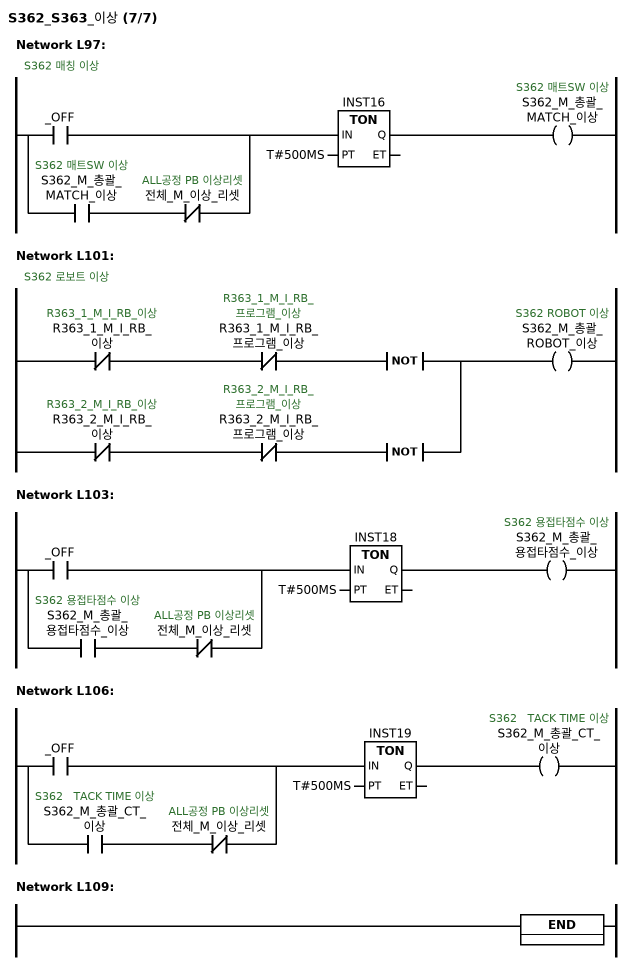
(* [picture p144: S362_S363_이상 rungs L97-L109] *)
(* S362 매칭 이상 *)
(* Rung L97 *)
INST16(IN := _OFF OR (S362_M_총괄_MATCH_이상 AND NOT 전체_M_이상_리셋), PT := T#500MS);
S362_M_총괄_MATCH_이상 := INST16.Q;
(* S362 로보트 이상 *)
(* Rung L101 *)
S362_M_총괄_ROBOT_이상 := NOT (NOT R363_1_M_I_RB_이상 AND NOT R363_1_M_I_RB_프로그램_이상) OR NOT (NOT R363_2_M_I_RB_이상 AND NOT R363_2_M_I_RB_프로그램_이상);
(* Rung L103 *)
INST18(IN := _OFF OR (S362_M_총괄_용접타점수_이상 AND NOT 전체_M_이상_리셋), PT := T#500MS);
S362_M_총괄_용접타점수_이상 := INST18.Q;
(* Rung L106 *)
INST19(IN := _OFF OR (S362_M_총괄_CT_이상 AND NOT 전체_M_이상_리셋), PT := T#500MS);
S362_M_총괄_CT_이상 := INST19.Q;
(* Rung L109 *)
END();
END_PROGRAM

PROGRAM S364_유틸리티 (* task: 스캔 프로그램 *)
VAR_EXTERNAL
    EGIS_CWS : BOOL;
    HOP_PBL_운전준비_ON : BOOL; (* AT %MW87500.0 *) (* HOP_PBL_운전준비_ON *)
    HOP_PLB_362_4_자동_운전 : BOOL; (* AT %MW87500.4 *) (* HOP PLB 362~4 자동기동 *)
    HOP_SSP_362_4_수동_선택 : BOOL; (* AT %MW87500.3 *) (* HOP 362~4 수동선택 *)
    HOP_SSP_362_4_자동_선택 : BOOL; (* AT %MW87500.2 *) (* HOP 362~4 자동선택 *)
    MCP_PBL_362_4_자동_운전 : BOOL; (* AT %MW87630.4 *) (* MCP PBL 362~4 자동기동 *)
    MCP_PBL_운전준비_ON : BOOL; (* AT %MW87630.0 *) (* MCP_PBL_운전준비_ON *)
    MCP_SPB_작업완료_RESET : BOOL; (* AT %MW87631.6 *) (* MCP_SPB_작업완료_RESET *)
    MCP_SPB_작업완료_SET : BOOL; (* AT %MW87631.7 *) (* MCP_SPB_작업완료_SET *)
    MCP_SSP_362_4_수동_선택 : BOOL; (* AT %MW87630.2 *) (* MCP 362~4 수동선택 *)
    MCP_SSP_362_4_자동_선택 : BOOL; (* AT %MW87630.3 *) (* MCP 362~4 자동동선택 *)
    R361_1_M_I_RB_1차_작업완료 : BOOL; (* AT %MW20011.2 *) (* R361_1_M_I_RB_1차_작업완료 *)
    R361_1_M_I_RB_2차_작업완료 : BOOL; (* AT %MW20011.3 *) (* R361_1_M_I_RB_2차_작업완료 *)
    R361_2_M_I_RB_2차_작업완료 : BOOL; (* AT %MW20021.3 *) (* R361_2_M_I_RB_2차_작업완료 *)
    R361_2_M_I_RB_간섭무_1 : BOOL; (* AT %MW20022.0 *) (* R361_2_M_I_RB_간섭무_1 *)
    R361_2_M_I_RB_원위치 : BOOL; (* AT %MW20020.3 *) (* R361_2_M_I_RB_원위치 *)
    R363_2_M_I_RB_간섭무_1 : BOOL; (* AT %MW20042.0 *) (* R363_2_M_I_RB_간섭무_1 *)
    R363_2_M_I_RB_원위치 : BOOL; (* AT %MW20040.3 *) (* R363_2_M_I_RB_원위치 *)
    R364_1_M_I_RB_1차_작업완료 : BOOL; (* AT %MW20051.2 *) (* R364_1_M_I_RB_1차_작업완료 *)
    R364_1_M_I_RB_간섭무_1 : BOOL; (* AT %MW20052.0 *) (* R364_1_M_I_RB_간섭무_1 *)
    R364_1_M_I_RB_원위치 : BOOL; (* AT %MW20050.3 *) (* R364_1_M_I_RB_원위치 *)
    S362_LC_정상1 : BOOL; (* AT %MW87105.3 *)
    S362_LC_정상2 : BOOL; (* AT %MW87105.4 *)
    S362_MAT_정상1 : BOOL; (* AT %MW87105.6 *)
    S362_MAT_정상2 : BOOL; (* AT %MW87105.7 *)
    S364_LC_정상1 : BOOL; (* AT %MW87165.3 *)
    S364_LC_정상2 : BOOL; (* AT %MW87165.4 *)
    S364_MAT_정상1 : BOOL; (* AT %MW87165.6 *)
    S364_MAT_정상2 : BOOL; (* AT %MW87165.7 *)
    S364_PB_AX_작업_완료 : BOOL; (* AT %MW87152.9 *) (* S364_PB_AX_작업_완료 *)
    S364_PRS_AX_LH_RACK_CHK1 : BOOL; (* AT %MW87162.0 *) (* S364_PRS_AX_LH_RACK_CHK1 *)
    S364_PRS_AX_LH_RACK_CHK2 : BOOL; (* AT %MW87162.1 *) (* S364_PRS_AX_LH_RACK_CHK2 *)
    S364_PRS_AX_LH_RACK_CHK3 : BOOL; (* AT %MW87162.2 *) (* S364_PRS_AX_LH_RACK_CHK3 *)
    S364_PRS_AX_LH_ROOF_FRT_CHK : BOOL; (* AT %MW87162.3 *) (* S364_PRS_AX_LH_ROOF_FRT_CHK *)
    S364_PRS_AX_LH_ROOF_RR_CHK : BOOL; (* AT %MW87162.4 *) (* S364_PRS_AX_LH_ROOF_RR_CHK *)
    S364_PRS_AX_RH_RACK_CHK1 : BOOL; (* AT %MW87152.0 *) (* S364_PRS_AX_RH_RACK_CHK1 *)
    S364_PRS_AX_RH_RACK_CHK2 : BOOL; (* AT %MW87152.1 *) (* S364_PRS_AX_RH_RACK_CHK2 *)
    S364_PRS_AX_RH_RACK_CHK3 : BOOL; (* AT %MW87152.2 *) (* S364_PRS_AX_RH_RACK_CHK3 *)
    S364_PRS_AX_RH_ROOF_FRT_CHK : BOOL; (* AT %MW87152.3 *) (* S364_PRS_AX_RH_ROOF_FRT_CHK *)
    S364_PRS_AX_RH_ROOF_RR_CHK : BOOL; (* AT %MW87152.4 *) (* S364_PRS_AX_RH_ROOF_RR_CHK *)
END_VAR
VAR_EXTERNAL RETAIN
    HMI_M_선택_MOD_S362 : BOOL; (* AT %MW6.0 *) (* HMI M 선택 MOD S362 *)
    HMI_M_선택_MOD_S364 : BOOL; (* AT %MW6.2 *) (* HMI M 선택 MOD S364 *)
    S362_M_BYPASS_보조 : BOOL; (* AT %MW1003.15 *) (* S362 M BYPASS 보조 *)
    S362_M_LC_정상 : BOOL; (* AT %MW1007.5 *) (* S362_M_LC_정상 *)
    S362_M_MAT_정상 : BOOL; (* AT %MW1007.6 *) (* S362_M_MAT_정상 *)
    S362_M_SAFETY_불간섭 : BOOL; (* AT %MW1004.4 *) (* S362_M_SAFETY_불간섭 *)
    S362_M_공정_차종_무 : BOOL; (* AT %MW1002.1 *) (* S362_M_공정_차종_무 *)
    S362_M_공정_차종_유 : BOOL; (* AT %MW1002.0 *) (* S362_M_공정_차종_유 *)
    S362_M_작업완료_SET_PLS : BOOL; (* AT %MW1000.8 *) (* S362 M 작업완료 SET PLS *)
    S362_M_작업완료_리셋_PLS : BOOL; (* AT %MW1000.9 *) (* S362 M 작업완료 리셋 PLS *)
    S362_M_총괄_이상 : BOOL; (* AT %MW1009.0 *) (* S362_M_총괄_이상 *)
    S364_M_AX_CLAMP_전진단 : BOOL; (* AT %MW2101.3 *) (* S364_M_AX_CLAMP_전진단 *)
    S364_M_AX_CLAMP_후진단 : BOOL; (* AT %MW2101.4 *) (* S364_M_AX_CLAMP_후진단 *)
    S364_M_AX_LATCH_전진단 : BOOL; (* AT %MW2100.3 *) (* S364_M_AX_LATCH_전진단 *)
    S364_M_AX_LATCH_후진단 : BOOL; (* AT %MW2100.4 *) (* S364_M_AX_LATCH_후진단 *)
    S364_M_AX_LH_SLD_CLP_전진단 : BOOL; (* AT %MW2103.3 *) (* S364_M_AX_LH_SLD_CLP_전진단 *)
    S364_M_AX_LH_SLD_CLP_후진단 : BOOL; (* AT %MW2103.4 *) (* S364_M_AX_LH_SLD_CLP_후진단 *)
    S364_M_AX_LH_SLD_LAT_전진단 : BOOL; (* AT %MW2102.3 *) (* S364_M_AX_LH_SLD_LAT_전진단 *)
    S364_M_AX_LH_SLD_LAT_후진단 : BOOL; (* AT %MW2102.4 *) (* S364_M_AX_LH_SLD_LAT_후진단 *)
    S364_M_AX_LH_SLD_전진단 : BOOL; (* AT %MW2107.3 *) (* S364_M_AX_LH_SLD_전진단 *)
    S364_M_AX_LH_SLD_후진단 : BOOL; (* AT %MW2107.4 *) (* S364_M_AX_LH_SLD_후진단 *)
    S364_M_AX_RH_SLD_CLP_전진단 : BOOL; (* AT %MW2111.3 *) (* S364_M_AX_RH_SLD_CLP_전진단 *)
    S364_M_AX_RH_SLD_CLP_후진단 : BOOL; (* AT %MW2111.4 *) (* S364_M_AX_RH_SLD_CLP_후진단 *)
    S364_M_AX_RH_SLD_LAT_전진단 : BOOL; (* AT %MW2110.3 *) (* S364_M_AX_RH_SLD_LAT_전진단 *)
    S364_M_AX_RH_SLD_LAT_후진단 : BOOL; (* AT %MW2110.4 *) (* S364_M_AX_RH_SLD_LAT_후진단 *)
    S364_M_AX_RH_SLD_전진단 : BOOL; (* AT %MW2115.3 *) (* S364_M_AX_RH_SLD_전진단 *)
    S364_M_AX_RH_SLD_후진단 : BOOL; (* AT %MW2115.4 *) (* S364_M_AX_RH_SLD_후진단 *)
    S364_M_BYPASS_보조 : BOOL; (* AT %MW2003.15 *) (* S364 M BYPASS 보조 *)
    S364_M_CTR_RACK_제품감지_무 : BOOL; (* AT %MW2002.9 *)
    S364_M_CTR_RACK_제품감지_유 : BOOL; (* AT %MW2002.8 *)
    S364_M_FRT_PNL_제품감지_무 : BOOL; (* AT %MW2002.13 *)
    S364_M_FRT_PNL_제품감지_유 : BOOL; (* AT %MW2002.12 *)
    S364_M_FRT_RACK_제품감지_무 : BOOL; (* AT %MW2002.7 *)
    S364_M_FRT_RACK_제품감지_유 : BOOL; (* AT %MW2002.6 *)
    S364_M_LC_정상 : BOOL; (* AT %MW2007.5 *) (* S364_M_LC_정상 *)
    S364_M_MAT_정상 : BOOL; (* AT %MW2007.6 *) (* S364_M_MAT_정상 *)
    S364_M_R361_1_언로딩완료 : BOOL; (* AT %MW2001.4 *)
    S364_M_R361_2_로딩가능 : BOOL; (* AT %MW2004.9 *)
    S364_M_R361_2_로딩완료 : BOOL; (* AT %MW2001.2 *)
    S364_M_R364_1_용접가능 : BOOL; (* AT %MW2004.10 *)
    S364_M_R364_1_용접완료 : BOOL; (* AT %MW2001.3 *)
    S364_M_RR_PNL_제품감지_무 : BOOL; (* AT %MW2002.15 *)
    S364_M_RR_PNL_제품감지_유 : BOOL; (* AT %MW2002.14 *)
    S364_M_RR_RACK_제품감지_무 : BOOL; (* AT %MW2002.11 *)
    S364_M_RR_RACK_제품감지_유 : BOOL; (* AT %MW2002.10 *)
    S364_M_SAFETY_불간섭 : BOOL; (* AT %MW2004.4 *) (* S364_M_SAFETY_불간섭 *)
    S364_M_SEQ : WORD; (* AT %MW10120 *) (* S364 M SEQ *)
    S364_M_공정_불간섭 : BOOL; (* AT %MW2004.1 *) (* S364_M_공정_불간섭 *)
    S364_M_공정_원위치 : BOOL; (* AT %MW2004.0 *) (* S364_M_공정_원위치 *)
    S364_M_공정_제품감지_무 : BOOL; (* AT %MW2002.5 *) (* S364_M_공정_제품감지_무 *)
    S364_M_공정_제품감지_유 : BOOL; (* AT %MW2002.4 *) (* S364_M_공정_제품감지_유 *)
    S364_M_공정_차종_무 : BOOL; (* AT %MW2002.1 *) (* S364_M_공정_차종_무 *)
    S364_M_공정_차종_유 : BOOL; (* AT %MW2002.0 *) (* S364_M_공정_차종_유 *)
    S364_M_수동모드 : BOOL; (* AT %MW2000.3 *) (* S364 선택 수동모드 *)
    S364_M_운전준비_ON : BOOL; (* AT %MW2000.0 *) (* S364 운전준비 ON *)
    S364_M_자동_START : BOOL; (* AT %MW2000.5 *) (* S364 자동운전중 *)
    S364_M_자동_운전중 : BOOL; (* AT %MW2000.4 *) (* S364 자동운전중 *)
    S364_M_자동모드 : BOOL; (* AT %MW2000.1 *) (* S364 선택 자동모드 *)
    S364_M_작업_완료 : BOOL; (* AT %MW2001.0 *) (* S364_M_작업_완료 *)
    S364_M_작업완료_SET_PLS : BOOL; (* AT %MW2000.8 *) (* S364 M 작업완료 SET PLS *)
    S364_M_작업완료_리셋_PLS : BOOL; (* AT %MW2000.9 *) (* S364 M 작업완료 리셋 PLS *)
    S364_M_작업자_작업가능 : BOOL; (* AT %MW2004.8 *)
    S364_M_작업자_작업완료 : BOOL; (* AT %MW2001.1 *)
    S364_M_차종1_AX : BOOL; (* AT %MW10121.0 *) (* S364 M 차종1 AX *)
    S364_M_차종1_B : BOOL; (* AT %MW10121.1 *) (* S364 M 차종1 B *)
    S364_M_차종1_C : BOOL; (* AT %MW10121.2 *) (* S364 M 차종1 C *)
    S364_M_차종1_D : BOOL; (* AT %MW10121.3 *) (* S364 M 차종1 D *)
    S364_M_차종1_E : BOOL; (* AT %MW10121.4 *) (* S364 M 차종1 E *)
    S364_M_차종1_F : BOOL; (* AT %MW10121.5 *) (* S364 M 차종1 F *)
    S364_M_차종1_G : BOOL; (* AT %MW10121.6 *) (* S364 M 차종1 G *)
    S364_M_차종1_H : BOOL; (* AT %MW10121.7 *) (* S364 M 차종1 H *)
    S364_M_차종2_3DR : BOOL; (* AT %MW10121.8 *) (* S364 M 차종2 3DR *)
    S364_M_차종2_4DR : BOOL; (* AT %MW10121.9 *) (* S364 M 차종2 4DR *)
    S364_M_차종2_5DR : BOOL; (* AT %MW10121.10 *) (* S364 M 차종2 5DR *)
    S364_M_차종2_SP1 : BOOL; (* AT %MW10121.12 *) (* S364 M 차종2 SP1 *)
    S364_M_차종2_SP2 : BOOL; (* AT %MW10121.13 *) (* S364 M 차종2 SP2 *)
    S364_M_차종2_WGN : BOOL; (* AT %MW10121.11 *) (* S364 M 차종2 WGN *)
    S364_M_차종3_LHD : BOOL; (* AT %MW10121.14 *) (* S364 M 차종3 LHD *)
    S364_M_차종3_RHD : BOOL; (* AT %MW10121.15 *) (* S364 M 차종3 RHD *)
    S364_M_차종4_EEC : BOOL; (* AT %MW10122.3 *) (* S364 M 차종4 EEC *)
    S364_M_차종4_SP1 : BOOL; (* AT %MW10122.8 *) (* S364 M 차종4 SP1 *)
    S364_M_차종4_SP2 : BOOL; (* AT %MW10122.9 *) (* S364 M 차종4 SP2 *)
    S364_M_차종4_SP3 : BOOL; (* AT %MW10122.11 *) (* S364 M 차종4 SP3 *)
    S364_M_차종4_SP4 : BOOL; (* AT %MW10122.12 *) (* S364 M 차종4 SP4 *)
    S364_M_차종4_SP5 : BOOL; (* AT %MW10122.13 *) (* S364 M 차종4 SP5 *)
    S364_M_차종4_SP6 : BOOL; (* AT %MW10122.14 *) (* S364 M 차종4 SP6 *)
    S364_M_차종4_SP7 : BOOL; (* AT %MW10122.15 *) (* S364 M 차종4 SP7 *)
    S364_M_차종4_내수 : BOOL; (* AT %MW10122.0 *) (* S364 M 차종4 내수 *)
    S364_M_차종4_러시아 : BOOL; (* AT %MW10122.10 *) (* S364 M 차종4 러시아 *)
    S364_M_차종4_북미 : BOOL; (* AT %MW10122.2 *) (* S364 M 차종4 북미 *)
    S364_M_차종4_브라질 : BOOL; (* AT %MW10122.7 *) (* S364 M 차종4 브라질 *)
    S364_M_차종4_수출 : BOOL; (* AT %MW10122.1 *) (* S364 M 차종4 수출 *)
    S364_M_차종4_중국 : BOOL; (* AT %MW10122.6 *) (* S364 M 차종4 중국 *)
    S364_M_차종4_중동 : BOOL; (* AT %MW10122.5 *) (* S364 M 차종4 중동 *)
    S364_M_차종4_호주 : BOOL; (* AT %MW10122.4 *) (* S364 M 차종4 호주 *)
    S364_M_차종5_AT : BOOL; (* AT %MW10123.1 *) (* S364 M 차종5 AT *)
    S364_M_차종5_MT : BOOL; (* AT %MW10123.0 *) (* S364 M 차종5 MT *)
    S364_M_차종5_SP1 : BOOL; (* AT %MW10123.2 *) (* S364 M 차종5 SP1 *)
    S364_M_차종6_DSROOF : BOOL; (* AT %MW10123.6 *) (* S364 M 차종6 DSROOF *)
    S364_M_차종6_SP1 : BOOL; (* AT %MW10123.7 *) (* S364 M 차종6 SP1 *)
    S364_M_차종6_썬루프 : BOOL; (* AT %MW10123.4 *) (* S364 M 차종6 썬루프 *)
    S364_M_차종6_일반루프 : BOOL; (* AT %MW10123.3 *) (* S364 M 차종6 일반루프 *)
    S364_M_차종6_파노라마루프 : BOOL; (* AT %MW10123.5 *) (* S364 M 차종6 파노라마루프 *)
    S364_M_차종7_DSL : BOOL; (* AT %MW10123.9 *) (* S364 M 차종7 DSL *)
    S364_M_차종7_GSL : BOOL; (* AT %MW10123.8 *) (* S364 M 차종7 GSL *)
    S364_M_차종7_SP1 : BOOL; (* AT %MW10123.10 *) (* S364 M 차종7 SP1 *)
    S364_M_차종7_SP2 : BOOL; (* AT %MW10123.11 *) (* S364 M 차종7 SP2 *)
    S364_M_차종7_SP3 : BOOL; (* AT %MW10123.12 *) (* S364 M 차종7 SP3 *)
    S364_M_차종7_SP4 : BOOL; (* AT %MW10123.13 *) (* S364 M 차종7 SP4 *)
    S364_M_차종7_SP5 : BOOL; (* AT %MW10123.14 *) (* S364 M 차종7 SP5 *)
    S364_M_차종7_SP6 : BOOL; (* AT %MW10123.15 *) (* S364 M 차종7 SP6 *)
    S364_M_차종8_2WD : BOOL; (* AT %MW10124.0 *) (* S364 M 차종8 2WD *)
    S364_M_차종8_4WD : BOOL; (* AT %MW10124.1 *) (* S364 M 차종8 4WD *)
    S364_M_차종8_SP1 : BOOL; (* AT %MW10124.2 *) (* S364 M 차종8 SP1 *)
    S364_M_차종9_MPI : BOOL; (* AT %MW10124.3 *) (* S364 M 차종9 MPI *)
    S364_M_차종9_SP1 : BOOL; (* AT %MW10124.5 *) (* S364 M 차종9 SP1 *)
    S364_M_차종9_SP10 : BOOL; (* AT %MW10124.14 *) (* S364 M 차종9 SP10 *)
    S364_M_차종9_SP11 : BOOL; (* AT %MW10124.15 *) (* S364 M 차종9 SP11 *)
    S364_M_차종9_SP2 : BOOL; (* AT %MW10124.6 *) (* S364 M 차종9 SP2 *)
    S364_M_차종9_SP3 : BOOL; (* AT %MW10124.7 *) (* S364 M 차종9 SP3 *)
    S364_M_차종9_SP4 : BOOL; (* AT %MW10124.8 *) (* S364 M 차종9 SP4 *)
    S364_M_차종9_SP5 : BOOL; (* AT %MW10124.9 *) (* S364 M 차종9 SP5 *)
    S364_M_차종9_SP6 : BOOL; (* AT %MW10124.10 *) (* S364 M 차종9 SP6 *)
    S364_M_차종9_SP7 : BOOL; (* AT %MW10124.11 *) (* S364 M 차종9 SP7 *)
    S364_M_차종9_SP8 : BOOL; (* AT %MW10124.12 *) (* S364 M 차종9 SP8 *)
    S364_M_차종9_SP9 : BOOL; (* AT %MW10124.13 *) (* S364 M 차종9 SP9 *)
    S364_M_차종9_T_GDI : BOOL; (* AT %MW10124.4 *) (* S364 M 차종9 T GDI *)
    S364_M_차종_OPT1_R_RACK_무 : BOOL; (* AT %MW10125.3 *) (* S364 M 차종 OPT1 R RACK 무 *)
    S364_M_차종_OPT1_R_RACK_유 : BOOL; (* AT %MW10125.2 *) (* S364 M 차종 OPT1 R RACK 유 *)
    S364_M_차종_OPT1_S_REP_EATER_무 : BOOL; (* AT %MW10125.7 *) (* S364 M 차종 OPT1 S REP EATER 무 *)
    S364_M_차종_OPT1_S_REP_EATER_유 : BOOL; (* AT %MW10125.6 *) (* S364 M 차종 OPT1 S REP EATER 유 *)
    S364_M_차종_OPT1_VAN_무 : BOOL; (* AT %MW10125.9 *) (* S364 M 차종 OPT1 VAN 무 *)
    S364_M_차종_OPT1_VAN_유 : BOOL; (* AT %MW10125.8 *) (* S364 M 차종 OPT1 VAN 유 *)
    S364_M_차종_OPT1_슬라이딩_무 : BOOL; (* AT %MW10125.1 *) (* S364 M 차종 OPT1 슬라이딩 무 *)
    S364_M_차종_OPT1_슬라이딩_유 : BOOL; (* AT %MW10125.0 *) (* S364 M 차종 OPT1 슬라이딩 유 *)
    S364_M_차종_OPT1_폴딩_무 : BOOL; (* AT %MW10125.5 *) (* S364 M 차종 OPT1 폴딩 무 *)
    S364_M_차종_OPT1_폴딩_유 : BOOL; (* AT %MW10125.4 *) (* S364 M 차종 OPT1 폴딩 유 *)
    S364_M_차종_공대차 : BOOL; (* AT %MW10130.12 *) (* S364 M 차종 공대차 *)
    S364_M_차종_공차 : BOOL; (* AT %MW10130.10 *) (* S364 M 차종 공차 *)
    S364_M_차종_불량차 : BOOL; (* AT %MW10130.11 *) (* S364 M 차종 불량차 *)
    S364_M_총괄_이상 : BOOL; (* AT %MW2009.0 *) (* S364_M_총괄_이상 *)
    전체_M_GATE_자동기동 : BOOL; (* AT %MW308.1 *) (* 전체_M_자동_운전 *)
    전체_라인_M_총괄_SAFETY_이상 : BOOL; (* AT %MW300.2 *) (* ALL공정 SAFETY  이상총괄 *)
    전체_라인_M_총괄_공기압_이상 : BOOL; (* AT %MW300.3 *) (* ALL공정 공기압 이상총괄 *)
    전체_라인_M_총괄_비상정지_이상 : BOOL; (* AT %MW300.1 *) (* ALL공정 비상정지 이상총괄 *)
    전체_라인_M_총괄_이상 : BOOL; (* AT %MW300.0 *) (* ALL공정 총괄이상 *)
END_VAR
VAR
    S364_READY : TON;
    T364_AUTO : TON;
END_VAR
VAR
    _t1 : BOOL;
    _e2 : R_TRIG;
END_VAR

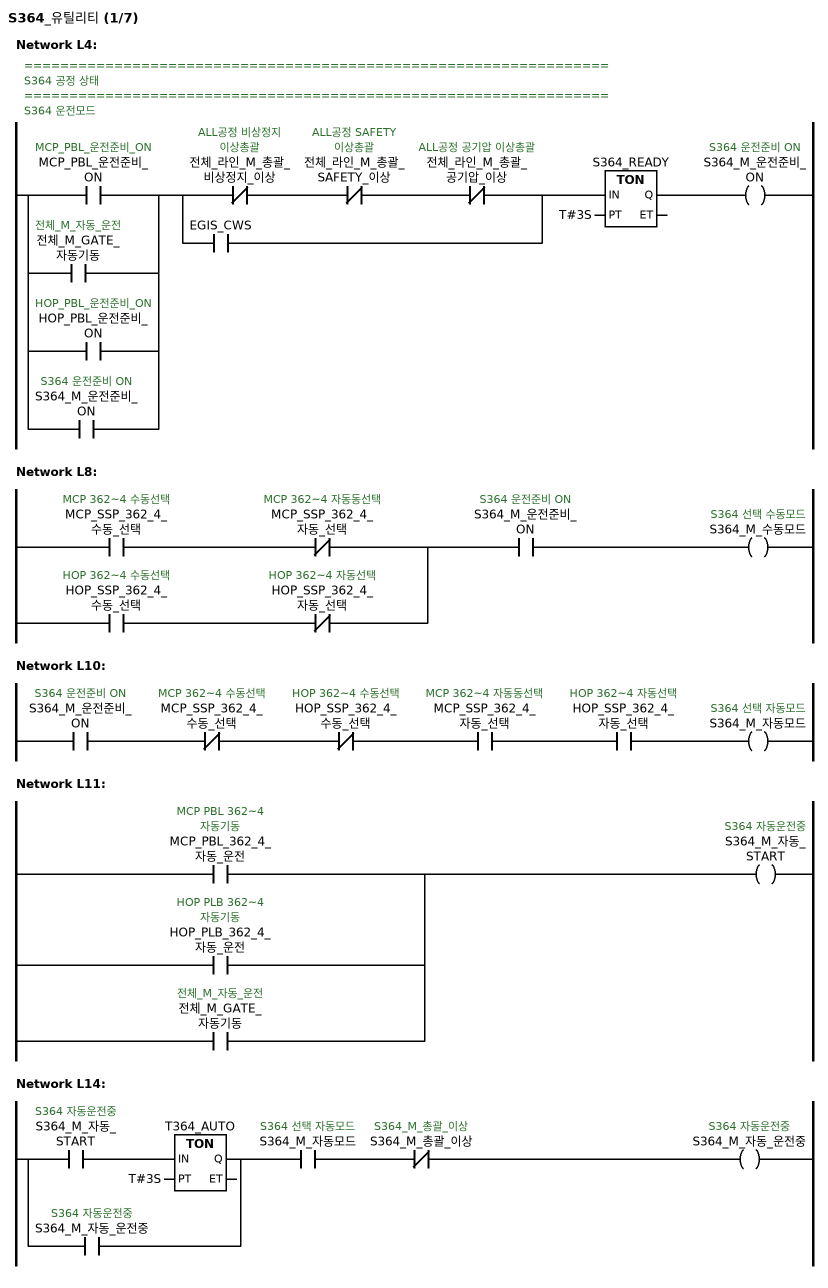
(* ================================================================= *)
(* S364 공정 상태 *)
(* ================================================================= *)
(* S364 운전모드 *)
(* Rung L4 *)
S364_READY(IN := (MCP_PBL_운전준비_ON OR 전체_M_GATE_자동기동 OR HOP_PBL_운전준비_ON OR S364_M_운전준비_ON) AND ((NOT 전체_라인_M_총괄_비상정지_이상 AND NOT 전체_라인_M_총괄_SAFETY_이상 AND NOT 전체_라인_M_총괄_공기압_이상) OR EGIS_CWS), PT := T#3S);
S364_M_운전준비_ON := S364_READY.Q;
(* Rung L8 *)
S364_M_수동모드 := ((MCP_SSP_362_4_수동_선택 AND NOT MCP_SSP_362_4_자동_선택) OR (HOP_SSP_362_4_수동_선택 AND NOT HOP_SSP_362_4_자동_선택)) AND S364_M_운전준비_ON;
(* Rung L10 *)
S364_M_자동모드 := S364_M_운전준비_ON AND NOT MCP_SSP_362_4_수동_선택 AND NOT HOP_SSP_362_4_수동_선택 AND MCP_SSP_362_4_자동_선택 AND HOP_SSP_362_4_자동_선택;
(* Rung L11 *)
S364_M_자동_START := MCP_PBL_362_4_자동_운전 OR HOP_PLB_362_4_자동_운전 OR 전체_M_GATE_자동기동;
(* Rung L14 *)
T364_AUTO(IN := S364_M_자동_START, PT := T#3S);
S364_M_자동_운전중 := (T364_AUTO.Q OR S364_M_자동_운전중) AND S364_M_자동모드 AND NOT S364_M_총괄_이상;

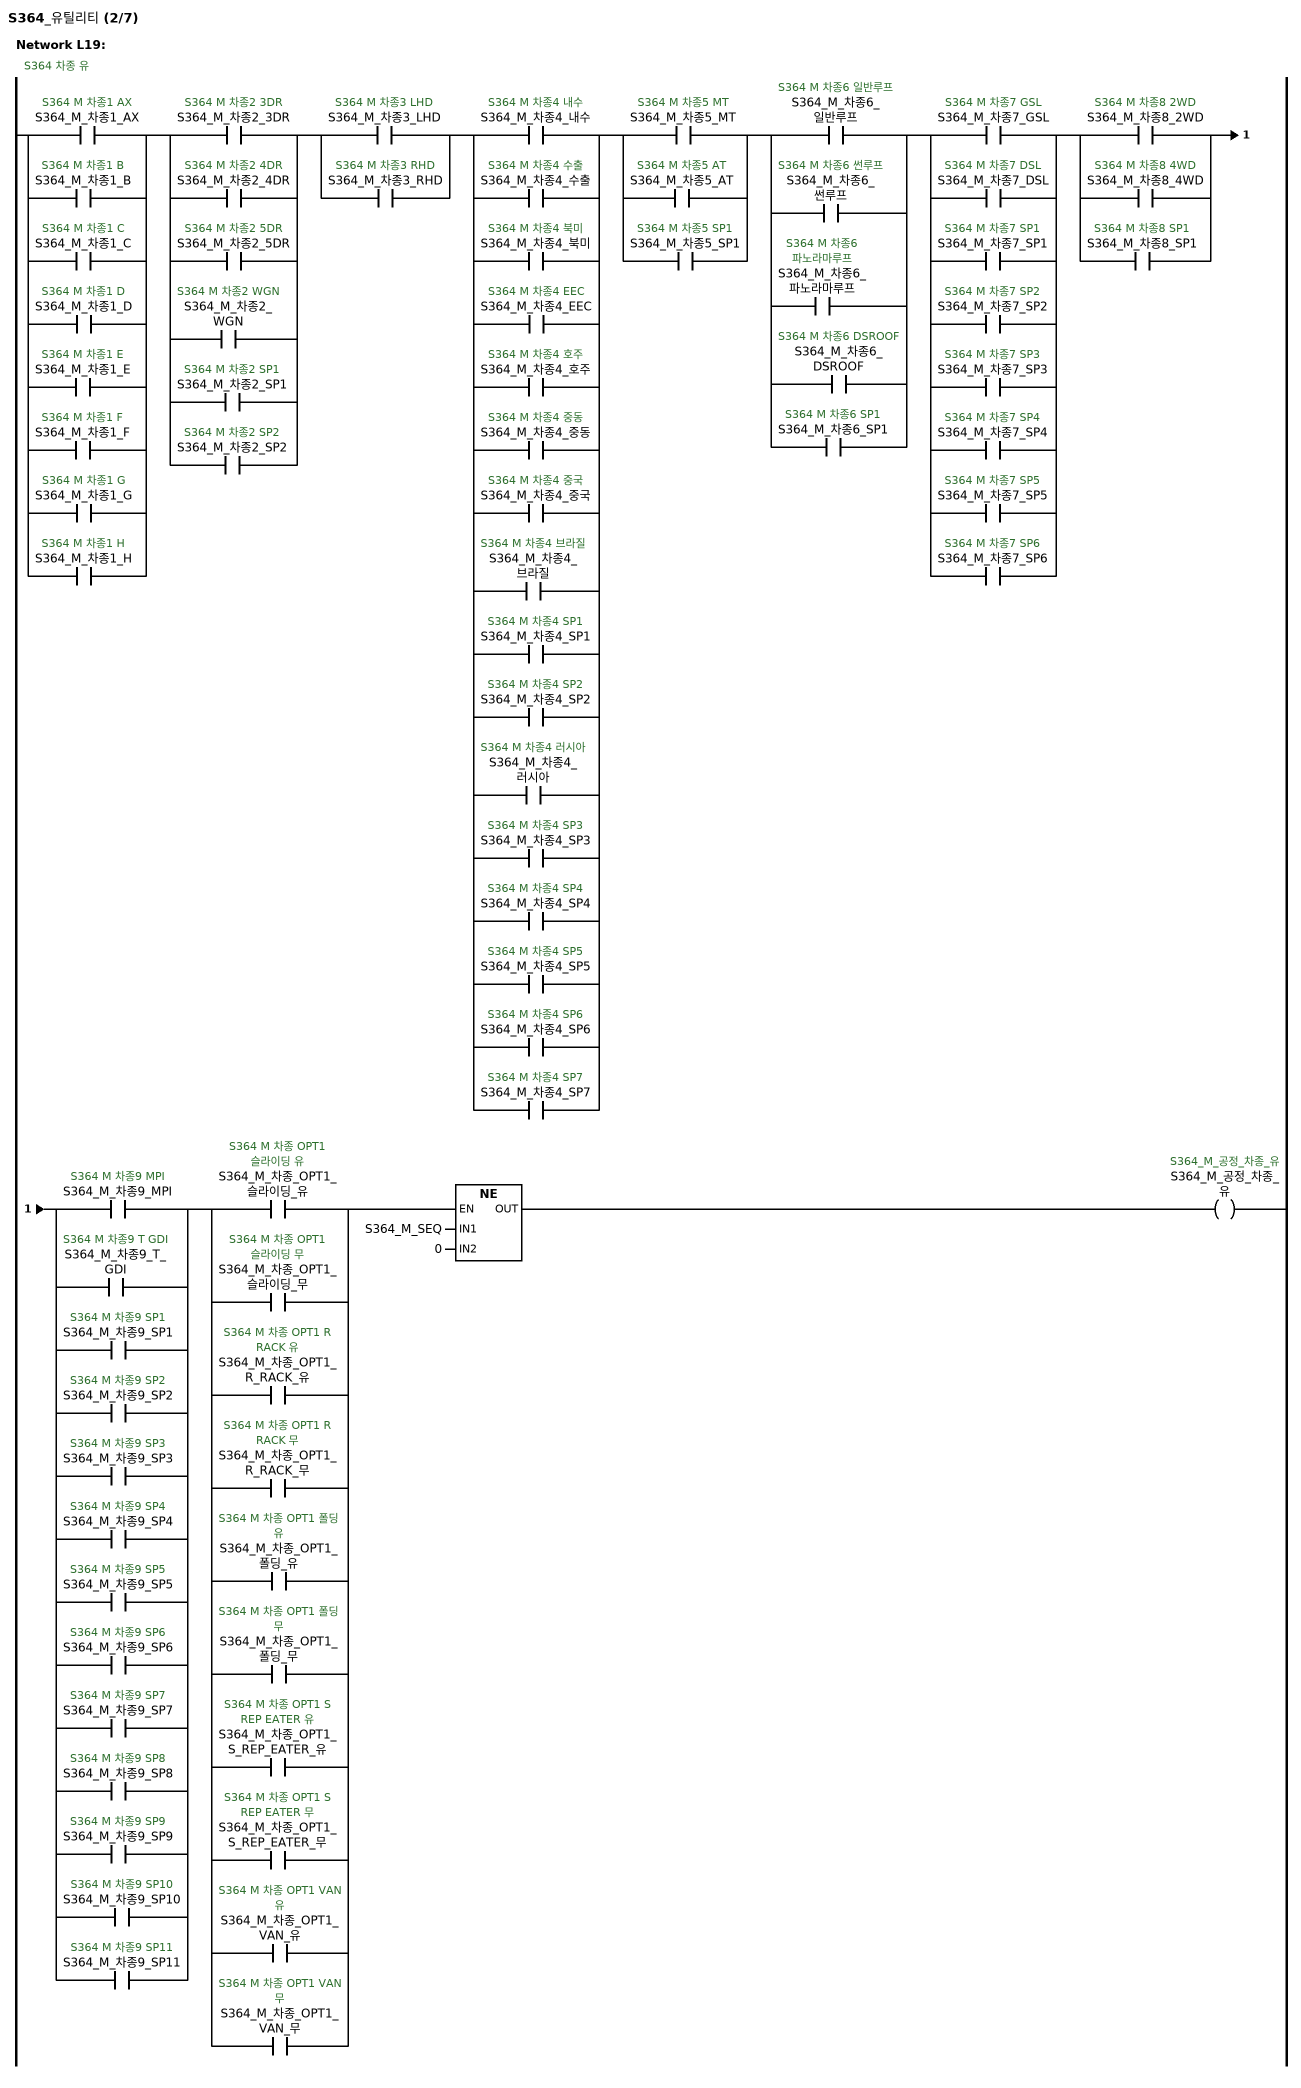
(* S364 차종 유 *)
(* Rung L19 *)
IF (S364_M_차종1_AX OR S364_M_차종1_B OR S364_M_차종1_C OR S364_M_차종1_D OR S364_M_차종1_E OR S364_M_차종1_F OR S364_M_차종1_G OR S364_M_차종1_H) AND (S364_M_차종2_3DR OR S364_M_차종2_4DR OR S364_M_차종2_5DR OR S364_M_차종2_WGN OR S364_M_차종2_SP1 OR S364_M_차종2_SP2) AND (S364_M_차종3_LHD OR S364_M_차종3_RHD) AND (S364_M_차종4_내수 OR S364_M_차종4_수출 OR S364_M_차종4_북미 OR S364_M_차종4_EEC OR S364_M_차종4_호주 OR S364_M_차종4_중동 OR S364_M_차종4_중국 OR S364_M_차종4_브라질 OR S364_M_차종4_SP1 OR S364_M_차종4_SP2 OR S364_M_차종4_러시아 OR S364_M_차종4_SP3 OR S364_M_차종4_SP4 OR S364_M_차종4_SP5 OR S364_M_차종4_SP6 OR S364_M_차종4_SP7) AND (S364_M_차종5_MT OR S364_M_차종5_AT OR S364_M_차종5_SP1) AND (S364_M_차종6_일반루프 OR S364_M_차종6_썬루프 OR S364_M_차종6_파노라마루프 OR S364_M_차종6_DSROOF OR S364_M_차종6_SP1) AND (S364_M_차종7_GSL OR S364_M_차종7_DSL OR S364_M_차종7_SP1 OR S364_M_차종7_SP2 OR S364_M_차종7_SP3 OR S364_M_차종7_SP4 OR S364_M_차종7_SP5 OR S364_M_차종7_SP6) AND (S364_M_차종8_2WD OR S364_M_차종8_4WD OR S364_M_차종8_SP1) AND (S364_M_차종9_MPI OR S364_M_차종9_T_GDI OR S364_M_차종9_SP1 OR S364_M_차종9_SP2 OR S364_M_차종9_SP3 OR S364_M_차종9_SP4 OR S364_M_차종9_SP5 OR S364_M_차종9_SP6 OR S364_M_차종9_SP7 OR S364_M_차종9_SP8 OR S364_M_차종9_SP9 OR S364_M_차종9_SP10 OR S364_M_차종9_SP11) AND (S364_M_차종_OPT1_슬라이딩_유 OR S364_M_차종_OPT1_슬라이딩_무 OR S364_M_차종_OPT1_R_RACK_유 OR S364_M_차종_OPT1_R_RACK_무 OR S364_M_차종_OPT1_폴딩_유 OR S364_M_차종_OPT1_폴딩_무 OR S364_M_차종_OPT1_S_REP_EATER_유 OR S364_M_차종_OPT1_S_REP_EATER_무 OR S364_M_차종_OPT1_VAN_유 OR S364_M_차종_OPT1_VAN_무) THEN
    _t1 := S364_M_SEQ <> 0;
END_IF;
S364_M_공정_차종_유 := _t1;

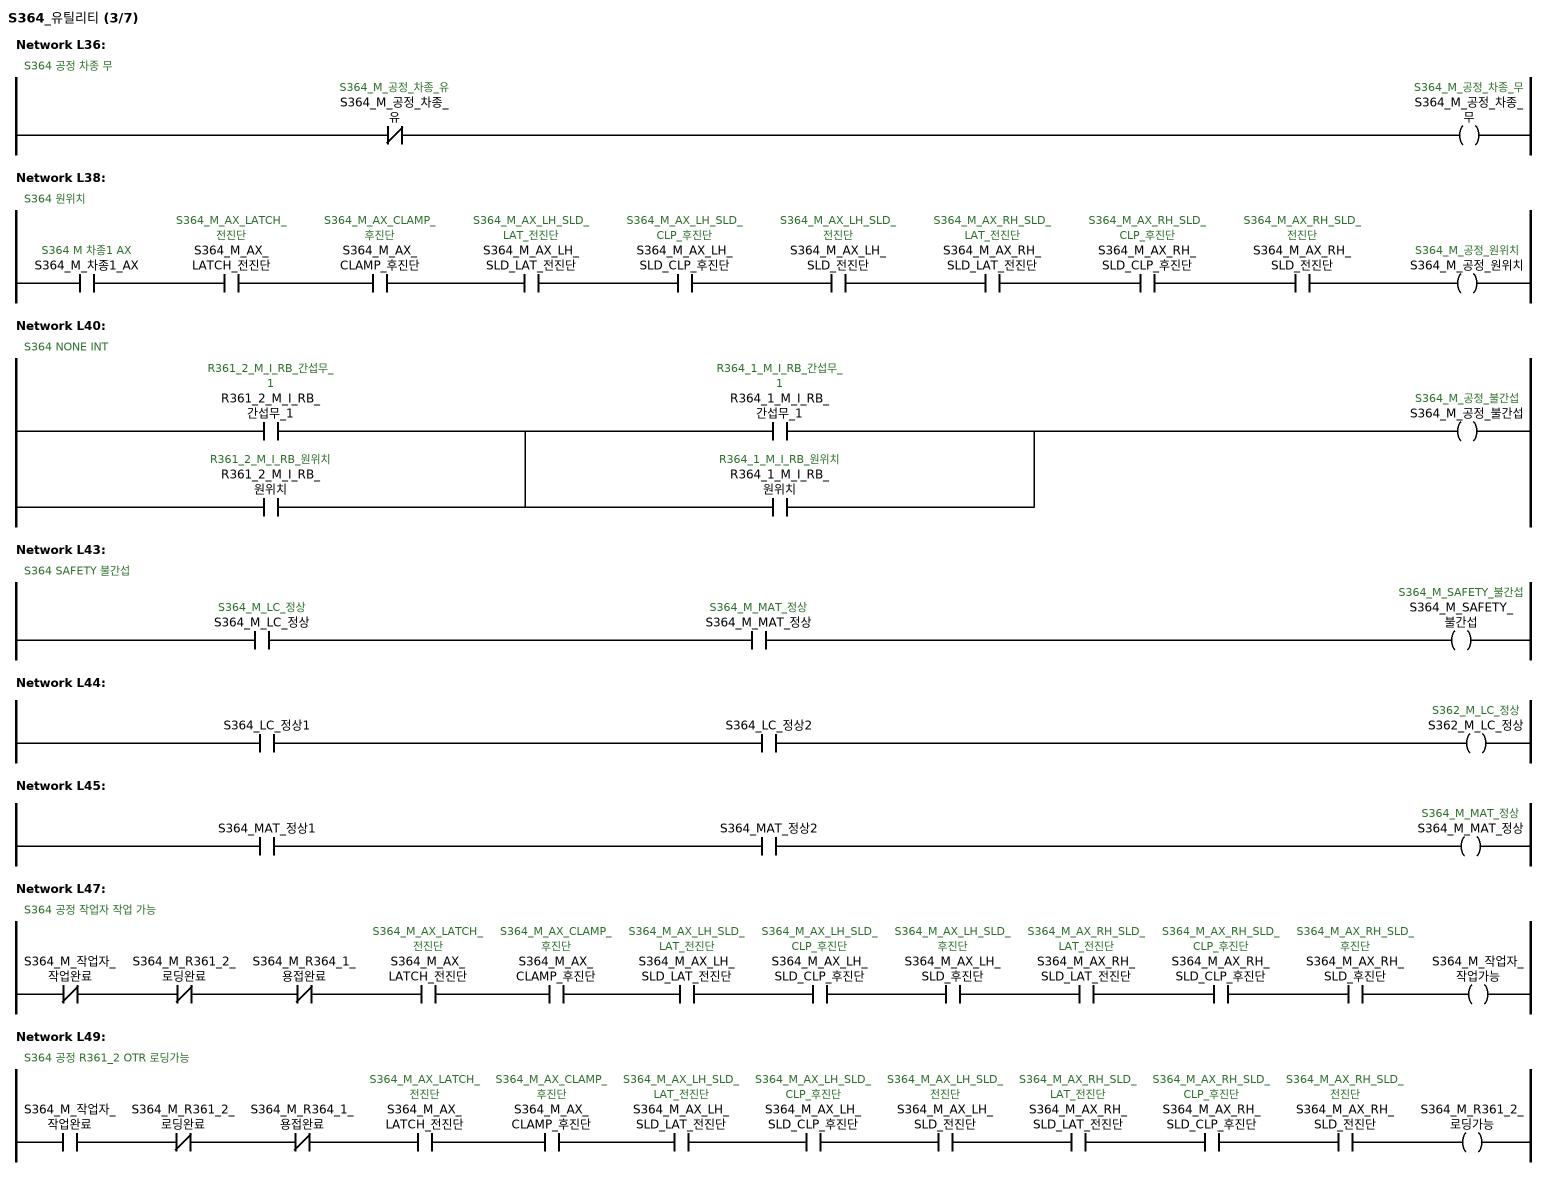
(* S364 공정 차종 무 *)
(* Rung L36 *)
S364_M_공정_차종_무 := NOT S364_M_공정_차종_유;
(* S364 원위치 *)
(* Rung L38 *)
S364_M_공정_원위치 := S364_M_차종1_AX AND S364_M_AX_LATCH_전진단 AND S364_M_AX_CLAMP_후진단 AND S364_M_AX_LH_SLD_LAT_전진단 AND S364_M_AX_LH_SLD_CLP_후진단 AND S364_M_AX_LH_SLD_전진단 AND S364_M_AX_RH_SLD_LAT_전진단 AND S364_M_AX_RH_SLD_CLP_후진단 AND S364_M_AX_RH_SLD_전진단;
(* S364 NONE INT *)
(* Rung L40 *)
S364_M_공정_불간섭 := (R361_2_M_I_RB_간섭무_1 OR R361_2_M_I_RB_원위치) AND (R364_1_M_I_RB_간섭무_1 OR R364_1_M_I_RB_원위치);
(* S364 SAFETY 불간섭 *)
(* Rung L43 *)
S364_M_SAFETY_불간섭 := S364_M_LC_정상 AND S364_M_MAT_정상;
(* Rung L44 *)
S362_M_LC_정상 := S364_LC_정상1 AND S364_LC_정상2;
(* Rung L45 *)
S364_M_MAT_정상 := S364_MAT_정상1 AND S364_MAT_정상2;
(* S364 공정 작업자 작업 가능 *)
(* Rung L47 *)
S364_M_작업자_작업가능 := NOT S364_M_작업자_작업완료 AND NOT S364_M_R361_2_로딩완료 AND NOT S364_M_R364_1_용접완료 AND S364_M_AX_LATCH_전진단 AND S364_M_AX_CLAMP_후진단 AND S364_M_AX_LH_SLD_LAT_전진단 AND S364_M_AX_LH_SLD_CLP_후진단 AND S364_M_AX_LH_SLD_후진단 AND S364_M_AX_RH_SLD_LAT_전진단 AND S364_M_AX_RH_SLD_CLP_후진단 AND S364_M_AX_RH_SLD_후진단;
(* S364 공정 R361_2 OTR 로딩가능 *)
(* Rung L49 *)
S364_M_R361_2_로딩가능 := S364_M_작업자_작업완료 AND NOT S364_M_R361_2_로딩완료 AND NOT S364_M_R364_1_용접완료 AND S364_M_AX_LATCH_전진단 AND S364_M_AX_CLAMP_후진단 AND S364_M_AX_LH_SLD_LAT_전진단 AND S364_M_AX_LH_SLD_CLP_후진단 AND S364_M_AX_LH_SLD_전진단 AND S364_M_AX_RH_SLD_LAT_전진단 AND S364_M_AX_RH_SLD_CLP_후진단 AND S364_M_AX_RH_SLD_전진단;

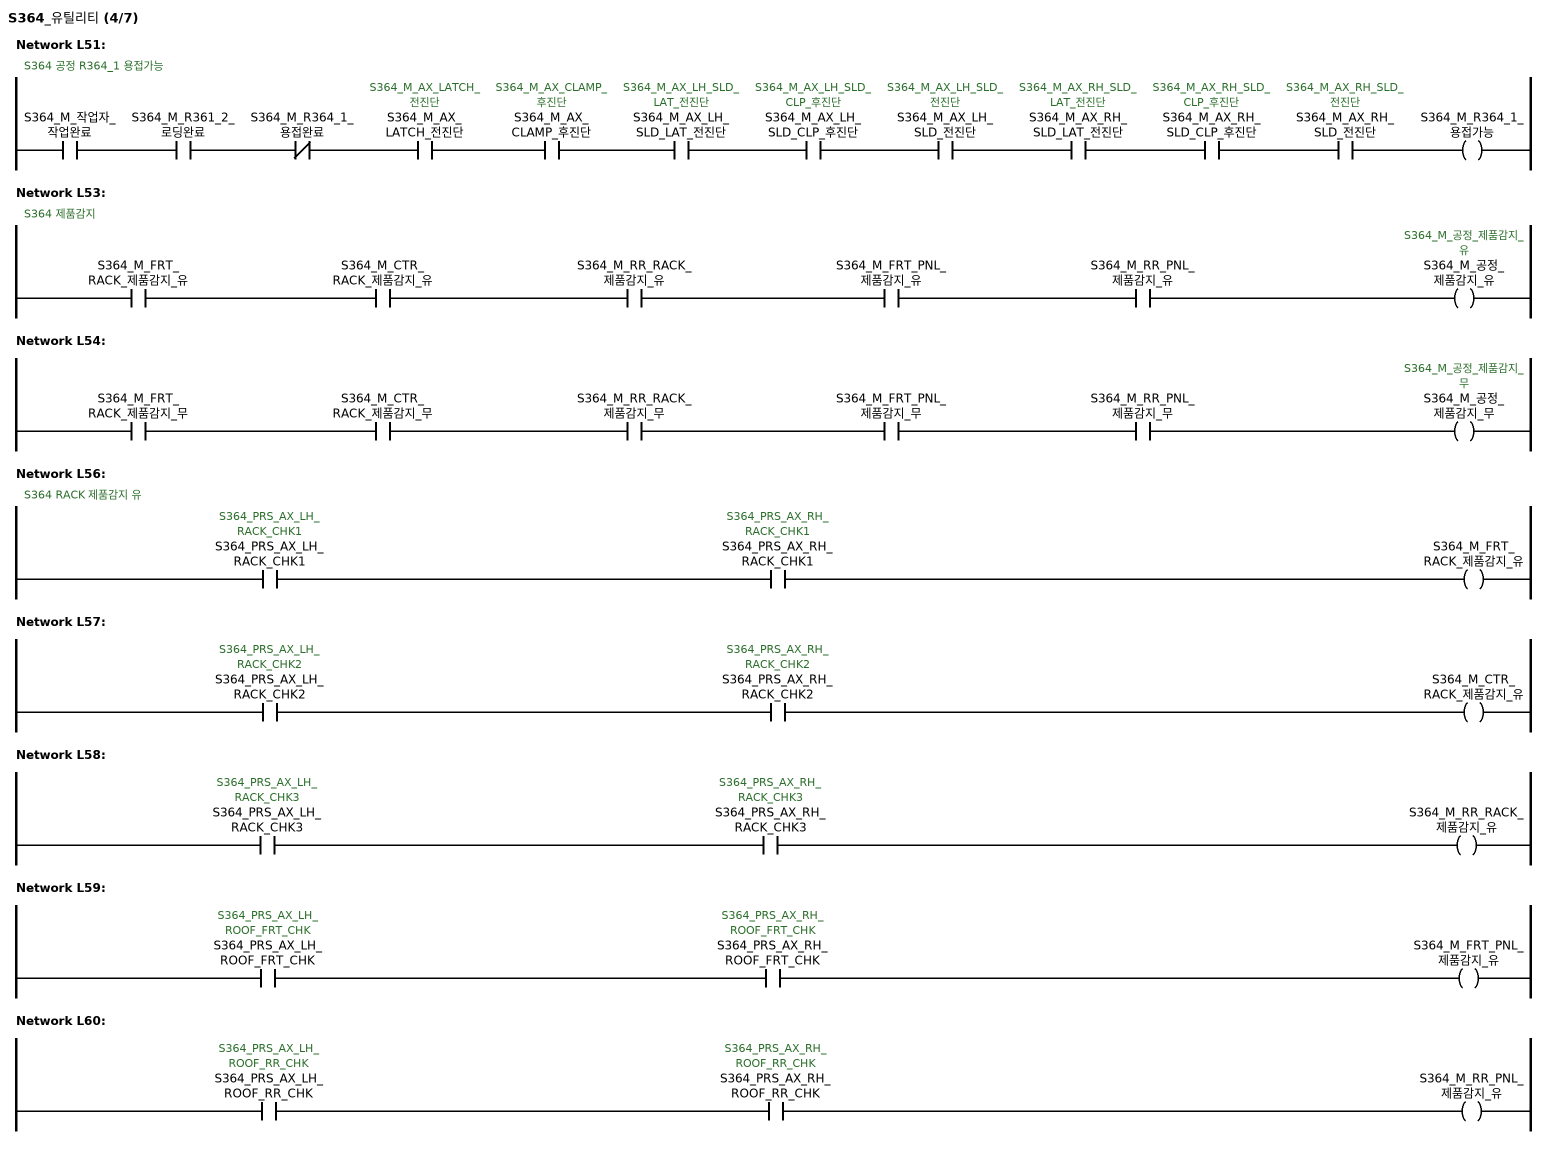
(* S364 공정 R364_1 용접가능 *)
(* Rung L51 *)
S364_M_R364_1_용접가능 := S364_M_작업자_작업완료 AND S364_M_R361_2_로딩완료 AND NOT S364_M_R364_1_용접완료 AND S364_M_AX_LATCH_전진단 AND S364_M_AX_CLAMP_후진단 AND S364_M_AX_LH_SLD_LAT_전진단 AND S364_M_AX_LH_SLD_CLP_후진단 AND S364_M_AX_LH_SLD_전진단 AND S364_M_AX_RH_SLD_LAT_전진단 AND S364_M_AX_RH_SLD_CLP_후진단 AND S364_M_AX_RH_SLD_전진단;
(* S364 제품감지 *)
(* Rung L53 *)
S364_M_공정_제품감지_유 := S364_M_FRT_RACK_제품감지_유 AND S364_M_CTR_RACK_제품감지_유 AND S364_M_RR_RACK_제품감지_유 AND S364_M_FRT_PNL_제품감지_유 AND S364_M_RR_PNL_제품감지_유;
(* Rung L54 *)
S364_M_공정_제품감지_무 := S364_M_FRT_RACK_제품감지_무 AND S364_M_CTR_RACK_제품감지_무 AND S364_M_RR_RACK_제품감지_무 AND S364_M_FRT_PNL_제품감지_무 AND S364_M_RR_PNL_제품감지_무;
(* S364 RACK 제품감지 유 *)
(* Rung L56 *)
S364_M_FRT_RACK_제품감지_유 := S364_PRS_AX_LH_RACK_CHK1 AND S364_PRS_AX_RH_RACK_CHK1;
(* Rung L57 *)
S364_M_CTR_RACK_제품감지_유 := S364_PRS_AX_LH_RACK_CHK2 AND S364_PRS_AX_RH_RACK_CHK2;
(* Rung L58 *)
S364_M_RR_RACK_제품감지_유 := S364_PRS_AX_LH_RACK_CHK3 AND S364_PRS_AX_RH_RACK_CHK3;
(* Rung L59 *)
S364_M_FRT_PNL_제품감지_유 := S364_PRS_AX_LH_ROOF_FRT_CHK AND S364_PRS_AX_RH_ROOF_FRT_CHK;
(* Rung L60 *)
S364_M_RR_PNL_제품감지_유 := S364_PRS_AX_LH_ROOF_RR_CHK AND S364_PRS_AX_RH_ROOF_RR_CHK;

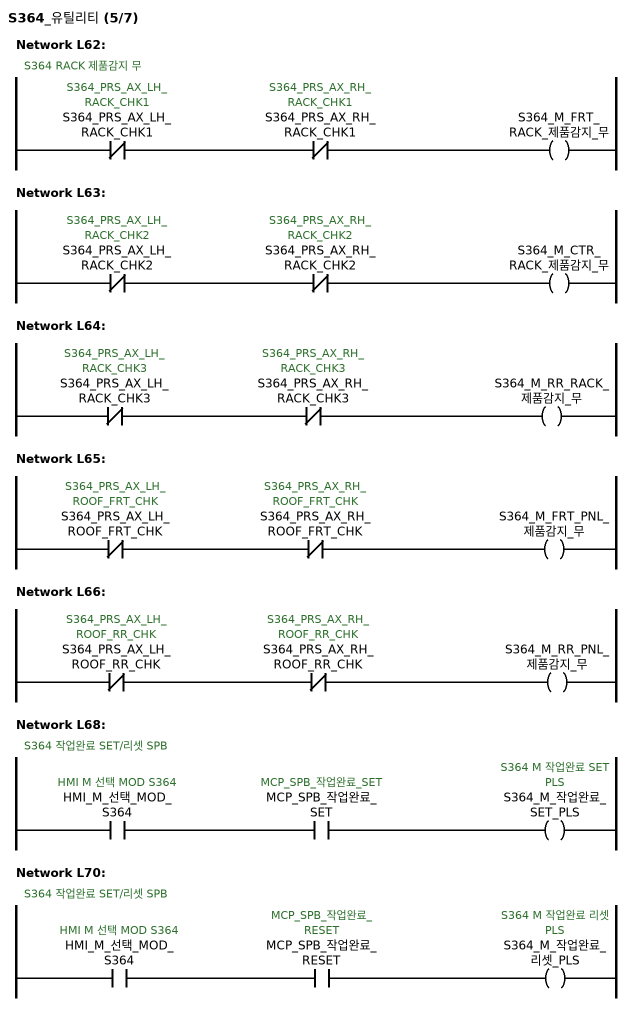
(* S364 RACK 제품감지 무 *)
(* Rung L62 *)
S364_M_FRT_RACK_제품감지_무 := NOT S364_PRS_AX_LH_RACK_CHK1 AND NOT S364_PRS_AX_RH_RACK_CHK1;
(* Rung L63 *)
S364_M_CTR_RACK_제품감지_무 := NOT S364_PRS_AX_LH_RACK_CHK2 AND NOT S364_PRS_AX_RH_RACK_CHK2;
(* Rung L64 *)
S364_M_RR_RACK_제품감지_무 := NOT S364_PRS_AX_LH_RACK_CHK3 AND NOT S364_PRS_AX_RH_RACK_CHK3;
(* Rung L65 *)
S364_M_FRT_PNL_제품감지_무 := NOT S364_PRS_AX_LH_ROOF_FRT_CHK AND NOT S364_PRS_AX_RH_ROOF_FRT_CHK;
(* Rung L66 *)
S364_M_RR_PNL_제품감지_무 := NOT S364_PRS_AX_LH_ROOF_RR_CHK AND NOT S364_PRS_AX_RH_ROOF_RR_CHK;
(* S364 작업완료 SET/리셋 SPB *)
(* Rung L68 *)
S364_M_작업완료_SET_PLS := HMI_M_선택_MOD_S364 AND MCP_SPB_작업완료_SET;
(* S364 작업완료 SET/리셋 SPB *)
(* Rung L70 *)
S364_M_작업완료_리셋_PLS := HMI_M_선택_MOD_S364 AND MCP_SPB_작업완료_RESET;

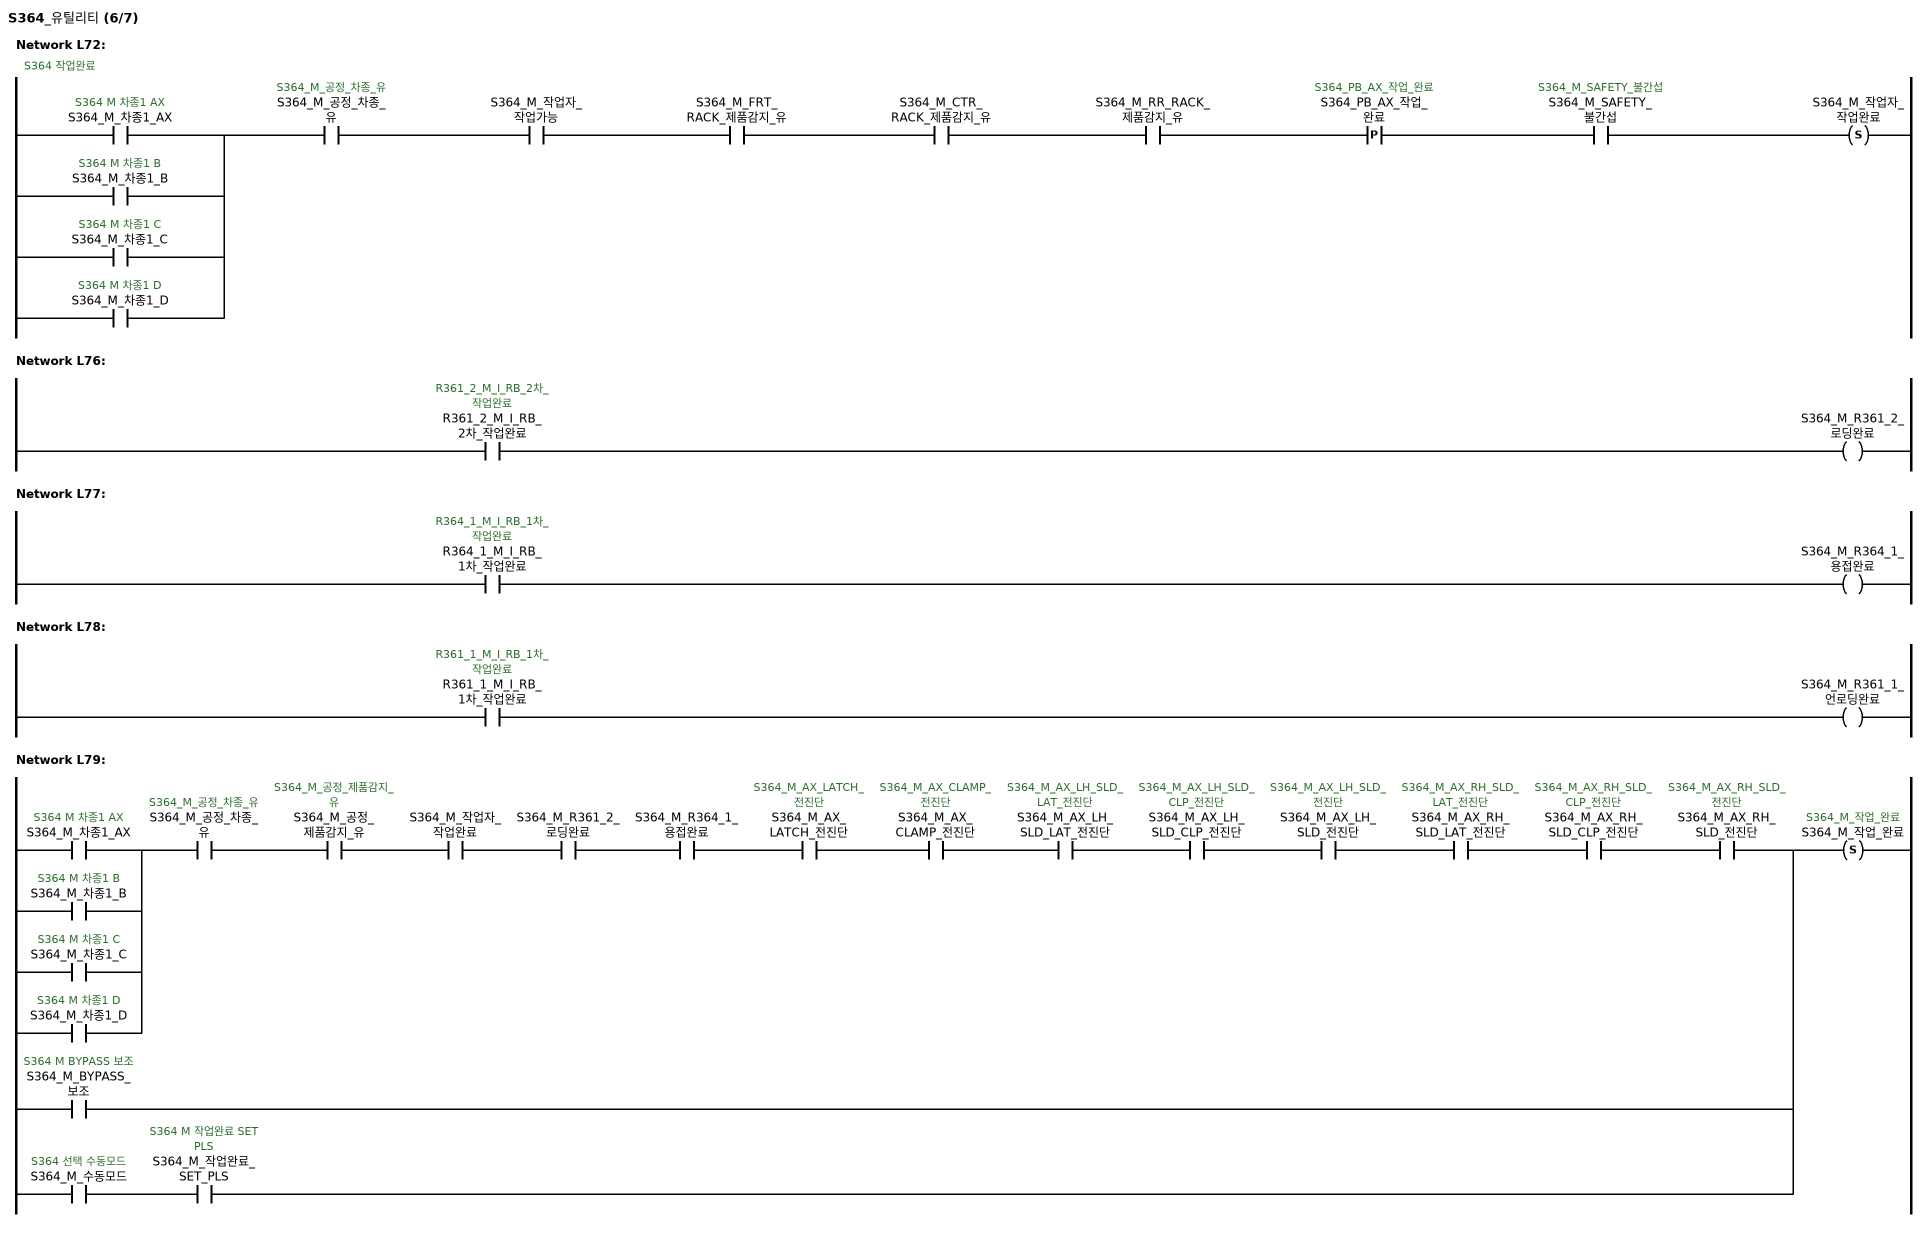
(* S364 작업완료 *)
(* Rung L72 *)
_e2(CLK := S364_PB_AX_작업_완료);
IF (S364_M_차종1_AX OR S364_M_차종1_B OR S364_M_차종1_C OR S364_M_차종1_D) AND S364_M_공정_차종_유 AND S364_M_작업자_작업가능 AND S364_M_FRT_RACK_제품감지_유 AND S364_M_CTR_RACK_제품감지_유 AND S364_M_RR_RACK_제품감지_유 AND _e2.Q AND S364_M_SAFETY_불간섭 THEN
    S364_M_작업자_작업완료 := TRUE;
END_IF;
(* Rung L76 *)
S364_M_R361_2_로딩완료 := R361_2_M_I_RB_2차_작업완료;
(* Rung L77 *)
S364_M_R364_1_용접완료 := R364_1_M_I_RB_1차_작업완료;
(* Rung L78 *)
S364_M_R361_1_언로딩완료 := R361_1_M_I_RB_1차_작업완료;
(* Rung L79 *)
IF ((S364_M_차종1_AX OR S364_M_차종1_B OR S364_M_차종1_C OR S364_M_차종1_D) AND S364_M_공정_차종_유 AND S364_M_공정_제품감지_유 AND S364_M_작업자_작업완료 AND S364_M_R361_2_로딩완료 AND S364_M_R364_1_용접완료 AND S364_M_AX_LATCH_전진단 AND S364_M_AX_CLAMP_전진단 AND S364_M_AX_LH_SLD_LAT_전진단 AND S364_M_AX_LH_SLD_CLP_전진단 AND S364_M_AX_LH_SLD_전진단 AND S364_M_AX_RH_SLD_LAT_전진단 AND S364_M_AX_RH_SLD_CLP_전진단 AND S364_M_AX_RH_SLD_전진단) OR S364_M_BYPASS_보조 OR (S364_M_수동모드 AND S364_M_작업완료_SET_PLS) THEN
    S364_M_작업_완료 := TRUE;
END_IF;

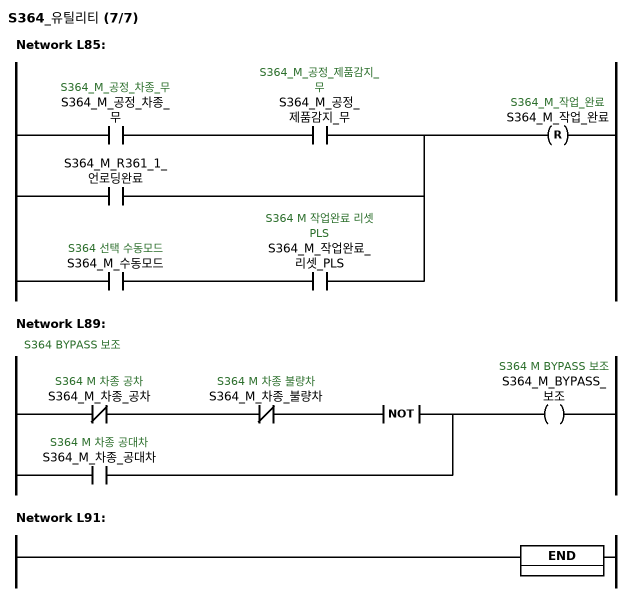
(* Rung L85 *)
IF (S364_M_공정_차종_무 AND S364_M_공정_제품감지_무) OR S364_M_R361_1_언로딩완료 OR (S364_M_수동모드 AND S364_M_작업완료_리셋_PLS) THEN
    S364_M_작업_완료 := FALSE;
END_IF;
(* S364 BYPASS 보조 *)
(* Rung L89 *)
S364_M_BYPASS_보조 := NOT (NOT S364_M_차종_공차 AND NOT S364_M_차종_불량차) OR S364_M_차종_공대차;
(* Rung L91 *)
END();
END_PROGRAM

PROGRAM S364_동작 (* task: 스캔 프로그램 *)
VAR_EXTERNAL RETAIN
    ALWAYS_ON : BOOL; (* AT %MW3.1 *) (* 항시 ON *)
    S364_HOME : BOOL; (* AT %MW2048.0 *) (* S364_HOME *)
    S364_M_AX_CLAMP_전진_LS_이상 : BOOL; (* AT %MW2101.5 *) (* S364_M_AX_CLAMP_전진_LS_이상 *)
    S364_M_AX_CLAMP_전진_보조 : BOOL; (* AT %MW2101.1 *) (* S364_M_AX_CLAMP_전진_보조 *)
    S364_M_AX_CLAMP_전진단 : BOOL; (* AT %MW2101.3 *) (* S364_M_AX_CLAMP_전진단 *)
    S364_M_AX_CLAMP_조건 : BOOL; (* AT %MW2101.0 *) (* S364_M_AX_CLAMP_조건 *)
    S364_M_AX_CLAMP_후진_LS_이상 : BOOL; (* AT %MW2101.6 *) (* S364_M_AX_CLAMP_후진_LS_이상 *)
    S364_M_AX_CLAMP_후진_보조 : BOOL; (* AT %MW2101.2 *) (* S364_M_AX_CLAMP_후진_보조 *)
    S364_M_AX_CLAMP_후진단 : BOOL; (* AT %MW2101.4 *) (* S364_M_AX_CLAMP_후진단 *)
    S364_M_AX_LATCH_전진_LS_이상 : BOOL; (* AT %MW2100.5 *) (* S364_M_AX_LATCH_전진_LS_이상 *)
    S364_M_AX_LATCH_전진_보조 : BOOL; (* AT %MW2100.1 *) (* S364_M_AX_LATCH_전진_보조 *)
    S364_M_AX_LATCH_전진단 : BOOL; (* AT %MW2100.3 *) (* S364_M_AX_LATCH_전진단 *)
    S364_M_AX_LATCH_조건 : BOOL; (* AT %MW2100.0 *) (* S364_M_AX_LATCH_조건 *)
    S364_M_AX_LATCH_후진_LS_이상 : BOOL; (* AT %MW2100.6 *) (* S364_M_AX_LATCH_후진_LS_이상 *)
    S364_M_AX_LATCH_후진_보조 : BOOL; (* AT %MW2100.2 *) (* S364_M_AX_LATCH_후진_보조 *)
    S364_M_AX_LATCH_후진단 : BOOL; (* AT %MW2100.4 *) (* S364_M_AX_LATCH_후진단 *)
    S364_M_AX_LH_SLD_CLP_전진_LS_이상 : BOOL; (* AT %MW2103.5 *) (* S364_M_AX_LH_SLD_CLP_전진_LS_이상 *)
    S364_M_AX_LH_SLD_CLP_전진_보조 : BOOL; (* AT %MW2103.1 *) (* S364_M_AX_LH_SLD_CLP_전진_보조 *)
    S364_M_AX_LH_SLD_CLP_전진단 : BOOL; (* AT %MW2103.3 *) (* S364_M_AX_LH_SLD_CLP_전진단 *)
    S364_M_AX_LH_SLD_CLP_조건 : BOOL; (* AT %MW2103.0 *) (* S364_M_AX_LH_SLD_CLP_조건 *)
    S364_M_AX_LH_SLD_CLP_후진_LS_이상 : BOOL; (* AT %MW2103.6 *) (* S364_M_AX_LH_SLD_CLP_후진_LS_이상 *)
    S364_M_AX_LH_SLD_CLP_후진_보조 : BOOL; (* AT %MW2103.2 *) (* S364_M_AX_LH_SLD_CLP_후진_보조 *)
    S364_M_AX_LH_SLD_CLP_후진단 : BOOL; (* AT %MW2103.4 *) (* S364_M_AX_LH_SLD_CLP_후진단 *)
    S364_M_AX_LH_SLD_LAT_전진_LS_이상 : BOOL; (* AT %MW2102.5 *) (* S364_M_AX_LH_SLD_LAT_전진_LS_이상 *)
    S364_M_AX_LH_SLD_LAT_전진_보조 : BOOL; (* AT %MW2102.1 *) (* S364_M_AX_LH_SLD_LAT_전진_보조 *)
    S364_M_AX_LH_SLD_LAT_전진단 : BOOL; (* AT %MW2102.3 *) (* S364_M_AX_LH_SLD_LAT_전진단 *)
    S364_M_AX_LH_SLD_LAT_조건 : BOOL; (* AT %MW2102.0 *) (* S364_M_AX_LH_SLD_LAT_조건 *)
    S364_M_AX_LH_SLD_LAT_후진_LS_이상 : BOOL; (* AT %MW2102.6 *) (* S364_M_AX_LH_SLD_LAT_후진_LS_이상 *)
    S364_M_AX_LH_SLD_LAT_후진_보조 : BOOL; (* AT %MW2102.2 *) (* S364_M_AX_LH_SLD_LAT_후진_보조 *)
    S364_M_AX_LH_SLD_LAT_후진단 : BOOL; (* AT %MW2102.4 *) (* S364_M_AX_LH_SLD_LAT_후진단 *)
    S364_M_AX_LH_SLD_전진_LS_이상 : BOOL; (* AT %MW2107.5 *) (* S364_M_AX_LH_SLD_전진_LS_이상 *)
    S364_M_AX_LH_SLD_전진_보조 : BOOL; (* AT %MW2107.1 *) (* S364_M_AX_LH_SLD_전진_보조 *)
    S364_M_AX_LH_SLD_전진단 : BOOL; (* AT %MW2107.3 *) (* S364_M_AX_LH_SLD_전진단 *)
    S364_M_AX_LH_SLD_조건 : BOOL; (* AT %MW2107.0 *) (* S364_M_AX_LH_SLD_조건 *)
    S364_M_AX_LH_SLD_후진_LS_이상 : BOOL; (* AT %MW2107.6 *) (* S364_M_AX_LH_SLD_후진_LS_이상 *)
    S364_M_AX_LH_SLD_후진_보조 : BOOL; (* AT %MW2107.2 *) (* S364_M_AX_LH_SLD_후진_보조 *)
    S364_M_AX_LH_SLD_후진단 : BOOL; (* AT %MW2107.4 *) (* S364_M_AX_LH_SLD_후진단 *)
    S364_M_AX_RH_SLD_CLP_전진_LS_이상 : BOOL; (* AT %MW2111.5 *) (* S364_M_AX_RH_SLD_CLP_전진_LS_이상 *)
    S364_M_AX_RH_SLD_CLP_전진_보조 : BOOL; (* AT %MW2111.1 *) (* S364_M_AX_RH_SLD_CLP_전진_보조 *)
    S364_M_AX_RH_SLD_CLP_전진단 : BOOL; (* AT %MW2111.3 *) (* S364_M_AX_RH_SLD_CLP_전진단 *)
    S364_M_AX_RH_SLD_CLP_조건 : BOOL; (* AT %MW2111.0 *) (* S364_M_AX_RH_SLD_CLP_조건 *)
    S364_M_AX_RH_SLD_CLP_후진_LS_이상 : BOOL; (* AT %MW2111.6 *) (* S364_M_AX_RH_SLD_CLP_후진_LS_이상 *)
    S364_M_AX_RH_SLD_CLP_후진_보조 : BOOL; (* AT %MW2111.2 *) (* S364_M_AX_RH_SLD_CLP_후진_보조 *)
    S364_M_AX_RH_SLD_CLP_후진단 : BOOL; (* AT %MW2111.4 *) (* S364_M_AX_RH_SLD_CLP_후진단 *)
    S364_M_AX_RH_SLD_LAT_전진_LS_이상 : BOOL; (* AT %MW2110.5 *) (* S364_M_AX_RH_SLD_LAT_전진_LS_이상 *)
    S364_M_AX_RH_SLD_LAT_전진_보조 : BOOL; (* AT %MW2110.1 *) (* S364_M_AX_RH_SLD_LAT_전진_보조 *)
    S364_M_AX_RH_SLD_LAT_전진단 : BOOL; (* AT %MW2110.3 *) (* S364_M_AX_RH_SLD_LAT_전진단 *)
    S364_M_AX_RH_SLD_LAT_조건 : BOOL; (* AT %MW2110.0 *) (* S364_M_AX_RH_SLD_LAT_조건 *)
    S364_M_AX_RH_SLD_LAT_후진_LS_이상 : BOOL; (* AT %MW2110.6 *) (* S364_M_AX_RH_SLD_LAT_후진_LS_이상 *)
    S364_M_AX_RH_SLD_LAT_후진_보조 : BOOL; (* AT %MW2110.2 *) (* S364_M_AX_RH_SLD_LAT_후진_보조 *)
    S364_M_AX_RH_SLD_LAT_후진단 : BOOL; (* AT %MW2110.4 *) (* S364_M_AX_RH_SLD_LAT_후진단 *)
    S364_M_AX_RH_SLD_전진_LS_이상 : BOOL; (* AT %MW2115.5 *) (* S364_M_AX_RH_SLD_전진_LS_이상 *)
    S364_M_AX_RH_SLD_전진_보조 : BOOL; (* AT %MW2115.1 *) (* S364_M_AX_RH_SLD_전진_보조 *)
    S364_M_AX_RH_SLD_전진단 : BOOL; (* AT %MW2115.3 *) (* S364_M_AX_RH_SLD_전진단 *)
    S364_M_AX_RH_SLD_조건 : BOOL; (* AT %MW2115.0 *) (* S364_M_AX_RH_SLD_조건 *)
    S364_M_AX_RH_SLD_후진_LS_이상 : BOOL; (* AT %MW2115.6 *) (* S364_M_AX_RH_SLD_후진_LS_이상 *)
    S364_M_AX_RH_SLD_후진_보조 : BOOL; (* AT %MW2115.2 *) (* S364_M_AX_RH_SLD_후진_보조 *)
    S364_M_AX_RH_SLD_후진단 : BOOL; (* AT %MW2115.4 *) (* S364_M_AX_RH_SLD_후진단 *)
    S364_M_CTR_RACK_제품감지_유 : BOOL; (* AT %MW2002.8 *)
    S364_M_FRT_RACK_제품감지_유 : BOOL; (* AT %MW2002.6 *)
    S364_M_R361_2_로딩완료 : BOOL; (* AT %MW2001.2 *)
    S364_M_RR_RACK_제품감지_유 : BOOL; (* AT %MW2002.10 *)
    S364_M_공정_불간섭 : BOOL; (* AT %MW2004.1 *) (* S364_M_공정_불간섭 *)
    S364_M_공정_제품감지_무 : BOOL; (* AT %MW2002.5 *) (* S364_M_공정_제품감지_무 *)
    S364_M_공정_제품감지_유 : BOOL; (* AT %MW2002.4 *) (* S364_M_공정_제품감지_유 *)
    S364_M_공정_차종_무 : BOOL; (* AT %MW2002.1 *) (* S364_M_공정_차종_무 *)
    S364_M_공정_차종_유 : BOOL; (* AT %MW2002.0 *) (* S364_M_공정_차종_유 *)
    S364_M_동작_선택_1 : BOOL; (* AT %MW2040.0 *) (* S364_M_동작_선택_1 *)
    S364_M_동작_선택_11 : BOOL; (* AT %MW2040.10 *) (* S364_M_동작_선택_11 *)
    S364_M_동작_선택_12 : BOOL; (* AT %MW2040.11 *) (* S364_M_동작_선택_12 *)
    S364_M_동작_선택_16 : BOOL; (* AT %MW2040.15 *) (* S364_M_동작_선택_16 *)
    S364_M_동작_선택_2 : BOOL; (* AT %MW2040.1 *) (* S364_M_동작_선택_2 *)
    S364_M_동작_선택_3 : BOOL; (* AT %MW2040.2 *) (* S364_M_동작_선택_3 *)
    S364_M_동작_선택_4 : BOOL; (* AT %MW2040.3 *) (* S364_M_동작_선택_4 *)
    S364_M_동작_선택_8 : BOOL; (* AT %MW2040.7 *) (* S364_M_동작_선택_8 *)
    S364_M_수동모드 : BOOL; (* AT %MW2000.3 *) (* S364 선택 수동모드 *)
    S364_M_운전준비_ON : BOOL; (* AT %MW2000.0 *) (* S364 운전준비 ON *)
    S364_M_자동_운전중 : BOOL; (* AT %MW2000.4 *) (* S364 자동운전중 *)
    S364_M_작업_완료 : BOOL; (* AT %MW2001.0 *) (* S364_M_작업_완료 *)
    S364_M_작업자_작업완료 : BOOL; (* AT %MW2001.1 *)
    S364_M_차종1_AX : BOOL; (* AT %MW10121.0 *) (* S364 M 차종1 AX *)
    S364_전진_ON : BOOL; (* AT %MW2048.1 *) (* S364_전진_ON *)
    S364_후진_ON : BOOL; (* AT %MW2048.2 *) (* S364_후진_ON *)
    전체_M_이상_리셋 : BOOL; (* AT %MW308.2 *) (* ALL공정 PB 이상리셋 *)
END_VAR
VAR_EXTERNAL
    EGIS_CWS : BOOL;
    S364_M_AX_CLAMP_전진_LAMP : WORD; (* AT %MW11602 *) (* S364_M_AX_CLAMP_전진_LAMP *)
    S364_M_AX_CLAMP_후진_LAMP : WORD; (* AT %MW11603 *) (* S364_M_AX_CLAMP_후진_LAMP *)
    S364_M_AX_LATCH_전진_LAMP : WORD; (* AT %MW11600 *) (* S364_M_AX_LATCH_전진_LAMP *)
    S364_M_AX_LATCH_후진_LAMP : WORD; (* AT %MW11601 *) (* S364_M_AX_LATCH_후진_LAMP *)
    S364_M_AX_LH_SLD_CLP_전진_LAMP : WORD; (* AT %MW11606 *) (* S364_M_AX_LH_SLD_CLP_전진_LAMP *)
    S364_M_AX_LH_SLD_CLP_후진_LAMP : WORD; (* AT %MW11607 *) (* S364_M_AX_LH_SLD_CLP_후진_LAMP *)
    S364_M_AX_LH_SLD_LAT_전진_LAMP : WORD; (* AT %MW11604 *) (* S364_M_AX_LH_SLD_LAT_전진_LAMP *)
    S364_M_AX_LH_SLD_LAT_후진_LAMP : WORD; (* AT %MW11605 *) (* S364_M_AX_LH_SLD_LAT_후진_LAMP *)
    S364_M_AX_LH_SLD_전진_LAMP : WORD; (* AT %MW11614 *) (* S364_M_AX_LH_SLD_전진_LAMP *)
    S364_M_AX_LH_SLD_후진_LAMP : WORD; (* AT %MW11615 *) (* S364_M_AX_LH_SLD_후진_LAMP *)
    S364_M_AX_RH_SLD_CLP_전진_LAMP : WORD; (* AT %MW11622 *) (* S364_M_AX_RH_SLD_CLP_전진_LAMP *)
    S364_M_AX_RH_SLD_CLP_후진_LAMP : WORD; (* AT %MW11623 *) (* S364_M_AX_RH_SLD_CLP_후진_LAMP *)
    S364_M_AX_RH_SLD_LAT_전진_LAMP : WORD; (* AT %MW11620 *) (* S364_M_AX_RH_SLD_LAT_전진_LAMP *)
    S364_M_AX_RH_SLD_LAT_후진_LAMP : WORD; (* AT %MW11621 *) (* S364_M_AX_RH_SLD_LAT_후진_LAMP *)
    S364_M_AX_RH_SLD_전진_LAMP : WORD; (* AT %MW11630 *) (* S364_M_AX_RH_SLD_전진_LAMP *)
    S364_M_AX_RH_SLD_후진_LAMP : WORD; (* AT %MW11631 *) (* S364_M_AX_RH_SLD_후진_LAMP *)
    S364_RS_AX_LH_CLAMP_후진1 : BOOL; (* AT %MW87160.3 *) (* S364_RS_AX_LH_CLAMP_후진1 *)
    S364_RS_AX_LH_CLAMP_후진2 : BOOL; (* AT %MW87160.4 *) (* S364_RS_AX_LH_CLAMP_후진2 *)
    S364_RS_AX_LH_LATCH_후진1 : BOOL; (* AT %MW87160.0 *) (* S364_RS_AX_LH_LATCH_후진1 *)
    S364_RS_AX_LH_LATCH_후진2 : BOOL; (* AT %MW87160.1 *) (* S364_RS_AX_LH_LATCH_후진2 *)
    S364_RS_AX_LH_SLD_CLP_전진 : BOOL; (* AT %MW87161.0 *) (* S364_RS_AX_LH_SLD_CLP_전진 *)
    S364_RS_AX_LH_SLD_CLP_후진1 : BOOL; (* AT %MW87161.1 *) (* S364_RS_AX_LH_SLD_CLP_후진1 *)
    S364_RS_AX_LH_SLD_CLP_후진2 : BOOL; (* AT %MW87161.2 *) (* S364_RS_AX_LH_SLD_CLP_후진2 *)
    S364_RS_AX_LH_SLD_CLP_후진3 : BOOL; (* AT %MW87161.3 *) (* S364_RS_AX_LH_SLD_CLP_후진3 *)
    S364_RS_AX_LH_SLD_CLP_후진4 : BOOL; (* AT %MW87161.4 *) (* S364_RS_AX_LH_SLD_CLP_후진4 *)
    S364_RS_AX_LH_SLD_LAT_전진 : BOOL; (* AT %MW87160.8 *) (* S364_RS_AX_LH_SLD_LAT_전진 *)
    S364_RS_AX_LH_SLD_LAT_후진1 : BOOL; (* AT %MW87160.9 *) (* S364_RS_AX_LH_SLD_LAT_후진1 *)
    S364_RS_AX_LH_SLD_LAT_후진2 : BOOL; (* AT %MW87160.10 *) (* S364_RS_AX_LH_SLD_LAT_후진2 *)
    S364_RS_AX_LH_SLD_LAT_후진3 : BOOL; (* AT %MW87160.11 *) (* S364_RS_AX_LH_SLD_LAT_후진3 *)
    S364_RS_AX_LH_SLD_LAT_후진4 : BOOL; (* AT %MW87160.12 *) (* S364_RS_AX_LH_SLD_LAT_후진4 *)
    S364_RS_AX_LH_SLIDE_전진 : BOOL; (* AT %MW87151.8 *) (* S364_RS_AX_LH_SLIDE_전진 *)
    S364_RS_AX_LH_SLIDE_후진 : BOOL; (* AT %MW87151.9 *) (* S364_RS_AX_LH_SLIDE_후진 *)
    S364_RS_AX_RH_CLAMP_전진 : BOOL; (* AT %MW87150.4 *) (* S364_RS_AX_RH_CLAMP_전진 *)
    S364_RS_AX_RH_CLAMP_후진1 : BOOL; (* AT %MW87150.5 *) (* S364_RS_AX_RH_CLAMP_후진1 *)
    S364_RS_AX_RH_CLAMP_후진2 : BOOL; (* AT %MW87150.6 *) (* S364_RS_AX_RH_CLAMP_후진2 *)
    S364_RS_AX_RH_LATCH_전진 : BOOL; (* AT %MW87150.0 *) (* S364_RS_AX_RH_LATCH_전진 *)
    S364_RS_AX_RH_LATCH_후진1 : BOOL; (* AT %MW87150.1 *) (* S364_RS_AX_RH_LATCH_후진1 *)
    S364_RS_AX_RH_LATCH_후진2 : BOOL; (* AT %MW87150.2 *) (* S364_RS_AX_RH_LATCH_후진2 *)
    S364_RS_AX_RH_SLD_CLP_전진 : BOOL; (* AT %MW87151.0 *) (* S364_RS_AX_RH_SLD_CLP_전진 *)
    S364_RS_AX_RH_SLD_CLP_후진1 : BOOL; (* AT %MW87151.1 *) (* S364_RS_AX_RH_SLD_CLP_후진1 *)
    S364_RS_AX_RH_SLD_CLP_후진2 : BOOL; (* AT %MW87151.2 *) (* S364_RS_AX_RH_SLD_CLP_후진2 *)
    S364_RS_AX_RH_SLD_CLP_후진3 : BOOL; (* AT %MW87151.3 *) (* S364_RS_AX_RH_SLD_CLP_후진3 *)
    S364_RS_AX_RH_SLD_CLP_후진4 : BOOL; (* AT %MW87151.4 *) (* S364_RS_AX_RH_SLD_CLP_후진4 *)
    S364_RS_AX_RH_SLD_LAT_전진 : BOOL; (* AT %MW87150.8 *) (* S364_RS_AX_RH_SLD_LAT_전진 *)
    S364_RS_AX_RH_SLD_LAT_후진1 : BOOL; (* AT %MW87150.9 *) (* S364_RS_AX_RH_SLD_LAT_후진1 *)
    S364_RS_AX_RH_SLD_LAT_후진2 : BOOL; (* AT %MW87150.10 *) (* S364_RS_AX_RH_SLD_LAT_후진2 *)
    S364_RS_AX_RH_SLD_LAT_후진3 : BOOL; (* AT %MW87150.11 *) (* S364_RS_AX_RH_SLD_LAT_후진3 *)
    S364_RS_AX_RH_SLD_LAT_후진4 : BOOL; (* AT %MW87150.12 *) (* S364_RS_AX_RH_SLD_LAT_후진4 *)
    S364_RS_AX_RH_SLIDE_전진 : BOOL; (* AT %MW87151.10 *) (* S364_RS_AX_RH_SLIDE_전진 *)
    S364_RS_AX_RH_SLIDE_후진 : BOOL; (* AT %MW87151.11 *) (* S364_RS_AX_RH_SLIDE_후진 *)
    S364_SOL_AX_CLAMP_전진 : BOOL; (* AT %MW97153.2 *) (* S364_SOL_AX_CLAMP_전진 *)
    S364_SOL_AX_CLAMP_후진 : BOOL; (* AT %MW97153.3 *) (* S364_SOL_AX_CLAMP_후진 *)
    S364_SOL_AX_LATCH_전진 : BOOL; (* AT %MW97153.0 *) (* S364_SOL_AX_LATCH_전진 *)
    S364_SOL_AX_LATCH_후진 : BOOL; (* AT %MW97153.1 *) (* S364_SOL_AX_LATCH_후진 *)
    S364_SOL_AX_LH_BRAKE_ON : BOOL; (* AT %MW97154.2 *) (* S364_SOL_AX_LH_BRAKE_ON *)
    S364_SOL_AX_LH_SLD_CLP_전진 : BOOL; (* AT %MW97153.6 *) (* S364_SOL_AX_LH_SLD_CLP_전진 *)
    S364_SOL_AX_LH_SLD_CLP_후진 : BOOL; (* AT %MW97153.7 *) (* S364_SOL_AX_LH_SLD_CLP_후진 *)
    S364_SOL_AX_LH_SLD_LAT_전진 : BOOL; (* AT %MW97153.4 *) (* S364_SOL_AX_LH_SLD_LAT_전진 *)
    S364_SOL_AX_LH_SLD_LAT_후진 : BOOL; (* AT %MW97153.5 *) (* S364_SOL_AX_LH_SLD_LAT_후진 *)
    S364_SOL_AX_LH_SLIDE_전진 : BOOL; (* AT %MW97154.0 *) (* S364_SOL_AX_LH_SLIDE_전진 *)
    S364_SOL_AX_LH_SLIDE_후진 : BOOL; (* AT %MW97154.1 *) (* S364_SOL_AX_LH_SLIDE_후진 *)
    S364_SOL_AX_RH_BRAKE_ON : BOOL; (* AT %MW97154.6 *) (* S364_SOL_AX_RH_BRAKE_ON *)
    S364_SOL_AX_RH_SLD_CLP_전진 : BOOL; (* AT %MW97153.10 *) (* S364_SOL_AX_RH_SLD_CLP_전진 *)
    S364_SOL_AX_RH_SLD_CLP_후진 : BOOL; (* AT %MW97153.11 *) (* S364_SOL_AX_RH_SLD_CLP_후진 *)
    S364_SOL_AX_RH_SLD_LAT_전진 : BOOL; (* AT %MW97153.8 *) (* S364_SOL_AX_RH_SLD_LAT_전진 *)
    S364_SOL_AX_RH_SLD_LAT_후진 : BOOL; (* AT %MW97153.9 *) (* S364_SOL_AX_RH_SLD_LAT_후진 *)
    S364_SOL_AX_RH_SLIDE_전진 : BOOL; (* AT %MW97154.4 *) (* S364_SOL_AX_RH_SLIDE_전진 *)
    S364_SOL_AX_RH_SLIDE_후진 : BOOL; (* AT %MW97154.5 *) (* S364_SOL_AX_RH_SLIDE_후진 *)
END_VAR
VAR
    S364_AX_CLAMP : ACT_6_CYL;
    S364_AX_LATCH : ACT_6_CYL;
    S364_AX_LH_SLIDE : ACT_6_CYL;
    S364_AX_LH_SLIDE_LATCH : ACT_6_CYL;
    S364_AX_RH_SLIDE : ACT_6_CYL;
    S364_AX_RH_SLIDE_CLAMP : ACT_6_CYL;
    S364_AX_RH_SLIDE_LATCH : ACT_6_CYL;
    S365_AX_LH_SLIDE_CLAMP : ACT_6_CYL;
END_VAR

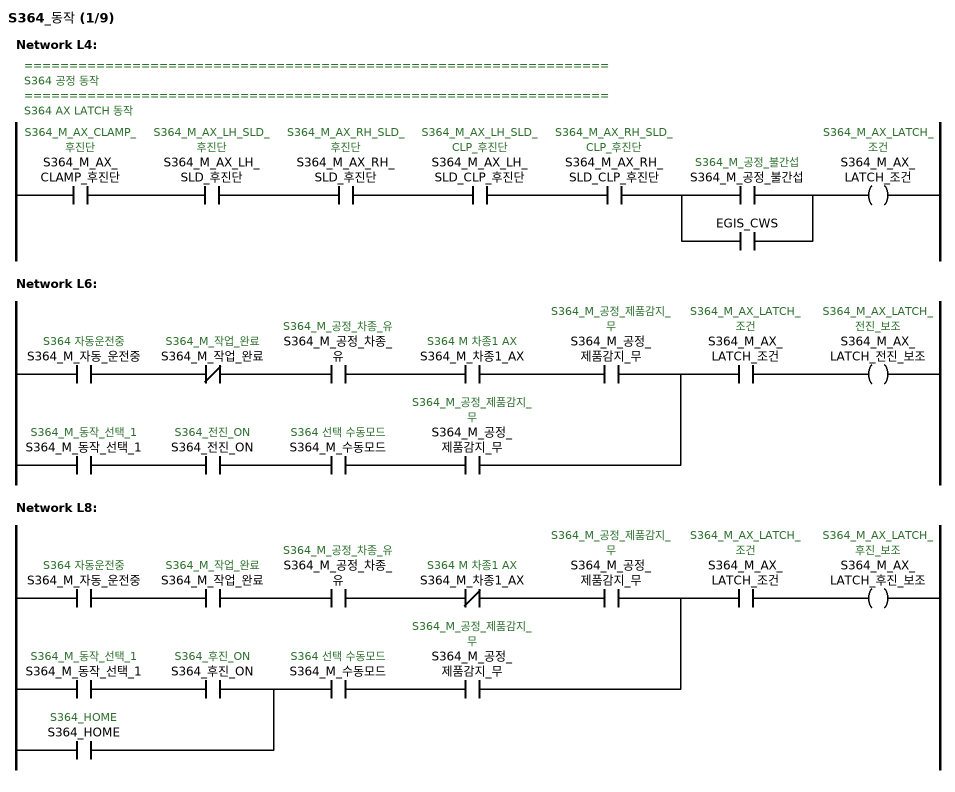
(* ================================================================= *)
(* S364 공정 동작 *)
(* ================================================================= *)
(* S364 AX LATCH 동작 *)
(* Rung L4 *)
S364_M_AX_LATCH_조건 := S364_M_AX_CLAMP_후진단 AND S364_M_AX_LH_SLD_후진단 AND S364_M_AX_RH_SLD_후진단 AND S364_M_AX_LH_SLD_CLP_후진단 AND S364_M_AX_RH_SLD_CLP_후진단 AND (S364_M_공정_불간섭 OR EGIS_CWS);
(* Rung L6 *)
S364_M_AX_LATCH_전진_보조 := ((S364_M_자동_운전중 AND NOT S364_M_작업_완료 AND S364_M_공정_차종_유 AND S364_M_차종1_AX AND S364_M_공정_제품감지_무) OR (S364_M_동작_선택_1 AND S364_전진_ON AND S364_M_수동모드 AND S364_M_공정_제품감지_무)) AND S364_M_AX_LATCH_조건;
(* Rung L8 *)
S364_M_AX_LATCH_후진_보조 := ((S364_M_자동_운전중 AND S364_M_작업_완료 AND S364_M_공정_차종_유 AND NOT S364_M_차종1_AX AND S364_M_공정_제품감지_무) OR (((S364_M_동작_선택_1 AND S364_후진_ON) OR S364_HOME) AND S364_M_수동모드 AND S364_M_공정_제품감지_무)) AND S364_M_AX_LATCH_조건;

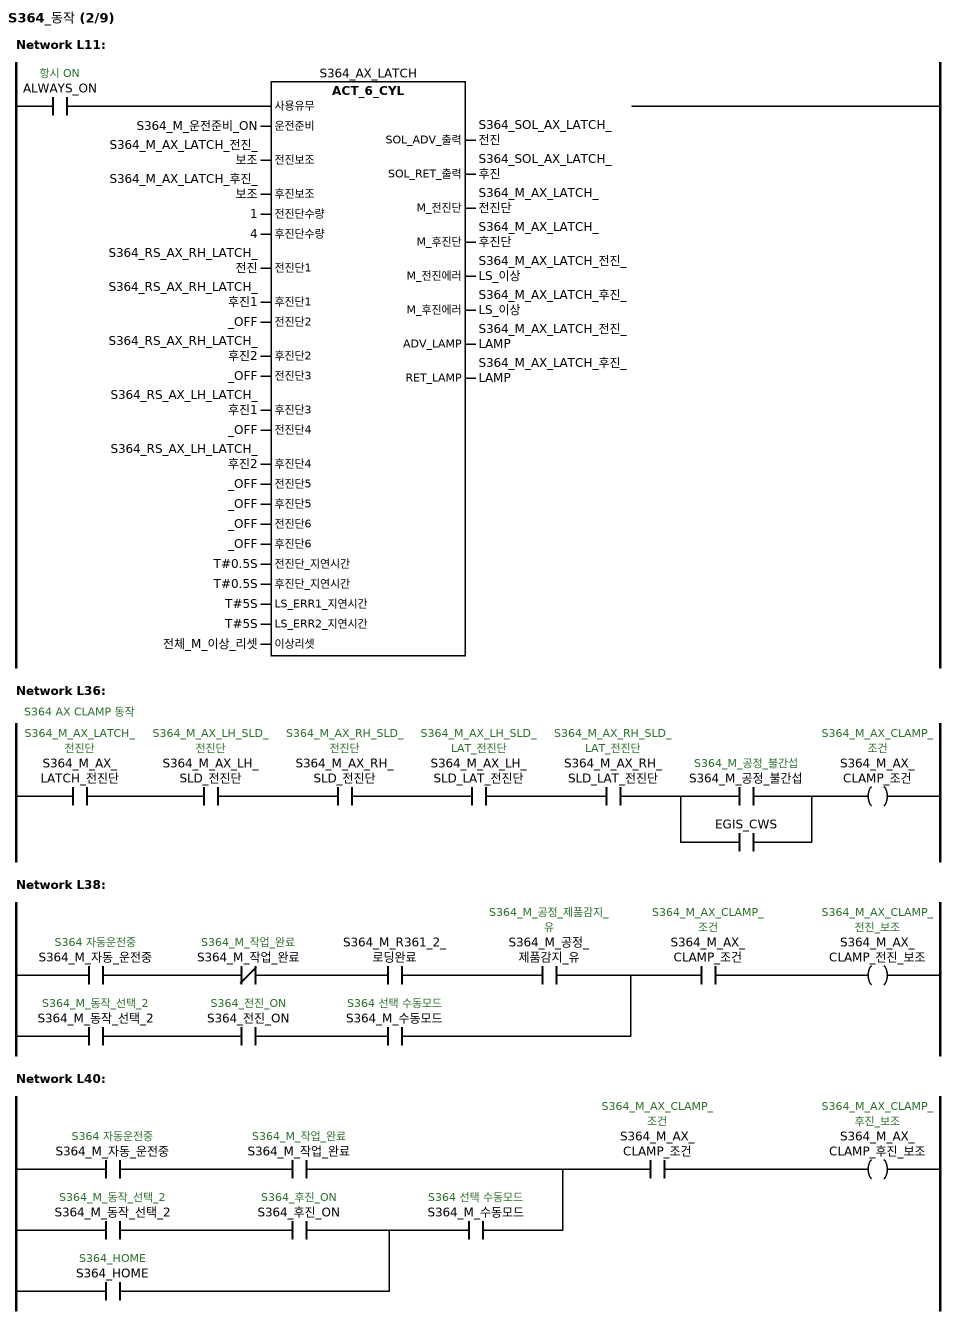
(* Rung L11 *)
S364_AX_LATCH(사용유무 := ALWAYS_ON, 운전준비 := S364_M_운전준비_ON, 전진보조 := S364_M_AX_LATCH_전진_보조, 후진보조 := S364_M_AX_LATCH_후진_보조, 전진단수량 := 1, 후진단수량 := 4, 전진단1 := S364_RS_AX_RH_LATCH_전진, 후진단1 := S364_RS_AX_RH_LATCH_후진1, 전진단2 := _OFF, 후진단2 := S364_RS_AX_RH_LATCH_후진2, 전진단3 := _OFF, 후진단3 := S364_RS_AX_LH_LATCH_후진1, 전진단4 := _OFF, 후진단4 := S364_RS_AX_LH_LATCH_후진2, 전진단5 := _OFF, 후진단5 := _OFF, 전진단6 := _OFF, 후진단6 := _OFF, 전진단_지연시간 := T#0.5S, 후진단_지연시간 := T#0.5S, LS_ERR1_지연시간 := T#5S, LS_ERR2_지연시간 := T#5S, 이상리셋 := 전체_M_이상_리셋, SOL_ADV_출력 => S364_SOL_AX_LATCH_전진, SOL_RET_출력 => S364_SOL_AX_LATCH_후진, M_전진단 => S364_M_AX_LATCH_전진단, M_후진단 => S364_M_AX_LATCH_후진단, M_전진에러 => S364_M_AX_LATCH_전진_LS_이상, M_후진에러 => S364_M_AX_LATCH_후진_LS_이상, ADV_LAMP => S364_M_AX_LATCH_전진_LAMP, RET_LAMP => S364_M_AX_LATCH_후진_LAMP);
(* S364 AX CLAMP 동작 *)
(* Rung L36 *)
S364_M_AX_CLAMP_조건 := S364_M_AX_LATCH_전진단 AND S364_M_AX_LH_SLD_전진단 AND S364_M_AX_RH_SLD_전진단 AND S364_M_AX_LH_SLD_LAT_전진단 AND S364_M_AX_RH_SLD_LAT_전진단 AND (S364_M_공정_불간섭 OR EGIS_CWS);
(* Rung L38 *)
S364_M_AX_CLAMP_전진_보조 := ((S364_M_자동_운전중 AND NOT S364_M_작업_완료 AND S364_M_R361_2_로딩완료 AND S364_M_공정_제품감지_유) OR (S364_M_동작_선택_2 AND S364_전진_ON AND S364_M_수동모드)) AND S364_M_AX_CLAMP_조건;
(* Rung L40 *)
S364_M_AX_CLAMP_후진_보조 := ((S364_M_자동_운전중 AND S364_M_작업_완료) OR (((S364_M_동작_선택_2 AND S364_후진_ON) OR S364_HOME) AND S364_M_수동모드)) AND S364_M_AX_CLAMP_조건;

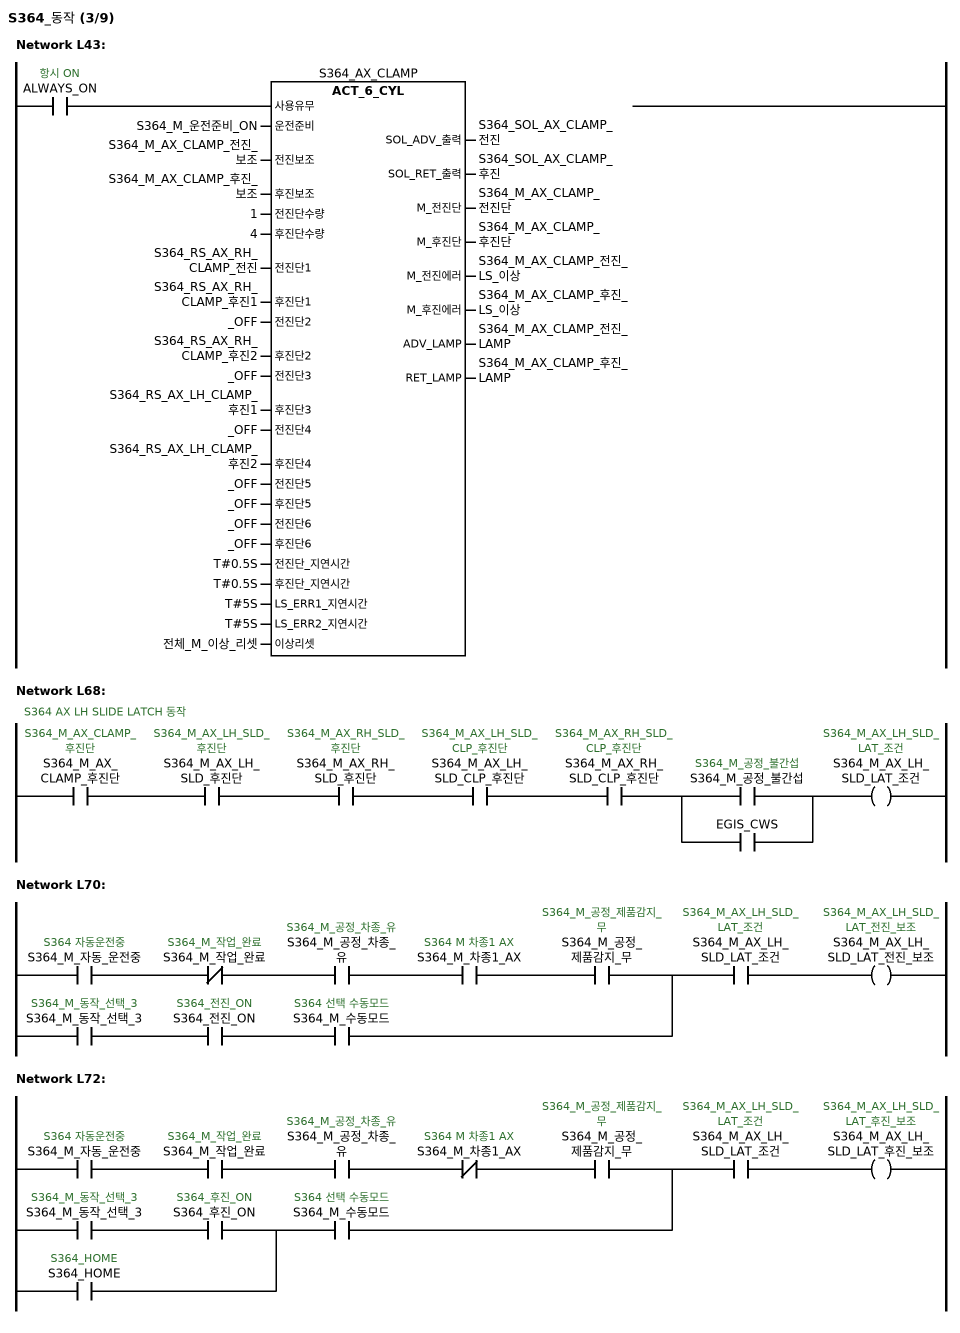
(* Rung L43 *)
S364_AX_CLAMP(사용유무 := ALWAYS_ON, 운전준비 := S364_M_운전준비_ON, 전진보조 := S364_M_AX_CLAMP_전진_보조, 후진보조 := S364_M_AX_CLAMP_후진_보조, 전진단수량 := 1, 후진단수량 := 4, 전진단1 := S364_RS_AX_RH_CLAMP_전진, 후진단1 := S364_RS_AX_RH_CLAMP_후진1, 전진단2 := _OFF, 후진단2 := S364_RS_AX_RH_CLAMP_후진2, 전진단3 := _OFF, 후진단3 := S364_RS_AX_LH_CLAMP_후진1, 전진단4 := _OFF, 후진단4 := S364_RS_AX_LH_CLAMP_후진2, 전진단5 := _OFF, 후진단5 := _OFF, 전진단6 := _OFF, 후진단6 := _OFF, 전진단_지연시간 := T#0.5S, 후진단_지연시간 := T#0.5S, LS_ERR1_지연시간 := T#5S, LS_ERR2_지연시간 := T#5S, 이상리셋 := 전체_M_이상_리셋, SOL_ADV_출력 => S364_SOL_AX_CLAMP_전진, SOL_RET_출력 => S364_SOL_AX_CLAMP_후진, M_전진단 => S364_M_AX_CLAMP_전진단, M_후진단 => S364_M_AX_CLAMP_후진단, M_전진에러 => S364_M_AX_CLAMP_전진_LS_이상, M_후진에러 => S364_M_AX_CLAMP_후진_LS_이상, ADV_LAMP => S364_M_AX_CLAMP_전진_LAMP, RET_LAMP => S364_M_AX_CLAMP_후진_LAMP);
(* S364 AX LH SLIDE LATCH 동작 *)
(* Rung L68 *)
S364_M_AX_LH_SLD_LAT_조건 := S364_M_AX_CLAMP_후진단 AND S364_M_AX_LH_SLD_후진단 AND S364_M_AX_RH_SLD_후진단 AND S364_M_AX_LH_SLD_CLP_후진단 AND S364_M_AX_RH_SLD_CLP_후진단 AND (S364_M_공정_불간섭 OR EGIS_CWS);
(* Rung L70 *)
S364_M_AX_LH_SLD_LAT_전진_보조 := ((S364_M_자동_운전중 AND NOT S364_M_작업_완료 AND S364_M_공정_차종_유 AND S364_M_차종1_AX AND S364_M_공정_제품감지_무) OR (S364_M_동작_선택_3 AND S364_전진_ON AND S364_M_수동모드)) AND S364_M_AX_LH_SLD_LAT_조건;
(* Rung L72 *)
S364_M_AX_LH_SLD_LAT_후진_보조 := ((S364_M_자동_운전중 AND S364_M_작업_완료 AND S364_M_공정_차종_유 AND NOT S364_M_차종1_AX AND S364_M_공정_제품감지_무) OR (((S364_M_동작_선택_3 AND S364_후진_ON) OR S364_HOME) AND S364_M_수동모드)) AND S364_M_AX_LH_SLD_LAT_조건;

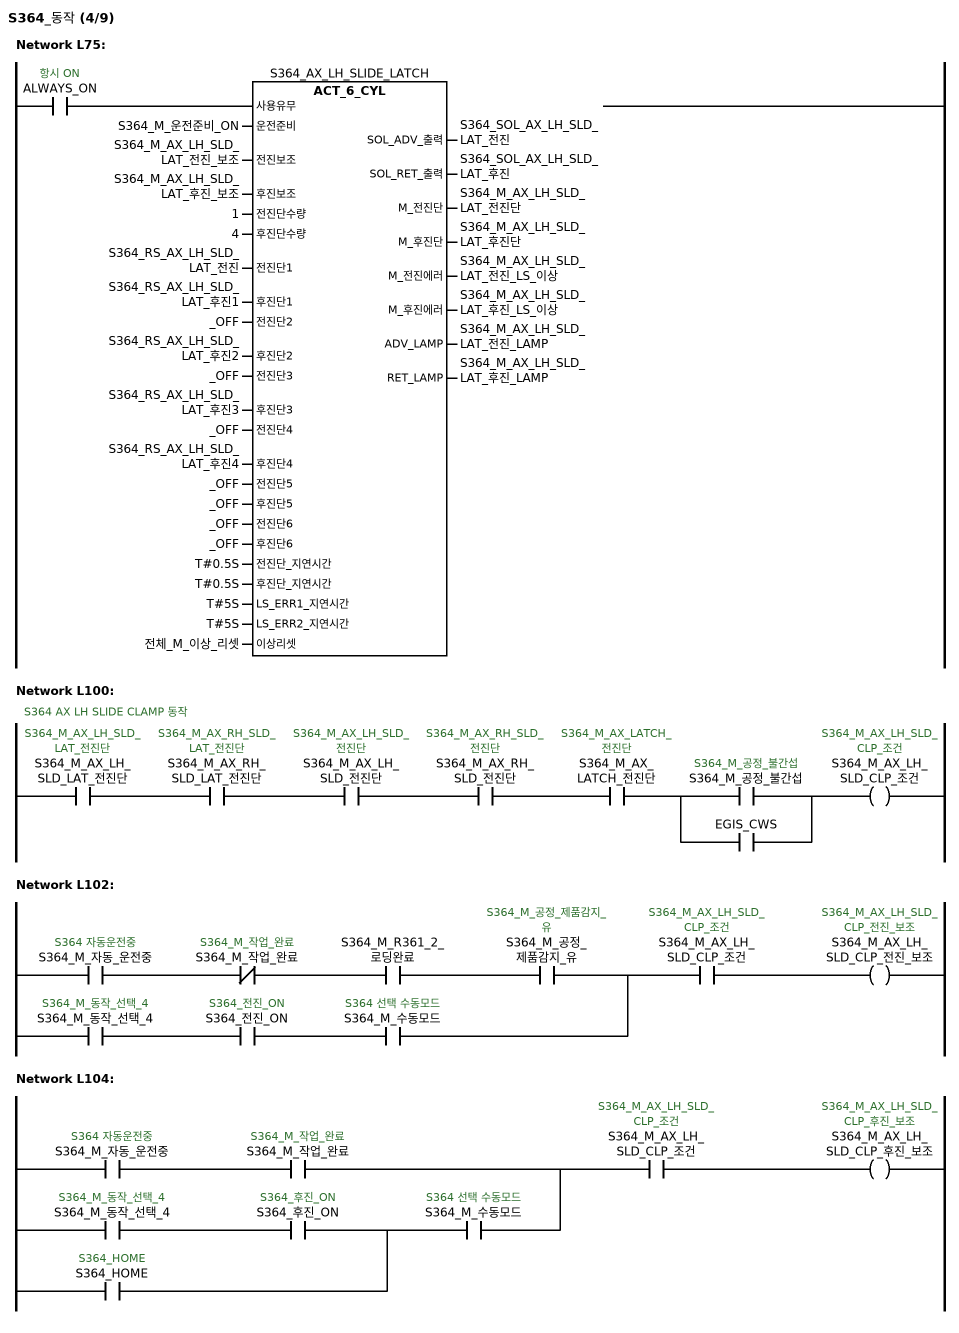
(* Rung L75 *)
S364_AX_LH_SLIDE_LATCH(사용유무 := ALWAYS_ON, 운전준비 := S364_M_운전준비_ON, 전진보조 := S364_M_AX_LH_SLD_LAT_전진_보조, 후진보조 := S364_M_AX_LH_SLD_LAT_후진_보조, 전진단수량 := 1, 후진단수량 := 4, 전진단1 := S364_RS_AX_LH_SLD_LAT_전진, 후진단1 := S364_RS_AX_LH_SLD_LAT_후진1, 전진단2 := _OFF, 후진단2 := S364_RS_AX_LH_SLD_LAT_후진2, 전진단3 := _OFF, 후진단3 := S364_RS_AX_LH_SLD_LAT_후진3, 전진단4 := _OFF, 후진단4 := S364_RS_AX_LH_SLD_LAT_후진4, 전진단5 := _OFF, 후진단5 := _OFF, 전진단6 := _OFF, 후진단6 := _OFF, 전진단_지연시간 := T#0.5S, 후진단_지연시간 := T#0.5S, LS_ERR1_지연시간 := T#5S, LS_ERR2_지연시간 := T#5S, 이상리셋 := 전체_M_이상_리셋, SOL_ADV_출력 => S364_SOL_AX_LH_SLD_LAT_전진, SOL_RET_출력 => S364_SOL_AX_LH_SLD_LAT_후진, M_전진단 => S364_M_AX_LH_SLD_LAT_전진단, M_후진단 => S364_M_AX_LH_SLD_LAT_후진단, M_전진에러 => S364_M_AX_LH_SLD_LAT_전진_LS_이상, M_후진에러 => S364_M_AX_LH_SLD_LAT_후진_LS_이상, ADV_LAMP => S364_M_AX_LH_SLD_LAT_전진_LAMP, RET_LAMP => S364_M_AX_LH_SLD_LAT_후진_LAMP);
(* S364 AX LH SLIDE CLAMP 동작 *)
(* Rung L100 *)
S364_M_AX_LH_SLD_CLP_조건 := S364_M_AX_LH_SLD_LAT_전진단 AND S364_M_AX_RH_SLD_LAT_전진단 AND S364_M_AX_LH_SLD_전진단 AND S364_M_AX_RH_SLD_전진단 AND S364_M_AX_LATCH_전진단 AND (S364_M_공정_불간섭 OR EGIS_CWS);
(* Rung L102 *)
S364_M_AX_LH_SLD_CLP_전진_보조 := ((S364_M_자동_운전중 AND NOT S364_M_작업_완료 AND S364_M_R361_2_로딩완료 AND S364_M_공정_제품감지_유) OR (S364_M_동작_선택_4 AND S364_전진_ON AND S364_M_수동모드)) AND S364_M_AX_LH_SLD_CLP_조건;
(* Rung L104 *)
S364_M_AX_LH_SLD_CLP_후진_보조 := ((S364_M_자동_운전중 AND S364_M_작업_완료) OR (((S364_M_동작_선택_4 AND S364_후진_ON) OR S364_HOME) AND S364_M_수동모드)) AND S364_M_AX_LH_SLD_CLP_조건;

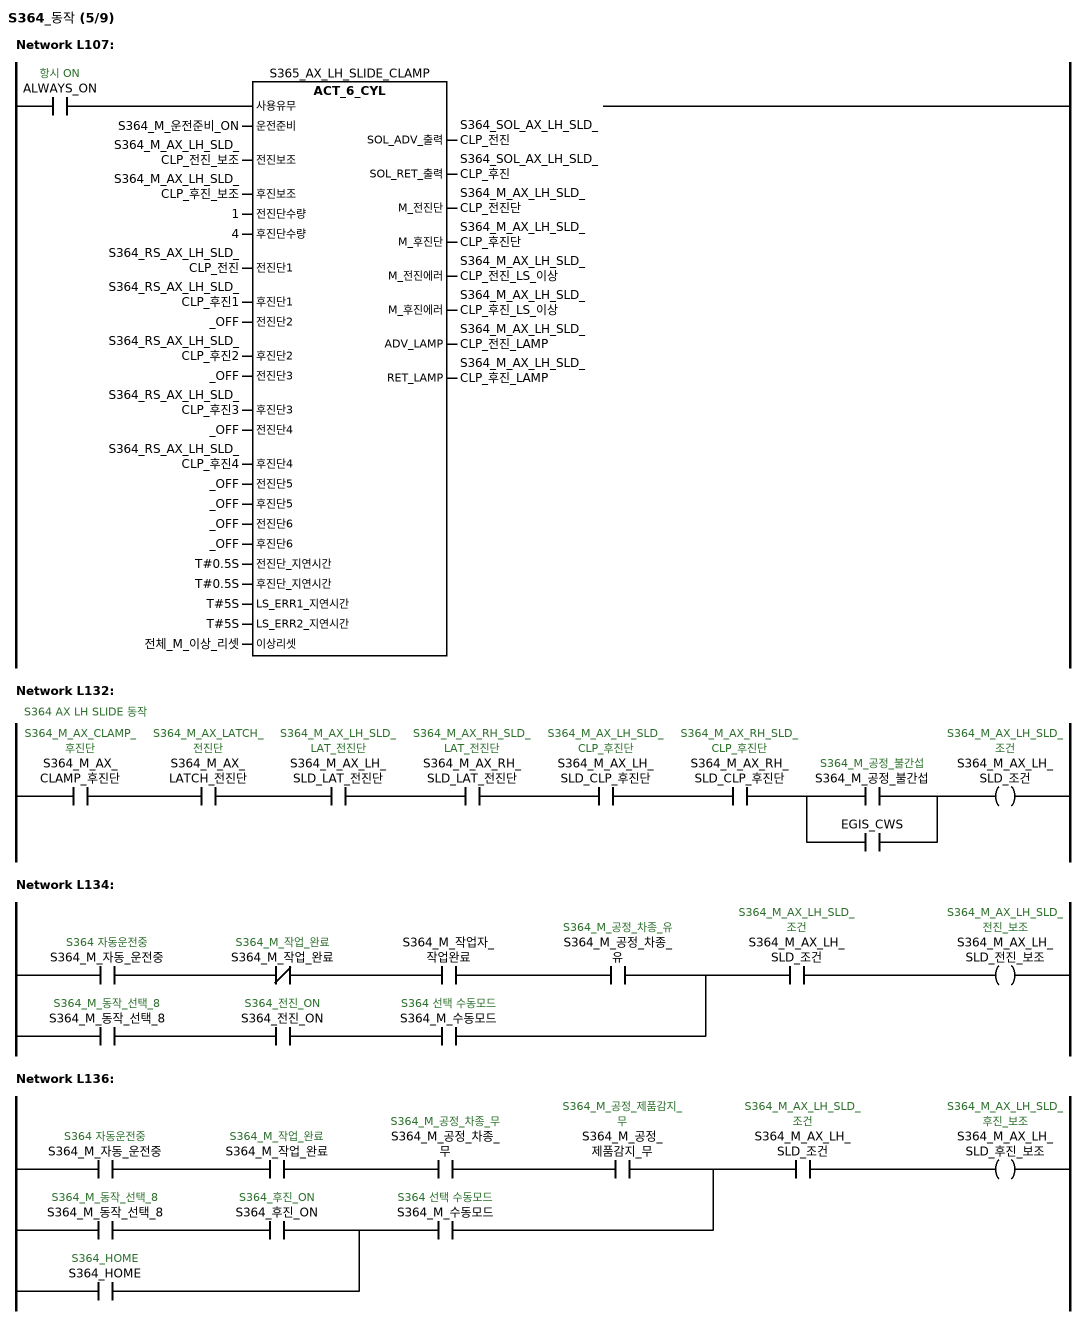
(* Rung L107 *)
S365_AX_LH_SLIDE_CLAMP(사용유무 := ALWAYS_ON, 운전준비 := S364_M_운전준비_ON, 전진보조 := S364_M_AX_LH_SLD_CLP_전진_보조, 후진보조 := S364_M_AX_LH_SLD_CLP_후진_보조, 전진단수량 := 1, 후진단수량 := 4, 전진단1 := S364_RS_AX_LH_SLD_CLP_전진, 후진단1 := S364_RS_AX_LH_SLD_CLP_후진1, 전진단2 := _OFF, 후진단2 := S364_RS_AX_LH_SLD_CLP_후진2, 전진단3 := _OFF, 후진단3 := S364_RS_AX_LH_SLD_CLP_후진3, 전진단4 := _OFF, 후진단4 := S364_RS_AX_LH_SLD_CLP_후진4, 전진단5 := _OFF, 후진단5 := _OFF, 전진단6 := _OFF, 후진단6 := _OFF, 전진단_지연시간 := T#0.5S, 후진단_지연시간 := T#0.5S, LS_ERR1_지연시간 := T#5S, LS_ERR2_지연시간 := T#5S, 이상리셋 := 전체_M_이상_리셋, SOL_ADV_출력 => S364_SOL_AX_LH_SLD_CLP_전진, SOL_RET_출력 => S364_SOL_AX_LH_SLD_CLP_후진, M_전진단 => S364_M_AX_LH_SLD_CLP_전진단, M_후진단 => S364_M_AX_LH_SLD_CLP_후진단, M_전진에러 => S364_M_AX_LH_SLD_CLP_전진_LS_이상, M_후진에러 => S364_M_AX_LH_SLD_CLP_후진_LS_이상, ADV_LAMP => S364_M_AX_LH_SLD_CLP_전진_LAMP, RET_LAMP => S364_M_AX_LH_SLD_CLP_후진_LAMP);
(* S364 AX LH SLIDE 동작 *)
(* Rung L132 *)
S364_M_AX_LH_SLD_조건 := S364_M_AX_CLAMP_후진단 AND S364_M_AX_LATCH_전진단 AND S364_M_AX_LH_SLD_LAT_전진단 AND S364_M_AX_RH_SLD_LAT_전진단 AND S364_M_AX_LH_SLD_CLP_후진단 AND S364_M_AX_RH_SLD_CLP_후진단 AND (S364_M_공정_불간섭 OR EGIS_CWS);
(* Rung L134 *)
S364_M_AX_LH_SLD_전진_보조 := ((S364_M_자동_운전중 AND NOT S364_M_작업_완료 AND S364_M_작업자_작업완료 AND S364_M_공정_차종_유) OR (S364_M_동작_선택_8 AND S364_전진_ON AND S364_M_수동모드)) AND S364_M_AX_LH_SLD_조건;
(* Rung L136 *)
S364_M_AX_LH_SLD_후진_보조 := ((S364_M_자동_운전중 AND S364_M_작업_완료 AND S364_M_공정_차종_무 AND S364_M_공정_제품감지_무) OR (((S364_M_동작_선택_8 AND S364_후진_ON) OR S364_HOME) AND S364_M_수동모드)) AND S364_M_AX_LH_SLD_조건;

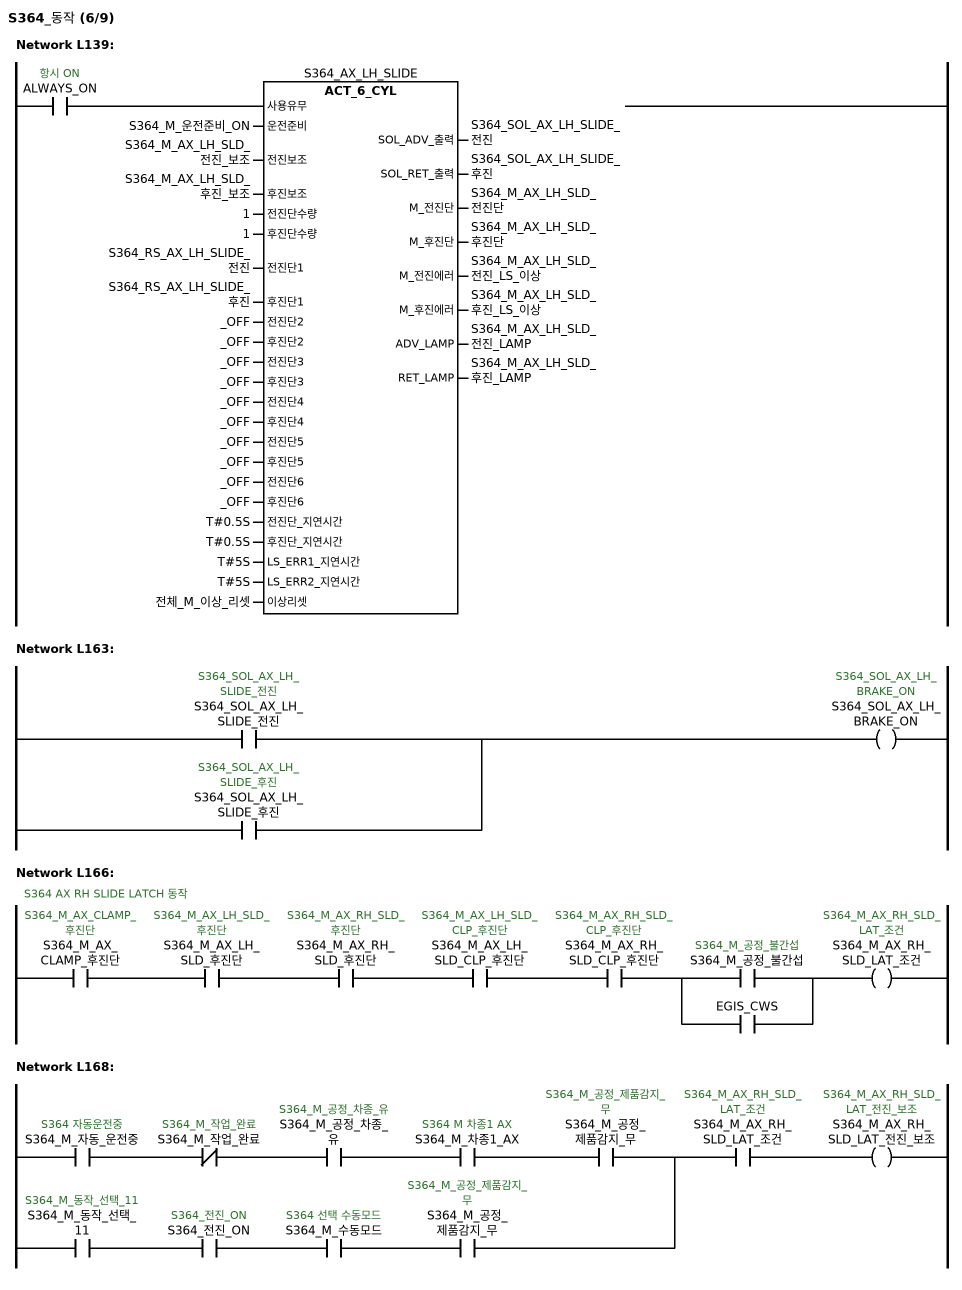
(* Rung L139 *)
S364_AX_LH_SLIDE(사용유무 := ALWAYS_ON, 운전준비 := S364_M_운전준비_ON, 전진보조 := S364_M_AX_LH_SLD_전진_보조, 후진보조 := S364_M_AX_LH_SLD_후진_보조, 전진단수량 := 1, 후진단수량 := 1, 전진단1 := S364_RS_AX_LH_SLIDE_전진, 후진단1 := S364_RS_AX_LH_SLIDE_후진, 전진단2 := _OFF, 후진단2 := _OFF, 전진단3 := _OFF, 후진단3 := _OFF, 전진단4 := _OFF, 후진단4 := _OFF, 전진단5 := _OFF, 후진단5 := _OFF, 전진단6 := _OFF, 후진단6 := _OFF, 전진단_지연시간 := T#0.5S, 후진단_지연시간 := T#0.5S, LS_ERR1_지연시간 := T#5S, LS_ERR2_지연시간 := T#5S, 이상리셋 := 전체_M_이상_리셋, SOL_ADV_출력 => S364_SOL_AX_LH_SLIDE_전진, SOL_RET_출력 => S364_SOL_AX_LH_SLIDE_후진, M_전진단 => S364_M_AX_LH_SLD_전진단, M_후진단 => S364_M_AX_LH_SLD_후진단, M_전진에러 => S364_M_AX_LH_SLD_전진_LS_이상, M_후진에러 => S364_M_AX_LH_SLD_후진_LS_이상, ADV_LAMP => S364_M_AX_LH_SLD_전진_LAMP, RET_LAMP => S364_M_AX_LH_SLD_후진_LAMP);
(* Rung L163 *)
S364_SOL_AX_LH_BRAKE_ON := S364_SOL_AX_LH_SLIDE_전진 OR S364_SOL_AX_LH_SLIDE_후진;
(* S364 AX RH SLIDE LATCH 동작 *)
(* Rung L166 *)
S364_M_AX_RH_SLD_LAT_조건 := S364_M_AX_CLAMP_후진단 AND S364_M_AX_LH_SLD_후진단 AND S364_M_AX_RH_SLD_후진단 AND S364_M_AX_LH_SLD_CLP_후진단 AND S364_M_AX_RH_SLD_CLP_후진단 AND (S364_M_공정_불간섭 OR EGIS_CWS);
(* Rung L168 *)
S364_M_AX_RH_SLD_LAT_전진_보조 := ((S364_M_자동_운전중 AND NOT S364_M_작업_완료 AND S364_M_공정_차종_유 AND S364_M_차종1_AX AND S364_M_공정_제품감지_무) OR (S364_M_동작_선택_11 AND S364_전진_ON AND S364_M_수동모드 AND S364_M_공정_제품감지_무)) AND S364_M_AX_RH_SLD_LAT_조건;

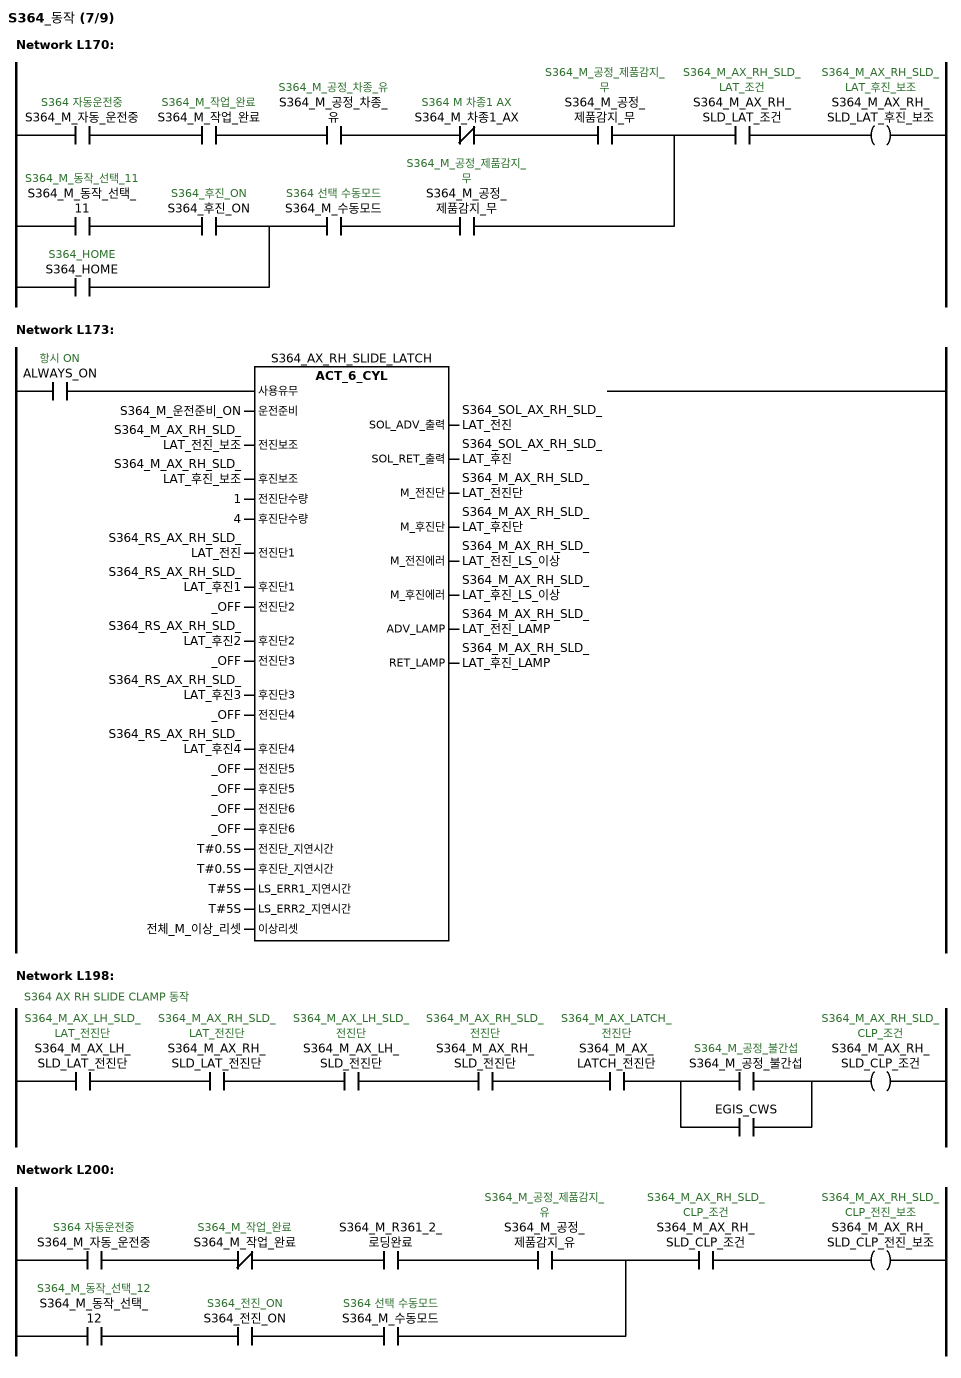
(* Rung L170 *)
S364_M_AX_RH_SLD_LAT_후진_보조 := ((S364_M_자동_운전중 AND S364_M_작업_완료 AND S364_M_공정_차종_유 AND NOT S364_M_차종1_AX AND S364_M_공정_제품감지_무) OR (((S364_M_동작_선택_11 AND S364_후진_ON) OR S364_HOME) AND S364_M_수동모드 AND S364_M_공정_제품감지_무)) AND S364_M_AX_RH_SLD_LAT_조건;
(* Rung L173 *)
S364_AX_RH_SLIDE_LATCH(사용유무 := ALWAYS_ON, 운전준비 := S364_M_운전준비_ON, 전진보조 := S364_M_AX_RH_SLD_LAT_전진_보조, 후진보조 := S364_M_AX_RH_SLD_LAT_후진_보조, 전진단수량 := 1, 후진단수량 := 4, 전진단1 := S364_RS_AX_RH_SLD_LAT_전진, 후진단1 := S364_RS_AX_RH_SLD_LAT_후진1, 전진단2 := _OFF, 후진단2 := S364_RS_AX_RH_SLD_LAT_후진2, 전진단3 := _OFF, 후진단3 := S364_RS_AX_RH_SLD_LAT_후진3, 전진단4 := _OFF, 후진단4 := S364_RS_AX_RH_SLD_LAT_후진4, 전진단5 := _OFF, 후진단5 := _OFF, 전진단6 := _OFF, 후진단6 := _OFF, 전진단_지연시간 := T#0.5S, 후진단_지연시간 := T#0.5S, LS_ERR1_지연시간 := T#5S, LS_ERR2_지연시간 := T#5S, 이상리셋 := 전체_M_이상_리셋, SOL_ADV_출력 => S364_SOL_AX_RH_SLD_LAT_전진, SOL_RET_출력 => S364_SOL_AX_RH_SLD_LAT_후진, M_전진단 => S364_M_AX_RH_SLD_LAT_전진단, M_후진단 => S364_M_AX_RH_SLD_LAT_후진단, M_전진에러 => S364_M_AX_RH_SLD_LAT_전진_LS_이상, M_후진에러 => S364_M_AX_RH_SLD_LAT_후진_LS_이상, ADV_LAMP => S364_M_AX_RH_SLD_LAT_전진_LAMP, RET_LAMP => S364_M_AX_RH_SLD_LAT_후진_LAMP);
(* S364 AX RH SLIDE CLAMP 동작 *)
(* Rung L198 *)
S364_M_AX_RH_SLD_CLP_조건 := S364_M_AX_LH_SLD_LAT_전진단 AND S364_M_AX_RH_SLD_LAT_전진단 AND S364_M_AX_LH_SLD_전진단 AND S364_M_AX_RH_SLD_전진단 AND S364_M_AX_LATCH_전진단 AND (S364_M_공정_불간섭 OR EGIS_CWS);
(* Rung L200 *)
S364_M_AX_RH_SLD_CLP_전진_보조 := ((S364_M_자동_운전중 AND NOT S364_M_작업_완료 AND S364_M_R361_2_로딩완료 AND S364_M_공정_제품감지_유) OR (S364_M_동작_선택_12 AND S364_전진_ON AND S364_M_수동모드)) AND S364_M_AX_RH_SLD_CLP_조건;

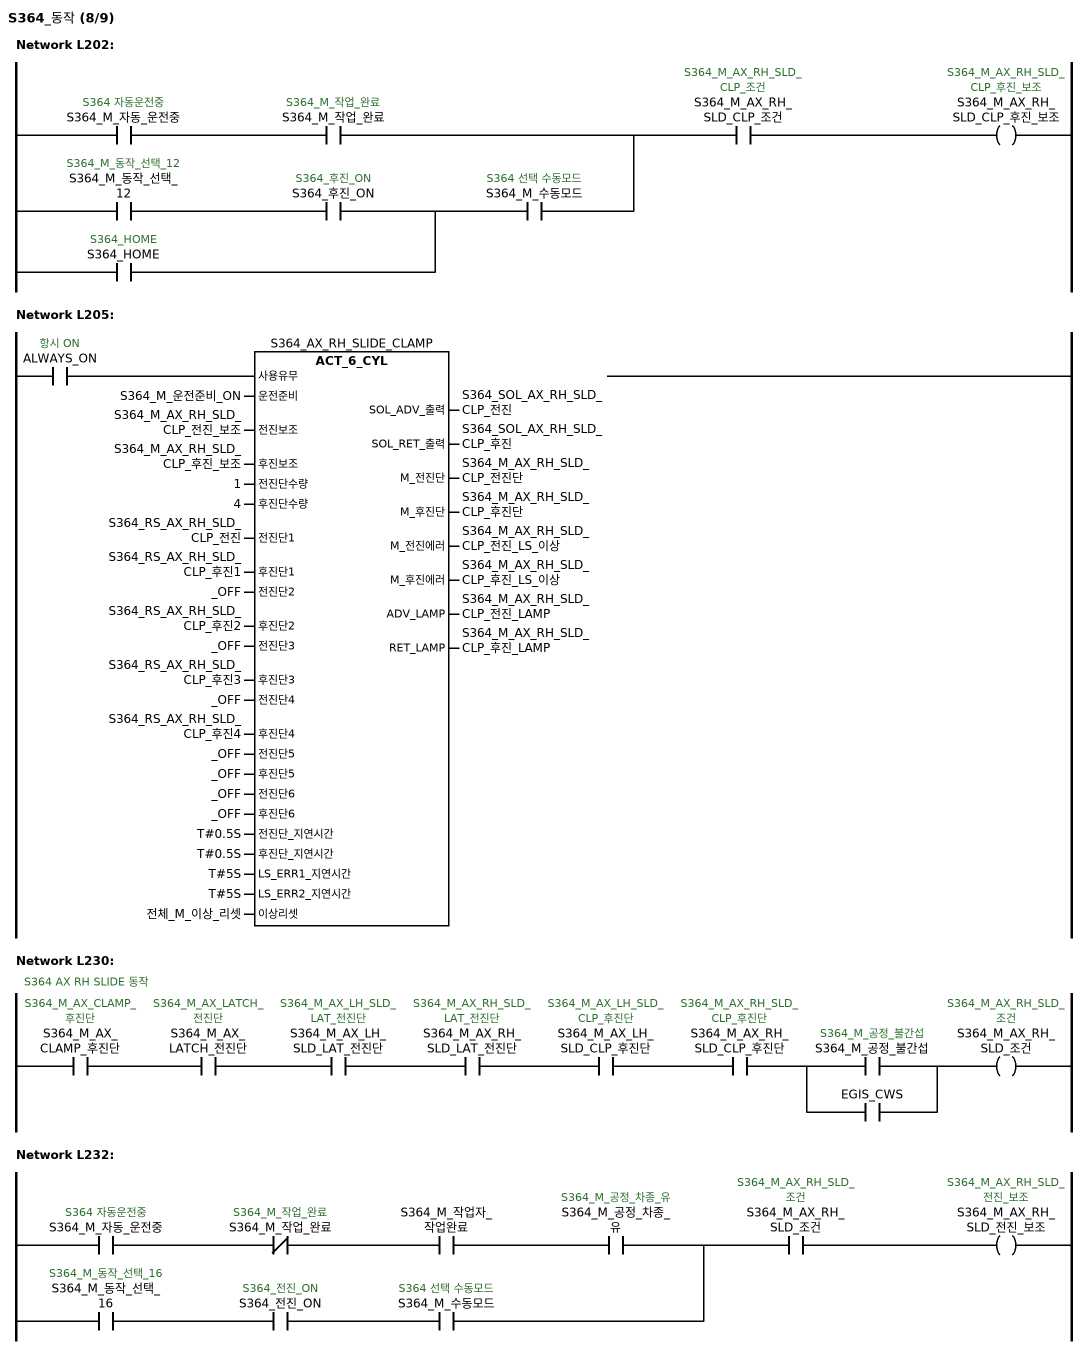
(* Rung L202 *)
S364_M_AX_RH_SLD_CLP_후진_보조 := ((S364_M_자동_운전중 AND S364_M_작업_완료) OR (((S364_M_동작_선택_12 AND S364_후진_ON) OR S364_HOME) AND S364_M_수동모드)) AND S364_M_AX_RH_SLD_CLP_조건;
(* Rung L205 *)
S364_AX_RH_SLIDE_CLAMP(사용유무 := ALWAYS_ON, 운전준비 := S364_M_운전준비_ON, 전진보조 := S364_M_AX_RH_SLD_CLP_전진_보조, 후진보조 := S364_M_AX_RH_SLD_CLP_후진_보조, 전진단수량 := 1, 후진단수량 := 4, 전진단1 := S364_RS_AX_RH_SLD_CLP_전진, 후진단1 := S364_RS_AX_RH_SLD_CLP_후진1, 전진단2 := _OFF, 후진단2 := S364_RS_AX_RH_SLD_CLP_후진2, 전진단3 := _OFF, 후진단3 := S364_RS_AX_RH_SLD_CLP_후진3, 전진단4 := _OFF, 후진단4 := S364_RS_AX_RH_SLD_CLP_후진4, 전진단5 := _OFF, 후진단5 := _OFF, 전진단6 := _OFF, 후진단6 := _OFF, 전진단_지연시간 := T#0.5S, 후진단_지연시간 := T#0.5S, LS_ERR1_지연시간 := T#5S, LS_ERR2_지연시간 := T#5S, 이상리셋 := 전체_M_이상_리셋, SOL_ADV_출력 => S364_SOL_AX_RH_SLD_CLP_전진, SOL_RET_출력 => S364_SOL_AX_RH_SLD_CLP_후진, M_전진단 => S364_M_AX_RH_SLD_CLP_전진단, M_후진단 => S364_M_AX_RH_SLD_CLP_후진단, M_전진에러 => S364_M_AX_RH_SLD_CLP_전진_LS_이상, M_후진에러 => S364_M_AX_RH_SLD_CLP_후진_LS_이상, ADV_LAMP => S364_M_AX_RH_SLD_CLP_전진_LAMP, RET_LAMP => S364_M_AX_RH_SLD_CLP_후진_LAMP);
(* S364 AX RH SLIDE 동작 *)
(* Rung L230 *)
S364_M_AX_RH_SLD_조건 := S364_M_AX_CLAMP_후진단 AND S364_M_AX_LATCH_전진단 AND S364_M_AX_LH_SLD_LAT_전진단 AND S364_M_AX_RH_SLD_LAT_전진단 AND S364_M_AX_LH_SLD_CLP_후진단 AND S364_M_AX_RH_SLD_CLP_후진단 AND (S364_M_공정_불간섭 OR EGIS_CWS);
(* Rung L232 *)
S364_M_AX_RH_SLD_전진_보조 := ((S364_M_자동_운전중 AND NOT S364_M_작업_완료 AND S364_M_작업자_작업완료 AND S364_M_공정_차종_유) OR (S364_M_동작_선택_16 AND S364_전진_ON AND S364_M_수동모드)) AND S364_M_AX_RH_SLD_조건;

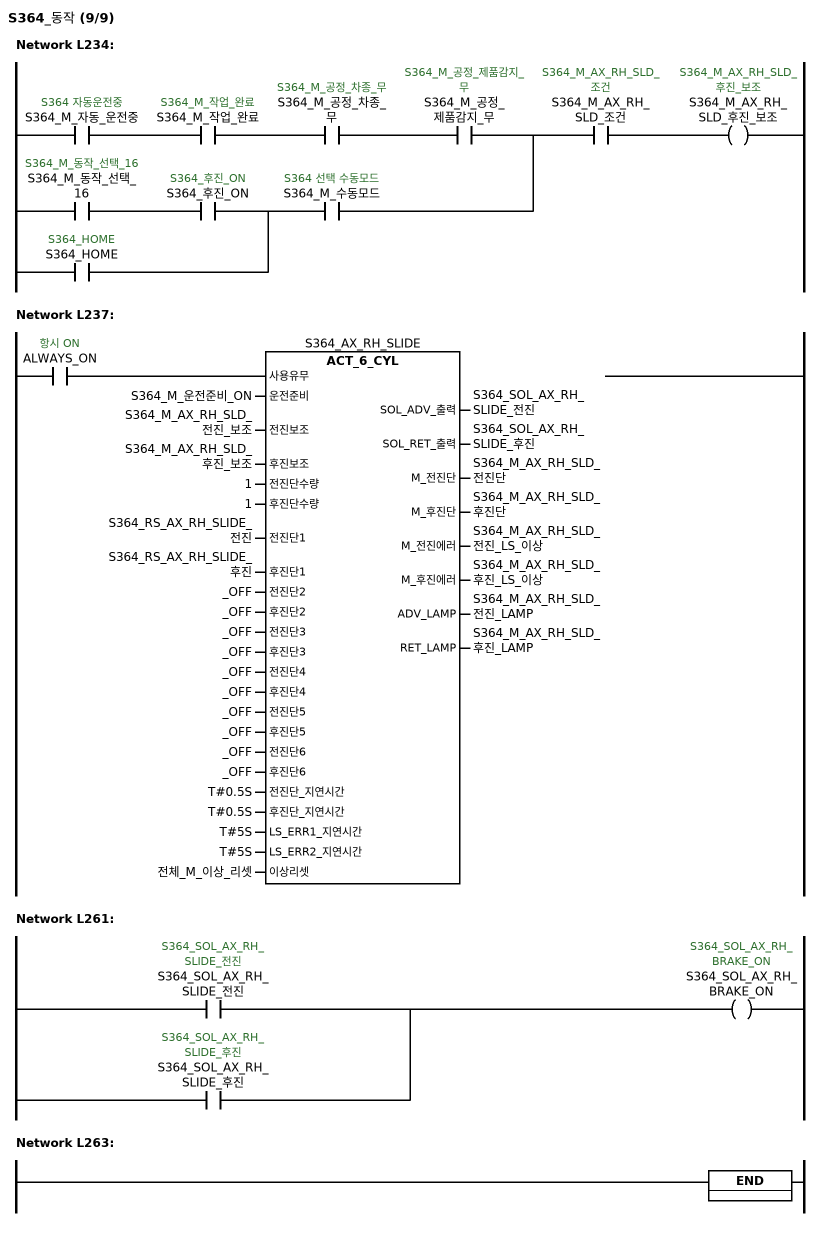
(* Rung L234 *)
S364_M_AX_RH_SLD_후진_보조 := ((S364_M_자동_운전중 AND S364_M_작업_완료 AND S364_M_공정_차종_무 AND S364_M_공정_제품감지_무) OR (((S364_M_동작_선택_16 AND S364_후진_ON) OR S364_HOME) AND S364_M_수동모드)) AND S364_M_AX_RH_SLD_조건;
(* Rung L237 *)
S364_AX_RH_SLIDE(사용유무 := ALWAYS_ON, 운전준비 := S364_M_운전준비_ON, 전진보조 := S364_M_AX_RH_SLD_전진_보조, 후진보조 := S364_M_AX_RH_SLD_후진_보조, 전진단수량 := 1, 후진단수량 := 1, 전진단1 := S364_RS_AX_RH_SLIDE_전진, 후진단1 := S364_RS_AX_RH_SLIDE_후진, 전진단2 := _OFF, 후진단2 := _OFF, 전진단3 := _OFF, 후진단3 := _OFF, 전진단4 := _OFF, 후진단4 := _OFF, 전진단5 := _OFF, 후진단5 := _OFF, 전진단6 := _OFF, 후진단6 := _OFF, 전진단_지연시간 := T#0.5S, 후진단_지연시간 := T#0.5S, LS_ERR1_지연시간 := T#5S, LS_ERR2_지연시간 := T#5S, 이상리셋 := 전체_M_이상_리셋, SOL_ADV_출력 => S364_SOL_AX_RH_SLIDE_전진, SOL_RET_출력 => S364_SOL_AX_RH_SLIDE_후진, M_전진단 => S364_M_AX_RH_SLD_전진단, M_후진단 => S364_M_AX_RH_SLD_후진단, M_전진에러 => S364_M_AX_RH_SLD_전진_LS_이상, M_후진에러 => S364_M_AX_RH_SLD_후진_LS_이상, ADV_LAMP => S364_M_AX_RH_SLD_전진_LAMP, RET_LAMP => S364_M_AX_RH_SLD_후진_LAMP);
(* Rung L261 *)
S364_SOL_AX_RH_BRAKE_ON := S364_SOL_AX_RH_SLIDE_전진 OR S364_SOL_AX_RH_SLIDE_후진;
(* Rung L263 *)
END();
END_PROGRAM

PROGRAM S364_로보트 (* task: 스캔 프로그램 *)
VAR_EXTERNAL RETAIN
    ALWAYS_ON : BOOL; (* AT %MW3.1 *) (* 항시 ON *)
    MCP_M_부저_정지 : BOOL; (* AT %MW350.5 *) (* MCP 부저정지 *)
    MCP_M_비상정지 : BOOL; (* AT %MW350.7 *) (* MCP 비상정지 이상 *)
    S362_M_공정_제품감지_유 : BOOL; (* AT %MW1001.4 *) (* S362_M_공정_제품감지_유 *)
    S364_M_R361_1_언로딩완료 : BOOL; (* AT %MW2001.4 *)
    S364_M_R361_2_로딩완료 : BOOL; (* AT %MW2001.2 *)
    S364_M_R364_1_용접가능 : BOOL; (* AT %MW2004.10 *)
    S364_M_공정_제품감지_무 : BOOL; (* AT %MW2002.5 *) (* S364_M_공정_제품감지_무 *)
    S364_M_공정_차종_AX : BOOL; (* AT %MW2002.3 *) (* S364_M_공정_차종_AX *)
    S364_M_공정_차종_무 : BOOL; (* AT %MW2002.1 *) (* S364_M_공정_차종_무 *)
    S364_M_공정_차종_유 : BOOL; (* AT %MW2002.0 *) (* S364_M_공정_차종_유 *)
    S364_M_수동모드 : BOOL; (* AT %MW2000.3 *) (* S364 선택 수동모드 *)
    S364_M_자동_START : BOOL; (* AT %MW2000.5 *) (* S364 자동운전중 *)
    S364_M_자동_운전중 : BOOL; (* AT %MW2000.4 *) (* S364 자동운전중 *)
    S364_M_작업_완료 : BOOL; (* AT %MW2001.0 *) (* S364_M_작업_완료 *)
    S364_M_작업완료_SET_PLS : BOOL; (* AT %MW2000.8 *) (* S364 M 작업완료 SET PLS *)
    S364_M_작업완료_리셋_PLS : BOOL; (* AT %MW2000.9 *) (* S364 M 작업완료 리셋 PLS *)
    S364_M_작업자_작업완료 : BOOL; (* AT %MW2001.1 *)
    S364_M_총괄_이상 : BOOL; (* AT %MW2009.0 *) (* S364_M_총괄_이상 *)
    전체_M_GATE_비상정지_정상 : BOOL; (* AT %MW308.4 *) (* 전체 M GATE 비상정지 정상 *)
    전체_M_GATE_자동기동 : BOOL; (* AT %MW308.1 *) (* 전체_M_자동_운전 *)
    전체_M_운전준비_보조 : BOOL; (* AT %MW308.5 *)
    전체_M_이상_리셋 : BOOL; (* AT %MW308.2 *) (* ALL공정 PB 이상리셋 *)
    전체_공정_M_총괄_비상정지_정상 : BOOL; (* AT %MW304.1 *)
END_VAR
VAR
    INST1 : FB494_Robot_Hyundai_HMMI_v1;
    INST2 : FB494_Robot_Hyundai_HMMI_v1;
    INST3 : FB494_Robot_Hyundai_HMMI_v1;
    R361_1_M_RB_PROG_NO : INT;
    R361_2_M_RB_PROG_NO : INT;
    R364_1_M_RB_PROG_NO : INT;
    로보트제외 : BOOL;
END_VAR
VAR_EXTERNAL
    MCP_PBL_운전준비_ON : BOOL; (* AT %MW87630.0 *) (* MCP_PBL_운전준비_ON *)
    R361_1_I_RB_INPUT : ARRAY[0..3] OF WORD; (* AT %MW84010 *) (* R361_1_I_RB_INPUT *)
    R361_1_M_I_RB_1차_작업완료 : BOOL; (* AT %MW20011.2 *) (* R361_1_M_I_RB_1차_작업완료 *)
    R361_1_M_I_RB_2차_작업완료 : BOOL; (* AT %MW20011.3 *) (* R361_1_M_I_RB_2차_작업완료 *)
    R361_1_M_I_RB_3차_작업완료 : BOOL; (* AT %MW20011.4 *) (* R361_1_M_I_RB_3차_작업완료 *)
    R361_1_M_I_RB_4차_작업완료 : BOOL; (* AT %MW20011.5 *) (* R361_1_M_I_RB_4차_작업완료 *)
    R361_1_M_I_RB_5차_작업완료 : BOOL; (* AT %MW20011.6 *) (* R361_1_M_I_RB_5차_작업완료 *)
    R361_1_M_I_RB_6차_작업완료 : BOOL; (* AT %MW20011.7 *) (* R361_1_M_I_RB_6차_작업완료 *)
    R361_1_M_I_RB_7차_작업완료 : BOOL; (* AT %MW20011.8 *) (* R361_1_M_I_RB_7차_작업완료 *)
    R361_1_M_I_RB_PAUSE_보조 : BOOL; (* AT %MW20010.5 *) (* R361_1_M_I_RB_PAUSE_보조 *)
    R361_1_M_I_RB_PLC_RUN_CHK_이상 : BOOL; (* AT %MW20010.7 *) (* R361_1_M_I_RB_PLC_RUN_CHK_이상 *)
    R361_1_M_I_RB_간섭무_1 : BOOL; (* AT %MW20012.0 *) (* R361_1_M_I_RB_간섭무_1 *)
    R361_1_M_I_RB_간섭무_10 : BOOL; (* AT %MW20012.9 *) (* R361_1_M_I_RB_간섭무_10 *)
    R361_1_M_I_RB_간섭무_11 : BOOL; (* AT %MW20012.10 *) (* R361_1_M_I_RB_간섭무_11 *)
    R361_1_M_I_RB_간섭무_12 : BOOL; (* AT %MW20012.11 *) (* R361_1_M_I_RB_간섭무_12 *)
    R361_1_M_I_RB_간섭무_2 : BOOL; (* AT %MW20012.1 *) (* R361_1_M_I_RB_간섭무_2 *)
    R361_1_M_I_RB_간섭무_3 : BOOL; (* AT %MW20012.2 *) (* R361_1_M_I_RB_간섭무_3 *)
    R361_1_M_I_RB_간섭무_4 : BOOL; (* AT %MW20012.3 *) (* R361_1_M_I_RB_간섭무_4 *)
    R361_1_M_I_RB_간섭무_5 : BOOL; (* AT %MW20012.4 *) (* R361_1_M_I_RB_간섭무_5 *)
    R361_1_M_I_RB_간섭무_6 : BOOL; (* AT %MW20012.5 *) (* R361_1_M_I_RB_간섭무_6 *)
    R361_1_M_I_RB_간섭무_7 : BOOL; (* AT %MW20012.6 *) (* R361_1_M_I_RB_간섭무_7 *)
    R361_1_M_I_RB_간섭무_8 : BOOL; (* AT %MW20012.7 *) (* R361_1_M_I_RB_간섭무_8 *)
    R361_1_M_I_RB_간섭무_9 : BOOL; (* AT %MW20012.8 *) (* R361_1_M_I_RB_간섭무_9 *)
    R361_1_M_I_RB_비상정지 : BOOL; (* AT %MW20010.4 *) (* R361_1_M_I_RB_비상정지 *)
    R361_1_M_I_RB_운전준비 : BOOL; (* AT %MW20010.0 *) (* R361_1_M_I_RB_운전준비 *)
    R361_1_M_I_RB_원위치 : BOOL; (* AT %MW20010.3 *) (* R361_1_M_I_RB_원위치 *)
    R361_1_M_I_RB_이상 : BOOL; (* AT %MW20010.2 *) (* R361_1_M_I_RB_이상 *)
    R361_1_M_I_RB_자동 : BOOL; (* AT %MW20010.1 *) (* R361_1_M_I_RB_자동 *)
    R361_1_M_I_RB_최종작업완료 : BOOL; (* AT %MW20011.0 *) (* R361_1_M_I_RB_최종작업완료 *)
    R361_1_M_I_RB_프로그램_이상 : BOOL; (* AT %MW20010.6 *) (* R361_1_M_I_RB_프로그램_이상 *)
    R361_1_M_O_RB_1_CYCLE_SET : BOOL; (* AT %MW21010.3 *) (* R361_1_M_O_RB_1_CYCLE_SET *)
    R361_1_M_O_RB_1차_작업완료_리셋 : BOOL; (* AT %MW21012.0 *) (* R361_1_M_O_RB_1차_작업완료_리셋 *)
    R361_1_M_O_RB_2차_작업완료_리셋 : BOOL; (* AT %MW21012.1 *) (* R361_1_M_O_RB_2차_작업완료_리셋 *)
    R361_1_M_O_RB_2차_진입OK : BOOL; (* AT %MW21011.8 *) (* R361_1_M_O_RB_2차_진입OK *)
    R361_1_M_O_RB_3차_작업완료_리셋 : BOOL; (* AT %MW21012.2 *) (* R361_1_M_O_RB_3차_작업완료_리셋 *)
    R361_1_M_O_RB_3차_진입OK : BOOL; (* AT %MW21011.9 *) (* R361_1_M_O_RB_3차_진입OK *)
    R361_1_M_O_RB_4차_작업완료_리셋 : BOOL; (* AT %MW21012.3 *) (* R361_1_M_O_RB_4차_작업완료_리셋 *)
    R361_1_M_O_RB_4차_진입OK : BOOL; (* AT %MW21011.10 *) (* R361_1_M_O_RB_4차_진입OK *)
    R361_1_M_O_RB_5차_작업완료_리셋 : BOOL; (* AT %MW21012.4 *) (* R361_1_M_O_RB_5차_작업완료_리셋 *)
    R361_1_M_O_RB_5차_진입OK : BOOL; (* AT %MW21011.11 *) (* R361_1_M_O_RB_5차_진입OK *)
    R361_1_M_O_RB_6차_작업완료_리셋 : BOOL; (* AT %MW21012.5 *) (* R361_1_M_O_RB_6차_작업완료_리셋 *)
    R361_1_M_O_RB_6차_진입OK : BOOL; (* AT %MW21011.12 *) (* R361_1_M_O_RB_6차_진입OK *)
    R361_1_M_O_RB_7차_작업완료_리셋 : BOOL; (* AT %MW21012.6 *) (* R361_1_M_O_RB_7차_작업완료_리셋 *)
    R361_1_M_O_RB_7차_진입OK : BOOL; (* AT %MW21011.13 *) (* R361_1_M_O_RB_7차_진입OK *)
    R361_1_M_O_RB_ATD_OK : BOOL; (* AT %MW21010.6 *) (* R361_1_M_O_RB_ATD_OK *)
    R361_1_M_O_RB_PLT_10_진입OK : BOOL; (* AT %MW21013.10 *) (* R361_1_M_O_RB_PLT_10_진입OK *)
    R361_1_M_O_RB_PLT_11_진입OK : BOOL; (* AT %MW21013.11 *) (* R361_1_M_O_RB_PLT_11_진입OK *)
    R361_1_M_O_RB_PLT_12_진입OK : BOOL; (* AT %MW21013.12 *) (* R361_1_M_O_RB_PLT_12_진입OK *)
    R361_1_M_O_RB_PLT_1_진입OK : BOOL; (* AT %MW21013.1 *) (* R361_1_M_O_RB_PLT_1_진입OK *)
    R361_1_M_O_RB_PLT_2_진입OK : BOOL; (* AT %MW21013.2 *) (* R361_1_M_O_RB_PLT_2_진입OK *)
    R361_1_M_O_RB_PLT_3_진입OK : BOOL; (* AT %MW21013.3 *) (* R361_1_M_O_RB_PLT_3_진입OK *)
    R361_1_M_O_RB_PLT_4_진입OK : BOOL; (* AT %MW21013.4 *) (* R361_1_M_O_RB_PLT_4_진입OK *)
    R361_1_M_O_RB_PLT_5_진입OK : BOOL; (* AT %MW21013.5 *) (* R361_1_M_O_RB_PLT_5_진입OK *)
    R361_1_M_O_RB_PLT_6_진입OK : BOOL; (* AT %MW21013.6 *) (* R361_1_M_O_RB_PLT_6_진입OK *)
    R361_1_M_O_RB_PLT_7_진입OK : BOOL; (* AT %MW21013.7 *) (* R361_1_M_O_RB_PLT_7_진입OK *)
    R361_1_M_O_RB_PLT_8_진입OK : BOOL; (* AT %MW21013.8 *) (* R361_1_M_O_RB_PLT_8_진입OK *)
    R361_1_M_O_RB_PLT_9_진입OK : BOOL; (* AT %MW21013.9 *) (* R361_1_M_O_RB_PLT_9_진입OK *)
    R361_1_M_O_RB_PLT_카운터리셋_보조 : BOOL; (* AT %MW21010.10 *) (* R361_1_M_O_RB_PLT_카운터리셋_보조 *)
    R361_1_M_O_RB_RESTART_OK : BOOL; (* AT %MW21010.2 *) (* R361_1_M_O_RB_RESTART_OK *)
    R361_1_M_O_RB_START_OK : BOOL; (* AT %MW21010.0 *) (* R361_1_M_O_RB_START_OK *)
    R361_1_M_O_RB_TEST_MODE_5000회 : BOOL; (* AT %MW21010.12 *) (* R361_1_M_O_RB_TEST_MODE_5000회 *)
    R361_1_M_O_RB_TIP_교체_시작 : BOOL; (* AT %MW21010.7 *) (* R361_1_M_O_RB_TIP_교체_시작 *)
    R361_1_M_O_RB_TIP_교체_완료 : BOOL; (* AT %MW21010.8 *) (* R361_1_M_O_RB_TIP_교체_완료 *)
    R361_1_M_O_RB_VIP_MODE : BOOL; (* AT %MW21010.11 *) (* R361_1_M_O_RB_VIP_MODE *)
    R361_1_M_O_RB_냉각수_차단_요청 : BOOL; (* AT %MW21010.9 *) (* R361_1_M_O_RB_냉각수_차단_요청 *)
    R361_1_M_O_RB_진입OK_AX차종 : BOOL; (* AT %MW21011.0 *) (* R361_1_M_O_RB_진입OK_AX차종 *)
    R361_1_M_O_RB_진입OK_B차종 : BOOL; (* AT %MW21011.1 *) (* R361_1_M_O_RB_진입OK_B차종 *)
    R361_1_M_O_RB_진입OK_C차종 : BOOL; (* AT %MW21011.2 *) (* R361_1_M_O_RB_진입OK_C차종 *)
    R361_1_M_O_RB_진입OK_D차종 : BOOL; (* AT %MW21011.3 *) (* R361_1_M_O_RB_진입OK_D차종 *)
    R361_1_M_O_RB_진입OK_E차종 : BOOL; (* AT %MW21011.4 *) (* R361_1_M_O_RB_진입OK_E차종 *)
    R361_1_M_O_RB_진입OK_F차종 : BOOL; (* AT %MW21011.5 *) (* R361_1_M_O_RB_진입OK_F차종 *)
    R361_1_M_O_RB_진입OK_G차종 : BOOL; (* AT %MW21011.6 *) (* R361_1_M_O_RB_진입OK_G차종 *)
    R361_1_M_O_RB_진입OK_H차종 : BOOL; (* AT %MW21011.7 *) (* R361_1_M_O_RB_진입OK_H차종 *)
    R361_1_M_O_RB_최종_작업완료_리셋 : BOOL; (* AT %MW21010.5 *) (* R361_1_M_O_RB_최종_작업완료_리셋 *)
    R361_1_M_O_RB_프로그램_OK : BOOL; (* AT %MW21010.1 *) (* R361_1_M_O_RB_프로그램_OK *)
    R361_1_O_RB_OUTPUT : ARRAY[0..3] OF WORD; (* AT %MW94010 *) (* R361_1_O_RB_OUTPUT *)
    R361_2_I_RB_INPUT : ARRAY[0..3] OF WORD; (* AT %MW84020 *) (* R361_2_I_RB_INPUT *)
    R361_2_M_I_RB_1차_작업완료 : BOOL; (* AT %MW20021.2 *) (* R361_2_M_I_RB_1차_작업완료 *)
    R361_2_M_I_RB_2차_작업완료 : BOOL; (* AT %MW20021.3 *) (* R361_2_M_I_RB_2차_작업완료 *)
    R361_2_M_I_RB_3차_작업완료 : BOOL; (* AT %MW20021.4 *) (* R361_2_M_I_RB_3차_작업완료 *)
    R361_2_M_I_RB_4차_작업완료 : BOOL; (* AT %MW20021.5 *) (* R361_2_M_I_RB_4차_작업완료 *)
    R361_2_M_I_RB_5차_작업완료 : BOOL; (* AT %MW20021.6 *) (* R361_2_M_I_RB_5차_작업완료 *)
    R361_2_M_I_RB_6차_작업완료 : BOOL; (* AT %MW20021.7 *) (* R361_2_M_I_RB_6차_작업완료 *)
    R361_2_M_I_RB_7차_작업완료 : BOOL; (* AT %MW20021.8 *) (* R361_2_M_I_RB_7차_작업완료 *)
    R361_2_M_I_RB_PAUSE_보조 : BOOL; (* AT %MW20020.5 *) (* R361_2_M_I_RB_PAUSE_보조 *)
    R361_2_M_I_RB_PLC_RUN_CHK_이상 : BOOL; (* AT %MW20020.7 *) (* R361_2_M_I_RB_PLC_RUN_CHK_이상 *)
    R361_2_M_I_RB_간섭무_1 : BOOL; (* AT %MW20022.0 *) (* R361_2_M_I_RB_간섭무_1 *)
    R361_2_M_I_RB_간섭무_10 : BOOL; (* AT %MW20022.9 *) (* R361_2_M_I_RB_간섭무_10 *)
    R361_2_M_I_RB_간섭무_11 : BOOL; (* AT %MW20022.10 *) (* R361_2_M_I_RB_간섭무_11 *)
    R361_2_M_I_RB_간섭무_12 : BOOL; (* AT %MW20022.11 *) (* R361_2_M_I_RB_간섭무_12 *)
    R361_2_M_I_RB_간섭무_2 : BOOL; (* AT %MW20022.1 *) (* R361_2_M_I_RB_간섭무_2 *)
    R361_2_M_I_RB_간섭무_3 : BOOL; (* AT %MW20022.2 *) (* R361_2_M_I_RB_간섭무_3 *)
    R361_2_M_I_RB_간섭무_4 : BOOL; (* AT %MW20022.3 *) (* R361_2_M_I_RB_간섭무_4 *)
    R361_2_M_I_RB_간섭무_5 : BOOL; (* AT %MW20022.4 *) (* R361_2_M_I_RB_간섭무_5 *)
    R361_2_M_I_RB_간섭무_6 : BOOL; (* AT %MW20022.5 *) (* R361_2_M_I_RB_간섭무_6 *)
    R361_2_M_I_RB_간섭무_7 : BOOL; (* AT %MW20022.6 *) (* R361_2_M_I_RB_간섭무_7 *)
    R361_2_M_I_RB_간섭무_8 : BOOL; (* AT %MW20022.7 *) (* R361_2_M_I_RB_간섭무_8 *)
    R361_2_M_I_RB_간섭무_9 : BOOL; (* AT %MW20022.8 *) (* R361_2_M_I_RB_간섭무_9 *)
    R361_2_M_I_RB_비상정지 : BOOL; (* AT %MW20020.4 *) (* R361_2_M_I_RB_비상정지 *)
    R361_2_M_I_RB_운전준비 : BOOL; (* AT %MW20020.0 *) (* R361_2_M_I_RB_운전준비 *)
    R361_2_M_I_RB_원위치 : BOOL; (* AT %MW20020.3 *) (* R361_2_M_I_RB_원위치 *)
    R361_2_M_I_RB_이상 : BOOL; (* AT %MW20020.2 *) (* R361_2_M_I_RB_이상 *)
    R361_2_M_I_RB_자동 : BOOL; (* AT %MW20020.1 *) (* R361_2_M_I_RB_자동 *)
    R361_2_M_I_RB_최종작업완료 : BOOL; (* AT %MW20021.0 *) (* R361_2_M_I_RB_최종작업완료 *)
    R361_2_M_I_RB_프로그램_이상 : BOOL; (* AT %MW20020.6 *) (* R361_2_M_I_RB_프로그램_이상 *)
    R361_2_M_O_RB_1_CYCLE_SET : BOOL; (* AT %MW21020.3 *) (* R361_2_M_O_RB_1_CYCLE_SET *)
    R361_2_M_O_RB_1차_작업완료_리셋 : BOOL; (* AT %MW21022.0 *) (* R361_2_M_O_RB_1차_작업완료_리셋 *)
    R361_2_M_O_RB_2차_작업완료_리셋 : BOOL; (* AT %MW21022.1 *) (* R361_2_M_O_RB_2차_작업완료_리셋 *)
    R361_2_M_O_RB_2차_진입OK : BOOL; (* AT %MW21021.8 *) (* R361_2_M_O_RB_2차_진입OK *)
    R361_2_M_O_RB_3차_작업완료_리셋 : BOOL; (* AT %MW21022.2 *) (* R361_2_M_O_RB_3차_작업완료_리셋 *)
    R361_2_M_O_RB_3차_진입OK : BOOL; (* AT %MW21021.9 *) (* R361_2_M_O_RB_3차_진입OK *)
    R361_2_M_O_RB_4차_작업완료_리셋 : BOOL; (* AT %MW21022.3 *) (* R361_2_M_O_RB_4차_작업완료_리셋 *)
    R361_2_M_O_RB_4차_진입OK : BOOL; (* AT %MW21021.10 *) (* R361_2_M_O_RB_4차_진입OK *)
    R361_2_M_O_RB_5차_작업완료_리셋 : BOOL; (* AT %MW21022.4 *) (* R361_2_M_O_RB_5차_작업완료_리셋 *)
    R361_2_M_O_RB_5차_진입OK : BOOL; (* AT %MW21021.11 *) (* R361_2_M_O_RB_5차_진입OK *)
    R361_2_M_O_RB_6차_작업완료_리셋 : BOOL; (* AT %MW21022.5 *) (* R361_2_M_O_RB_6차_작업완료_리셋 *)
    R361_2_M_O_RB_6차_진입OK : BOOL; (* AT %MW21021.12 *) (* R361_2_M_O_RB_6차_진입OK *)
    R361_2_M_O_RB_7차_작업완료_리셋 : BOOL; (* AT %MW21022.6 *) (* R361_2_M_O_RB_7차_작업완료_리셋 *)
    R361_2_M_O_RB_7차_진입OK : BOOL; (* AT %MW21021.13 *) (* R361_2_M_O_RB_7차_진입OK *)
    R361_2_M_O_RB_ATD_OK : BOOL; (* AT %MW21020.6 *) (* R361_2_M_O_RB_ATD_OK *)
    R361_2_M_O_RB_PLT_10_진입OK : BOOL; (* AT %MW21023.10 *) (* R361_2_M_O_RB_PLT_10_진입OK *)
    R361_2_M_O_RB_PLT_11_진입OK : BOOL; (* AT %MW21023.11 *) (* R361_2_M_O_RB_PLT_11_진입OK *)
    R361_2_M_O_RB_PLT_12_진입OK : BOOL; (* AT %MW21023.12 *) (* R361_2_M_O_RB_PLT_12_진입OK *)
    R361_2_M_O_RB_PLT_1_진입OK : BOOL; (* AT %MW21023.1 *) (* R361_2_M_O_RB_PLT_1_진입OK *)
    R361_2_M_O_RB_PLT_2_진입OK : BOOL; (* AT %MW21023.2 *) (* R361_2_M_O_RB_PLT_2_진입OK *)
    R361_2_M_O_RB_PLT_3_진입OK : BOOL; (* AT %MW21023.3 *) (* R361_2_M_O_RB_PLT_3_진입OK *)
    R361_2_M_O_RB_PLT_4_진입OK : BOOL; (* AT %MW21023.4 *) (* R361_2_M_O_RB_PLT_4_진입OK *)
    R361_2_M_O_RB_PLT_5_진입OK : BOOL; (* AT %MW21023.5 *) (* R361_2_M_O_RB_PLT_5_진입OK *)
    R361_2_M_O_RB_PLT_6_진입OK : BOOL; (* AT %MW21023.6 *) (* R361_2_M_O_RB_PLT_6_진입OK *)
    R361_2_M_O_RB_PLT_7_진입OK : BOOL; (* AT %MW21023.7 *) (* R361_2_M_O_RB_PLT_7_진입OK *)
    R361_2_M_O_RB_PLT_8_진입OK : BOOL; (* AT %MW21023.8 *) (* R361_2_M_O_RB_PLT_8_진입OK *)
    R361_2_M_O_RB_PLT_9_진입OK : BOOL; (* AT %MW21023.9 *) (* R361_2_M_O_RB_PLT_9_진입OK *)
    R361_2_M_O_RB_PLT_카운터리셋_보조 : BOOL; (* AT %MW21020.10 *) (* R361_2_M_O_RB_PLT_카운터리셋_보조 *)
    R361_2_M_O_RB_RESTART_OK : BOOL; (* AT %MW21020.2 *) (* R361_2_M_O_RB_RESTART_OK *)
    R361_2_M_O_RB_START_OK : BOOL; (* AT %MW21020.0 *) (* R361_2_M_O_RB_START_OK *)
    R361_2_M_O_RB_TEST_MODE_5000회 : BOOL; (* AT %MW21020.12 *) (* R361_2_M_O_RB_TEST_MODE_5000회 *)
    R361_2_M_O_RB_TIP_교체_시작 : BOOL; (* AT %MW21020.7 *) (* R361_2_M_O_RB_TIP_교체_시작 *)
    R361_2_M_O_RB_TIP_교체_완료 : BOOL; (* AT %MW21020.8 *) (* R361_2_M_O_RB_TIP_교체_완료 *)
    R361_2_M_O_RB_VIP_MODE : BOOL; (* AT %MW21020.11 *) (* R361_2_M_O_RB_VIP_MODE *)
    R361_2_M_O_RB_냉각수_차단_요청 : BOOL; (* AT %MW21020.9 *) (* R361_2_M_O_RB_냉각수_차단_요청 *)
    R361_2_M_O_RB_진입OK_AX차종 : BOOL; (* AT %MW21021.0 *) (* R361_2_M_O_RB_진입OK_AX차종 *)
    R361_2_M_O_RB_진입OK_B차종 : BOOL; (* AT %MW21021.1 *) (* R361_2_M_O_RB_진입OK_B차종 *)
    R361_2_M_O_RB_진입OK_C차종 : BOOL; (* AT %MW21021.2 *) (* R361_2_M_O_RB_진입OK_C차종 *)
    R361_2_M_O_RB_진입OK_D차종 : BOOL; (* AT %MW21021.3 *) (* R361_2_M_O_RB_진입OK_D차종 *)
    R361_2_M_O_RB_진입OK_E차종 : BOOL; (* AT %MW21021.4 *) (* R361_2_M_O_RB_진입OK_E차종 *)
    R361_2_M_O_RB_진입OK_F차종 : BOOL; (* AT %MW21021.5 *) (* R361_2_M_O_RB_진입OK_F차종 *)
    R361_2_M_O_RB_진입OK_G차종 : BOOL; (* AT %MW21021.6 *) (* R361_2_M_O_RB_진입OK_G차종 *)
    R361_2_M_O_RB_진입OK_H차종 : BOOL; (* AT %MW21021.7 *) (* R361_2_M_O_RB_진입OK_H차종 *)
    R361_2_M_O_RB_최종_작업완료_리셋 : BOOL; (* AT %MW21020.5 *) (* R361_2_M_O_RB_최종_작업완료_리셋 *)
    R361_2_M_O_RB_프로그램_OK : BOOL; (* AT %MW21020.1 *) (* R361_2_M_O_RB_프로그램_OK *)
    R361_2_O_RB_OUTPUT : ARRAY[0..3] OF WORD; (* AT %MW94020 *) (* R361_2_O_RB_OUTPUT *)
    R364_1_I_RB_INPUT : ARRAY[0..3] OF WORD; (* AT %MW84050 *) (* R364_1_I_RB_INPUT *)
    R364_1_M_I_RB_1차_작업완료 : BOOL; (* AT %MW20051.2 *) (* R364_1_M_I_RB_1차_작업완료 *)
    R364_1_M_I_RB_2차_작업완료 : BOOL; (* AT %MW20051.3 *) (* R364_1_M_I_RB_2차_작업완료 *)
    R364_1_M_I_RB_3차_작업완료 : BOOL; (* AT %MW20051.4 *) (* R364_1_M_I_RB_3차_작업완료 *)
    R364_1_M_I_RB_4차_작업완료 : BOOL; (* AT %MW20051.5 *) (* R364_1_M_I_RB_4차_작업완료 *)
    R364_1_M_I_RB_5차_작업완료 : BOOL; (* AT %MW20051.6 *) (* R364_1_M_I_RB_5차_작업완료 *)
    R364_1_M_I_RB_6차_작업완료 : BOOL; (* AT %MW20051.7 *) (* R364_1_M_I_RB_6차_작업완료 *)
    R364_1_M_I_RB_7차_작업완료 : BOOL; (* AT %MW20051.8 *) (* R364_1_M_I_RB_7차_작업완료 *)
    R364_1_M_I_RB_PAUSE_보조 : BOOL; (* AT %MW20050.5 *) (* R364_1_M_I_RB_PAUSE_보조 *)
    R364_1_M_I_RB_PLC_RUN_CHK_이상 : BOOL; (* AT %MW20050.7 *) (* R364_1_M_I_RB_PLC_RUN_CHK_이상 *)
    R364_1_M_I_RB_간섭무_1 : BOOL; (* AT %MW20052.0 *) (* R364_1_M_I_RB_간섭무_1 *)
    R364_1_M_I_RB_간섭무_10 : BOOL; (* AT %MW20052.9 *) (* R364_1_M_I_RB_간섭무_10 *)
    R364_1_M_I_RB_간섭무_11 : BOOL; (* AT %MW20052.10 *) (* R364_1_M_I_RB_간섭무_11 *)
    R364_1_M_I_RB_간섭무_12 : BOOL; (* AT %MW20052.11 *) (* R364_1_M_I_RB_간섭무_12 *)
    R364_1_M_I_RB_간섭무_2 : BOOL; (* AT %MW20052.1 *) (* R364_1_M_I_RB_간섭무_2 *)
    R364_1_M_I_RB_간섭무_3 : BOOL; (* AT %MW20052.2 *) (* R364_1_M_I_RB_간섭무_3 *)
    R364_1_M_I_RB_간섭무_4 : BOOL; (* AT %MW20052.3 *) (* R364_1_M_I_RB_간섭무_4 *)
    R364_1_M_I_RB_간섭무_5 : BOOL; (* AT %MW20052.4 *) (* R364_1_M_I_RB_간섭무_5 *)
    R364_1_M_I_RB_간섭무_6 : BOOL; (* AT %MW20052.5 *) (* R364_1_M_I_RB_간섭무_6 *)
    R364_1_M_I_RB_간섭무_7 : BOOL; (* AT %MW20052.6 *) (* R364_1_M_I_RB_간섭무_7 *)
    R364_1_M_I_RB_간섭무_8 : BOOL; (* AT %MW20052.7 *) (* R364_1_M_I_RB_간섭무_8 *)
    R364_1_M_I_RB_간섭무_9 : BOOL; (* AT %MW20052.8 *) (* R364_1_M_I_RB_간섭무_9 *)
    R364_1_M_I_RB_비상정지 : BOOL; (* AT %MW20050.4 *) (* R364_1_M_I_RB_비상정지 *)
    R364_1_M_I_RB_운전준비 : BOOL; (* AT %MW20050.0 *) (* R364_1_M_I_RB_운전준비 *)
    R364_1_M_I_RB_원위치 : BOOL; (* AT %MW20050.3 *) (* R364_1_M_I_RB_원위치 *)
    R364_1_M_I_RB_이상 : BOOL; (* AT %MW20050.2 *) (* R364_1_M_I_RB_이상 *)
    R364_1_M_I_RB_자동 : BOOL; (* AT %MW20050.1 *) (* R364_1_M_I_RB_자동 *)
    R364_1_M_I_RB_최종작업완료 : BOOL; (* AT %MW20051.0 *) (* R364_1_M_I_RB_최종작업완료 *)
    R364_1_M_I_RB_프로그램_이상 : BOOL; (* AT %MW20050.6 *) (* R364_1_M_I_RB_프로그램_이상 *)
    R364_1_M_O_RB_1_CYCLE_SET : BOOL; (* AT %MW21050.3 *) (* R364_1_M_O_RB_1_CYCLE_SET *)
    R364_1_M_O_RB_1차_작업완료_리셋 : BOOL; (* AT %MW21052.0 *) (* R364_1_M_O_RB_1차_작업완료_리셋 *)
    R364_1_M_O_RB_2차_작업완료_리셋 : BOOL; (* AT %MW21052.1 *) (* R364_1_M_O_RB_2차_작업완료_리셋 *)
    R364_1_M_O_RB_2차_진입OK : BOOL; (* AT %MW21051.8 *) (* R364_1_M_O_RB_2차_진입OK *)
    R364_1_M_O_RB_3차_작업완료_리셋 : BOOL; (* AT %MW21052.2 *) (* R364_1_M_O_RB_3차_작업완료_리셋 *)
    R364_1_M_O_RB_3차_진입OK : BOOL; (* AT %MW21051.9 *) (* R364_1_M_O_RB_3차_진입OK *)
    R364_1_M_O_RB_4차_작업완료_리셋 : BOOL; (* AT %MW21052.3 *) (* R364_1_M_O_RB_4차_작업완료_리셋 *)
    R364_1_M_O_RB_4차_진입OK : BOOL; (* AT %MW21051.10 *) (* R364_1_M_O_RB_4차_진입OK *)
    R364_1_M_O_RB_5차_작업완료_리셋 : BOOL; (* AT %MW21052.4 *) (* R364_1_M_O_RB_5차_작업완료_리셋 *)
    R364_1_M_O_RB_5차_진입OK : BOOL; (* AT %MW21051.11 *) (* R364_1_M_O_RB_5차_진입OK *)
    R364_1_M_O_RB_6차_작업완료_리셋 : BOOL; (* AT %MW21052.5 *) (* R364_1_M_O_RB_6차_작업완료_리셋 *)
    R364_1_M_O_RB_6차_진입OK : BOOL; (* AT %MW21051.12 *) (* R364_1_M_O_RB_6차_진입OK *)
    R364_1_M_O_RB_7차_작업완료_리셋 : BOOL; (* AT %MW21052.6 *) (* R364_1_M_O_RB_7차_작업완료_리셋 *)
    R364_1_M_O_RB_7차_진입OK : BOOL; (* AT %MW21051.13 *) (* R364_1_M_O_RB_7차_진입OK *)
    R364_1_M_O_RB_ATD_OK : BOOL; (* AT %MW21050.6 *) (* R364_1_M_O_RB_ATD_OK *)
    R364_1_M_O_RB_PLT_10_진입OK : BOOL; (* AT %MW21053.10 *) (* R364_1_M_O_RB_PLT_10_진입OK *)
    R364_1_M_O_RB_PLT_11_진입OK : BOOL; (* AT %MW21053.11 *) (* R364_1_M_O_RB_PLT_11_진입OK *)
    R364_1_M_O_RB_PLT_12_진입OK : BOOL; (* AT %MW21053.12 *) (* R364_1_M_O_RB_PLT_12_진입OK *)
    R364_1_M_O_RB_PLT_1_진입OK : BOOL; (* AT %MW21053.1 *) (* R364_1_M_O_RB_PLT_1_진입OK *)
    R364_1_M_O_RB_PLT_2_진입OK : BOOL; (* AT %MW21053.2 *) (* R364_1_M_O_RB_PLT_2_진입OK *)
    R364_1_M_O_RB_PLT_3_진입OK : BOOL; (* AT %MW21053.3 *) (* R364_1_M_O_RB_PLT_3_진입OK *)
    R364_1_M_O_RB_PLT_4_진입OK : BOOL; (* AT %MW21053.4 *) (* R364_1_M_O_RB_PLT_4_진입OK *)
    R364_1_M_O_RB_PLT_5_진입OK : BOOL; (* AT %MW21053.5 *) (* R364_1_M_O_RB_PLT_5_진입OK *)
    R364_1_M_O_RB_PLT_6_진입OK : BOOL; (* AT %MW21053.6 *) (* R364_1_M_O_RB_PLT_6_진입OK *)
    R364_1_M_O_RB_PLT_7_진입OK : BOOL; (* AT %MW21053.7 *) (* R364_1_M_O_RB_PLT_7_진입OK *)
    R364_1_M_O_RB_PLT_8_진입OK : BOOL; (* AT %MW21053.8 *) (* R364_1_M_O_RB_PLT_8_진입OK *)
    R364_1_M_O_RB_PLT_9_진입OK : BOOL; (* AT %MW21053.9 *) (* R364_1_M_O_RB_PLT_9_진입OK *)
    R364_1_M_O_RB_PLT_카운터리셋_보조 : BOOL; (* AT %MW21050.10 *) (* R364_1_M_O_RB_PLT_카운터리셋_보조 *)
    R364_1_M_O_RB_PROG_NO : WORD; (* AT %MW21054 *)
    R364_1_M_O_RB_RESTART_OK : BOOL; (* AT %MW21050.2 *) (* R364_1_M_O_RB_RESTART_OK *)
    R364_1_M_O_RB_START_OK : BOOL; (* AT %MW21050.0 *) (* R364_1_M_O_RB_START_OK *)
    R364_1_M_O_RB_TEST_MODE_5000회 : BOOL; (* AT %MW21050.12 *) (* R364_1_M_O_RB_TEST_MODE_5000회 *)
    R364_1_M_O_RB_TIP_교체_시작 : BOOL; (* AT %MW21050.7 *) (* R364_1_M_O_RB_TIP_교체_시작 *)
    R364_1_M_O_RB_TIP_교체_완료 : BOOL; (* AT %MW21050.8 *) (* R364_1_M_O_RB_TIP_교체_완료 *)
    R364_1_M_O_RB_VIP_MODE : BOOL; (* AT %MW21050.11 *) (* R364_1_M_O_RB_VIP_MODE *)
    R364_1_M_O_RB_냉각수_차단_요청 : BOOL; (* AT %MW21050.9 *) (* R364_1_M_O_RB_냉각수_차단_요청 *)
    R364_1_M_O_RB_진입OK_AX차종 : BOOL; (* AT %MW21051.0 *) (* R364_1_M_O_RB_진입OK_AX차종 *)
    R364_1_M_O_RB_진입OK_B차종 : BOOL; (* AT %MW21051.1 *) (* R364_1_M_O_RB_진입OK_B차종 *)
    R364_1_M_O_RB_진입OK_C차종 : BOOL; (* AT %MW21051.2 *) (* R364_1_M_O_RB_진입OK_C차종 *)
    R364_1_M_O_RB_진입OK_D차종 : BOOL; (* AT %MW21051.3 *) (* R364_1_M_O_RB_진입OK_D차종 *)
    R364_1_M_O_RB_진입OK_E차종 : BOOL; (* AT %MW21051.4 *) (* R364_1_M_O_RB_진입OK_E차종 *)
    R364_1_M_O_RB_진입OK_F차종 : BOOL; (* AT %MW21051.5 *) (* R364_1_M_O_RB_진입OK_F차종 *)
    R364_1_M_O_RB_진입OK_G차종 : BOOL; (* AT %MW21051.6 *) (* R364_1_M_O_RB_진입OK_G차종 *)
    R364_1_M_O_RB_진입OK_H차종 : BOOL; (* AT %MW21051.7 *) (* R364_1_M_O_RB_진입OK_H차종 *)
    R364_1_M_O_RB_최종_작업완료_리셋 : BOOL; (* AT %MW21050.5 *) (* R364_1_M_O_RB_최종_작업완료_리셋 *)
    R364_1_M_O_RB_프로그램_OK : BOOL; (* AT %MW21050.1 *) (* R364_1_M_O_RB_프로그램_OK *)
    R364_1_O_RB_OUTPUT : ARRAY[0..3] OF WORD; (* AT %MW94050 *) (* R364_1_O_RB_OUTPUT *)
END_VAR
(* ladder body could not be read *)
END_PROGRAM

PROGRAM S364_로보트_용접타점수 (* task: 스캔 프로그램 *)
VAR_EXTERNAL
    R364_1_I_RB_용접타점수 : WORD; (* AT %MW84055 *) (* R364_1_I_RB_용접타점수 *)
    R364_1_M_I_RB_1차_작업완료 : BOOL; (* AT %MW20051.2 *) (* R364_1_M_I_RB_1차_작업완료 *)
    R366_1_I_RB_용접타점수 : WORD; (* AT %MW84065 *) (* R366_1_I_RB_용접타점수 *)
END_VAR
VAR_EXTERNAL RETAIN
    R364_1_M_AX_차종_용접타점수 : WORD; (* AT %MW8010 *)
    R364_1_M_용접완료 : BOOL; (* AT %MW2006.1 *)
    R364_1_M_용접타점수_OK : BOOL; (* AT %MW2006.8 *)
    R366_1_M_용접완료 : BOOL; (* AT %MW3006.1 *)
    R366_1_M_용접타점수_OK : BOOL; (* AT %MW3006.8 *)
    S364_M_전체_용접완료 : BOOL; (* AT %MW2006.0 *)
    S364_M_차종1_AX : BOOL; (* AT %MW10121.0 *) (* S364 M 차종1 AX *)
    S366_M_R366_1_용접완료 : BOOL; (* AT %MW3001.3 *)
    S366_M_전체_용접완료 : BOOL; (* AT %MW3006.0 *)
END_VAR
VAR
    _t1 : BOOL;
END_VAR

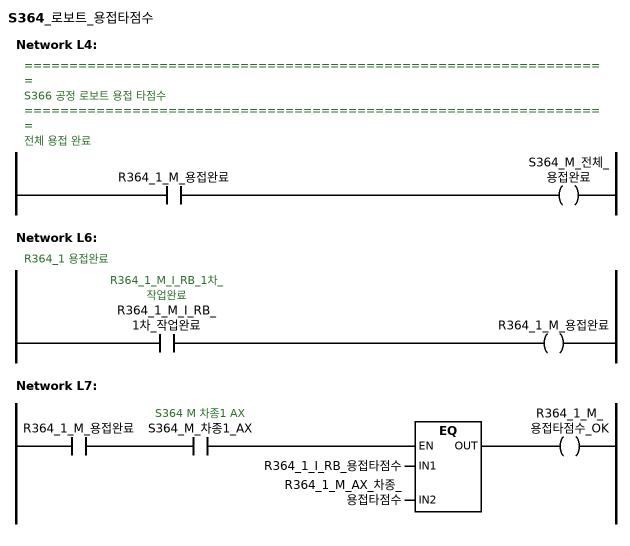
(* ================================================================= *)
(* S366 공정 로보트 용접 타점수 *)
(* ================================================================= *)
(* 전체 용접 완료 *)
(* Rung L4 *)
S364_M_전체_용접완료 := R364_1_M_용접완료;
(* R364_1 용접완료 *)
(* Rung L6 *)
R364_1_M_용접완료 := R364_1_M_I_RB_1차_작업완료;
(* Rung L7 *)
IF R364_1_M_용접완료 AND S364_M_차종1_AX THEN _t1 := R364_1_I_RB_용접타점수 = R364_1_M_AX_차종_용접타점수; END_IF;
R364_1_M_용접타점수_OK := _t1;
END_PROGRAM

PROGRAM S364_이상 (* task: 스캔 프로그램 *)
VAR
    INST : TON;
    INST1 : TON;
    INST10 : TON;
    INST11 : TON;
    INST12 : TON;
    INST13 : TON;
    INST14 : TON;
    INST15 : TON;
    INST16 : TON;
    INST17 : TON;
    INST18 : TON;
    INST19 : TON;
    INST2 : TON;
    INST20 : TON;
    INST21 : TON;
    INST22 : TON;
    INST23 : TON;
    INST24 : TON;
    INST25 : TON;
    INST26 : TON;
    INST27 : TON;
    INST28 : TON;
    INST29 : TON;
    INST3 : TON;
    INST4 : TON;
    INST5 : TON;
    INST8 : TON;
    INST9 : TON;
END_VAR
VAR_EXTERNAL
    R361_1_M_I_RB_이상 : BOOL; (* AT %MW20010.2 *) (* R361_1_M_I_RB_이상 *)
    R361_1_M_I_RB_프로그램_이상 : BOOL; (* AT %MW20010.6 *) (* R361_1_M_I_RB_프로그램_이상 *)
    R364_1_M_I_RB_이상 : BOOL; (* AT %MW20050.2 *) (* R364_1_M_I_RB_이상 *)
    R364_1_M_I_RB_프로그램_이상 : BOOL; (* AT %MW20050.6 *) (* R364_1_M_I_RB_프로그램_이상 *)
    S364_7_15_PLC_BOX_CP_TRIP : BOOL; (* AT %MW87152.15 *) (* S364_7_15_PLC_BOX_CP_TRIP *)
    S364_7_16_PLC_BOX_CP_TRIP : BOOL; (* AT %MW87162.15 *) (* S364_7_16_PLC_BOX_CP_TRIP *)
    S364_LC_정상1 : BOOL; (* AT %MW87165.3 *)
    S364_LC_정상2 : BOOL; (* AT %MW87165.4 *)
    S364_MAT_정상1 : BOOL; (* AT %MW87165.6 *)
    S364_MAT_정상2 : BOOL; (* AT %MW87165.7 *)
    S364_PB_AX_작업_완료 : BOOL; (* AT %MW87152.9 *) (* S364_PB_AX_작업_완료 *)
    S364_공기압_AIR_CHECK : BOOL; (* AT %MW87152.14 *) (* S364_공기압_AIR_CHECK *)
    _0004_EB01_CFG_ER : BOOL; (* AT %MW184022.0 *) (* EB 구성 에러 *)
    _0004_EB01_DEER : BOOL; (* AT %MW184022.1 *) (* EB 운전 중 탈락 *)
    _0004_EB05_CFG_ER : BOOL; (* AT %MW184032.0 *) (* EB 구성 에러 *)
    _0004_EB05_DEER : BOOL; (* AT %MW184032.1 *) (* EB 운전 중 탈락 *)
    _0007_EB10_CFG_ER : BOOL; (* AT %MW187040.0 *) (* EB 구성 에러 *)
    _0007_EB10_DEER : BOOL; (* AT %MW187040.1 *) (* EB 운전 중 탈락 *)
    _0007_EB10_IO_DEER : BOOL; (* AT %MW187041.2 *) (* EB IO 탈락 에러 *)
    _0007_EB10_IO_TYER : BOOL; (* AT %MW187041.1 *) (* EB IO 타입 에러 *)
    _0007_EB15_CFG_ER : BOOL; (* AT %MW187058.0 *) (* EB 구성 에러 *)
    _0007_EB15_DEER : BOOL; (* AT %MW187058.1 *) (* EB 운전 중 탈락 *)
    _0007_EB15_IO_DEER : BOOL; (* AT %MW187059.2 *) (* EB IO 탈락 에러 *)
    _0007_EB15_IO_TYER : BOOL; (* AT %MW187059.1 *) (* EB IO 타입 에러 *)
    _0007_EB16_CFG_ER : BOOL; (* AT %MW187064.0 *) (* EB 구성 에러 *)
    _0007_EB16_DEER : BOOL; (* AT %MW187064.1 *) (* EB 운전 중 탈락 *)
    _0007_EB16_IO_DEER : BOOL; (* AT %MW187065.2 *) (* EB IO 탈락 에러 *)
    _0007_EB16_IO_TYER : BOOL; (* AT %MW187065.1 *) (* EB IO 타입 에러 *)
END_VAR
VAR_EXTERNAL RETAIN
    R364_1_M_NODE_4_05_통신_이상 : BOOL; (* AT %MW2024.8 *)
    R364_1_M_용접_카운트_이상 : BOOL; (* AT %MW2029.0 *)
    R364_1_M_용접완료 : BOOL; (* AT %MW2006.1 *)
    R364_1_M_용접타점수_OK : BOOL; (* AT %MW2006.8 *)
    S362_M_공정_불간섭 : BOOL; (* AT %MW1004.1 *) (* S362_M_공정_불간섭 *)
    S362_M_공정_제품감지_무 : BOOL; (* AT %MW1001.5 *) (* S362_M_공정_제품감지_무 *)
    S362_M_공정_차종_유 : BOOL; (* AT %MW1002.0 *) (* S362_M_공정_차종_유 *)
    S362_M_자동_운전중 : BOOL; (* AT %MW1000.4 *) (* S362 자동운전중 *)
    S362_M_작업자_작업_가능 : BOOL; (* AT %MW1004.8 *) (* S362 M 작업자 작업 가능 *)
    S364_LH_M_NODE_7_16_통신_이상 : BOOL; (* AT %MW2024.0 *)
    S364_M_AX_CLAMP_전진_LS_이상 : BOOL; (* AT %MW2101.5 *) (* S364_M_AX_CLAMP_전진_LS_이상 *)
    S364_M_AX_CLAMP_후진_LS_이상 : BOOL; (* AT %MW2101.6 *) (* S364_M_AX_CLAMP_후진_LS_이상 *)
    S364_M_AX_LATCH_전진_LS_이상 : BOOL; (* AT %MW2100.5 *) (* S364_M_AX_LATCH_전진_LS_이상 *)
    S364_M_AX_LATCH_후진_LS_이상 : BOOL; (* AT %MW2100.6 *) (* S364_M_AX_LATCH_후진_LS_이상 *)
    S364_M_AX_LH_SLD_CLP_전진_LS_이상 : BOOL; (* AT %MW2103.5 *) (* S364_M_AX_LH_SLD_CLP_전진_LS_이상 *)
    S364_M_AX_LH_SLD_CLP_후진_LS_이상 : BOOL; (* AT %MW2103.6 *) (* S364_M_AX_LH_SLD_CLP_후진_LS_이상 *)
    S364_M_AX_LH_SLD_LAT_전진_LS_이상 : BOOL; (* AT %MW2102.5 *) (* S364_M_AX_LH_SLD_LAT_전진_LS_이상 *)
    S364_M_AX_LH_SLD_LAT_후진_LS_이상 : BOOL; (* AT %MW2102.6 *) (* S364_M_AX_LH_SLD_LAT_후진_LS_이상 *)
    S364_M_AX_LH_SLD_전진_LS_이상 : BOOL; (* AT %MW2107.5 *) (* S364_M_AX_LH_SLD_전진_LS_이상 *)
    S364_M_AX_LH_SLD_전진단 : BOOL; (* AT %MW2107.3 *) (* S364_M_AX_LH_SLD_전진단 *)
    S364_M_AX_LH_SLD_후진_LS_이상 : BOOL; (* AT %MW2107.6 *) (* S364_M_AX_LH_SLD_후진_LS_이상 *)
    S364_M_AX_LH_SLD_후진단 : BOOL; (* AT %MW2107.4 *) (* S364_M_AX_LH_SLD_후진단 *)
    S364_M_AX_RH_SLD_CLP_전진_LS_이상 : BOOL; (* AT %MW2111.5 *) (* S364_M_AX_RH_SLD_CLP_전진_LS_이상 *)
    S364_M_AX_RH_SLD_CLP_후진_LS_이상 : BOOL; (* AT %MW2111.6 *) (* S364_M_AX_RH_SLD_CLP_후진_LS_이상 *)
    S364_M_AX_RH_SLD_LAT_전진_LS_이상 : BOOL; (* AT %MW2110.5 *) (* S364_M_AX_RH_SLD_LAT_전진_LS_이상 *)
    S364_M_AX_RH_SLD_LAT_후진_LS_이상 : BOOL; (* AT %MW2110.6 *) (* S364_M_AX_RH_SLD_LAT_후진_LS_이상 *)
    S364_M_AX_RH_SLD_전진_LS_이상 : BOOL; (* AT %MW2115.5 *) (* S364_M_AX_RH_SLD_전진_LS_이상 *)
    S364_M_AX_RH_SLD_전진단 : BOOL; (* AT %MW2115.3 *) (* S364_M_AX_RH_SLD_전진단 *)
    S364_M_AX_RH_SLD_후진_LS_이상 : BOOL; (* AT %MW2115.6 *) (* S364_M_AX_RH_SLD_후진_LS_이상 *)
    S364_M_AX_RH_SLD_후진단 : BOOL; (* AT %MW2115.4 *) (* S364_M_AX_RH_SLD_후진단 *)
    S364_M_CTR_RACK_제품감지_유 : BOOL; (* AT %MW2002.8 *)
    S364_M_CTR_RACK_제품감지_이상 : BOOL; (* AT %MW2014.1 *)
    S364_M_FRT_PNL_제품감지_유 : BOOL; (* AT %MW2002.12 *)
    S364_M_FRT_PNL_제품감지_이상 : BOOL; (* AT %MW2014.3 *)
    S364_M_FRT_RACK_제품감지_유 : BOOL; (* AT %MW2002.6 *)
    S364_M_FRT_RACK_제품감지_이상 : BOOL; (* AT %MW2014.0 *)
    S364_M_LH_CP_OFF : BOOL; (* AT %MW2017.0 *) (* S364_M_LH_CP_OFF *)
    S364_M_OP_LC_이상 : BOOL; (* AT %MW2012.0 *) (* S364_M_OP_LC_이상 *)
    S364_M_OP_MAT_이상 : BOOL; (* AT %MW2012.1 *) (* S364_M_OP_MAT_이상 *)
    S364_M_RH_CP_OFF : BOOL; (* AT %MW2017.1 *) (* S364_M_RH_CP_OFF *)
    S364_M_RR_PNL_제품감지_유 : BOOL; (* AT %MW2002.14 *)
    S364_M_RR_PNL_제품감지_이상 : BOOL; (* AT %MW2014.4 *)
    S364_M_RR_RACK_제품감지_유 : BOOL; (* AT %MW2002.10 *)
    S364_M_RR_RACK_제품감지_이상 : BOOL; (* AT %MW2014.2 *)
    S364_M_공정_불간섭 : BOOL; (* AT %MW2004.1 *) (* S364_M_공정_불간섭 *)
    S364_M_공정_제품감지_무 : BOOL; (* AT %MW2002.5 *) (* S364_M_공정_제품감지_무 *)
    S364_M_공정_차종_유 : BOOL; (* AT %MW2002.0 *) (* S364_M_공정_차종_유 *)
    S364_M_자동_운전중 : BOOL; (* AT %MW2000.4 *) (* S364 자동운전중 *)
    S364_M_작업_완료 : BOOL; (* AT %MW2001.0 *) (* S364_M_작업_완료 *)
    S364_M_작업자_작업가능 : BOOL; (* AT %MW2004.8 *)
    S364_M_작업자_작업완료 : BOOL; (* AT %MW2001.1 *)
    S364_M_차종1_AX : BOOL; (* AT %MW10121.0 *) (* S364 M 차종1 AX *)
    S364_M_차종_OPT1_R_RACK_무 : BOOL; (* AT %MW10125.3 *) (* S364 M 차종 OPT1 R RACK 무 *)
    S364_M_총괄_CP_이상 : BOOL; (* AT %MW2009.7 *) (* S364 CP OFF 이상 *)
    S364_M_총괄_CT_이상 : BOOL; (* AT %MW2010.4 *) (* S364   TACK TIME 이상 *)
    S364_M_총괄_EOCR_이상 : BOOL; (* AT %MW2009.8 *) (* S364_M_총괄_EOCR_이상 *)
    S364_M_총괄_INV_이상 : BOOL; (* AT %MW2009.9 *) (* S364_M_총괄_INV_이상 *)
    S364_M_총괄_LS_이상 : BOOL; (* AT %MW2009.15 *) (* S364 LS 이상 *)
    S364_M_총괄_MATCH_이상 : BOOL; (* AT %MW2010.0 *) (* S364 매트SW 이상 *)
    S364_M_총괄_MC_이상 : BOOL; (* AT %MW2009.13 *) (* S364_M_총괄_MC_이상 *)
    S364_M_총괄_NFB_이상 : BOOL; (* AT %MW2009.11 *) (* S364_M_총괄_NFB_이상 *)
    S364_M_총괄_ROBOT_이상 : BOOL; (* AT %MW2010.1 *) (* S364 ROBOT 이상 *)
    S364_M_총괄_SAFETY_이상 : BOOL; (* AT %MW2009.2 *) (* S364 SAFETY 이상 *)
    S364_M_총괄_공기압_이상 : BOOL; (* AT %MW2009.3 *) (* S364 공기압 이상 *)
    S364_M_총괄_사양_이상 : BOOL; (* AT %MW2009.6 *) (* S364 사양 이상 *)
    S364_M_총괄_오버런_이상 : BOOL; (* AT %MW2009.12 *) (* S364_M_총괄_오버런_이상 *)
    S364_M_총괄_용접타점수_이상 : BOOL; (* AT %MW2010.2 *) (* S364 용접타점수 이상 *)
    S364_M_총괄_이상 : BOOL; (* AT %MW2009.0 *) (* S364_M_총괄_이상 *)
    S364_M_총괄_제품감지_이상 : BOOL; (* AT %MW2009.4 *) (* S364 제품감지 이상 *)
    S364_M_총괄_차종_이상 : BOOL; (* AT %MW2009.5 *) (* S364 차종 이상 *)
    S364_M_총괄_통신_이상 : BOOL; (* AT %MW2009.14 *) (* S364 통신이상 *)
    S364_RH_M_NODE_7_15_통신_이상 : BOOL; (* AT %MW2024.1 *)
    전체_M_이상_리셋 : BOOL; (* AT %MW308.2 *) (* ALL공정 PB 이상리셋 *)
END_VAR

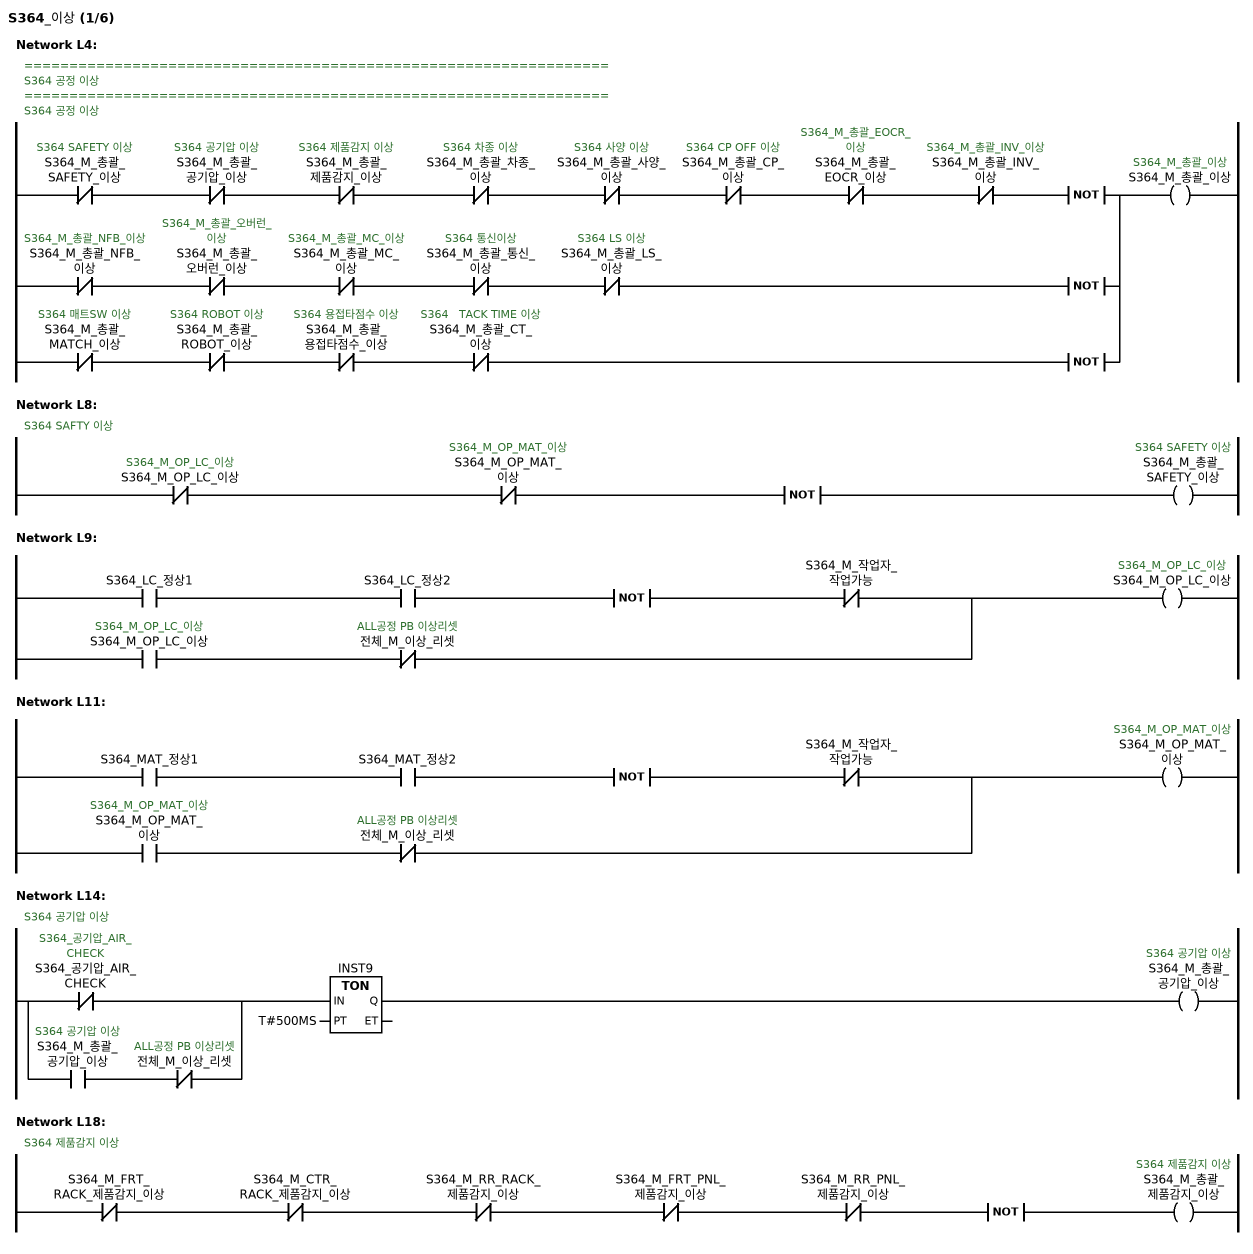
(* ================================================================= *)
(* S364 공정 이상 *)
(* ================================================================= *)
(* S364 공정 이상 *)
(* Rung L4 *)
S364_M_총괄_이상 := NOT (NOT S364_M_총괄_SAFETY_이상 AND NOT S364_M_총괄_공기압_이상 AND NOT S364_M_총괄_제품감지_이상 AND NOT S364_M_총괄_차종_이상 AND NOT S364_M_총괄_사양_이상 AND NOT S364_M_총괄_CP_이상 AND NOT S364_M_총괄_EOCR_이상 AND NOT S364_M_총괄_INV_이상) OR NOT (NOT S364_M_총괄_NFB_이상 AND NOT S364_M_총괄_오버런_이상 AND NOT S364_M_총괄_MC_이상 AND NOT S364_M_총괄_통신_이상 AND NOT S364_M_총괄_LS_이상) OR NOT (NOT S364_M_총괄_MATCH_이상 AND NOT S364_M_총괄_ROBOT_이상 AND NOT S364_M_총괄_용접타점수_이상 AND NOT S364_M_총괄_CT_이상);
(* S364 SAFTY 이상 *)
(* Rung L8 *)
S364_M_총괄_SAFETY_이상 := NOT (NOT S364_M_OP_LC_이상 AND NOT S364_M_OP_MAT_이상);
(* Rung L9 *)
S364_M_OP_LC_이상 := (NOT (S364_LC_정상1 AND S364_LC_정상2) AND NOT S364_M_작업자_작업가능) OR (S364_M_OP_LC_이상 AND NOT 전체_M_이상_리셋);
(* Rung L11 *)
S364_M_OP_MAT_이상 := (NOT (S364_MAT_정상1 AND S364_MAT_정상2) AND NOT S364_M_작업자_작업가능) OR (S364_M_OP_MAT_이상 AND NOT 전체_M_이상_리셋);
(* S364 공기압 이상 *)
(* Rung L14 *)
INST9(IN := NOT S364_공기압_AIR_CHECK OR (S364_M_총괄_공기압_이상 AND NOT 전체_M_이상_리셋), PT := T#500MS);
S364_M_총괄_공기압_이상 := INST9.Q;
(* S364 제품감지 이상 *)
(* Rung L18 *)
S364_M_총괄_제품감지_이상 := NOT (NOT S364_M_FRT_RACK_제품감지_이상 AND NOT S364_M_CTR_RACK_제품감지_이상 AND NOT S364_M_RR_RACK_제품감지_이상 AND NOT S364_M_FRT_PNL_제품감지_이상 AND NOT S364_M_RR_PNL_제품감지_이상);

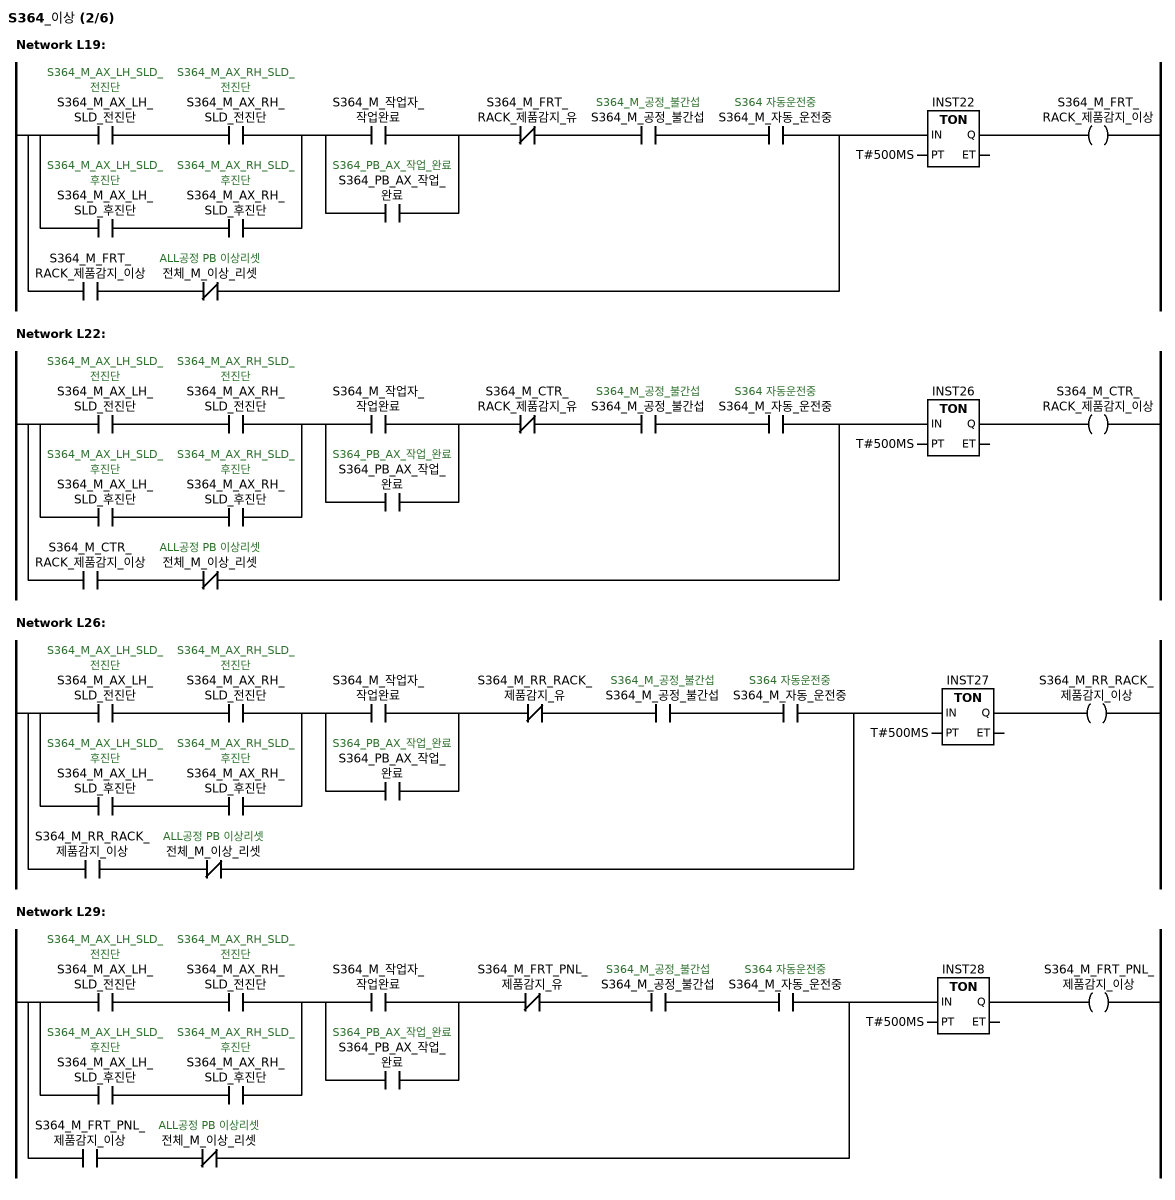
(* Rung L19 *)
INST22(IN := (((S364_M_AX_LH_SLD_전진단 AND S364_M_AX_RH_SLD_전진단) OR (S364_M_AX_LH_SLD_후진단 AND S364_M_AX_RH_SLD_후진단)) AND (S364_M_작업자_작업완료 OR S364_PB_AX_작업_완료) AND NOT S364_M_FRT_RACK_제품감지_유 AND S364_M_공정_불간섭 AND S364_M_자동_운전중) OR (S364_M_FRT_RACK_제품감지_이상 AND NOT 전체_M_이상_리셋), PT := T#500MS);
S364_M_FRT_RACK_제품감지_이상 := INST22.Q;
(* Rung L22 *)
INST26(IN := (((S364_M_AX_LH_SLD_전진단 AND S364_M_AX_RH_SLD_전진단) OR (S364_M_AX_LH_SLD_후진단 AND S364_M_AX_RH_SLD_후진단)) AND (S364_M_작업자_작업완료 OR S364_PB_AX_작업_완료) AND NOT S364_M_CTR_RACK_제품감지_유 AND S364_M_공정_불간섭 AND S364_M_자동_운전중) OR (S364_M_CTR_RACK_제품감지_이상 AND NOT 전체_M_이상_리셋), PT := T#500MS);
S364_M_CTR_RACK_제품감지_이상 := INST26.Q;
(* Rung L26 *)
INST27(IN := (((S364_M_AX_LH_SLD_전진단 AND S364_M_AX_RH_SLD_전진단) OR (S364_M_AX_LH_SLD_후진단 AND S364_M_AX_RH_SLD_후진단)) AND (S364_M_작업자_작업완료 OR S364_PB_AX_작업_완료) AND NOT S364_M_RR_RACK_제품감지_유 AND S364_M_공정_불간섭 AND S364_M_자동_운전중) OR (S364_M_RR_RACK_제품감지_이상 AND NOT 전체_M_이상_리셋), PT := T#500MS);
S364_M_RR_RACK_제품감지_이상 := INST27.Q;
(* Rung L29 *)
INST28(IN := (((S364_M_AX_LH_SLD_전진단 AND S364_M_AX_RH_SLD_전진단) OR (S364_M_AX_LH_SLD_후진단 AND S364_M_AX_RH_SLD_후진단)) AND (S364_M_작업자_작업완료 OR S364_PB_AX_작업_완료) AND NOT S364_M_FRT_PNL_제품감지_유 AND S364_M_공정_불간섭 AND S364_M_자동_운전중) OR (S364_M_FRT_PNL_제품감지_이상 AND NOT 전체_M_이상_리셋), PT := T#500MS);
S364_M_FRT_PNL_제품감지_이상 := INST28.Q;

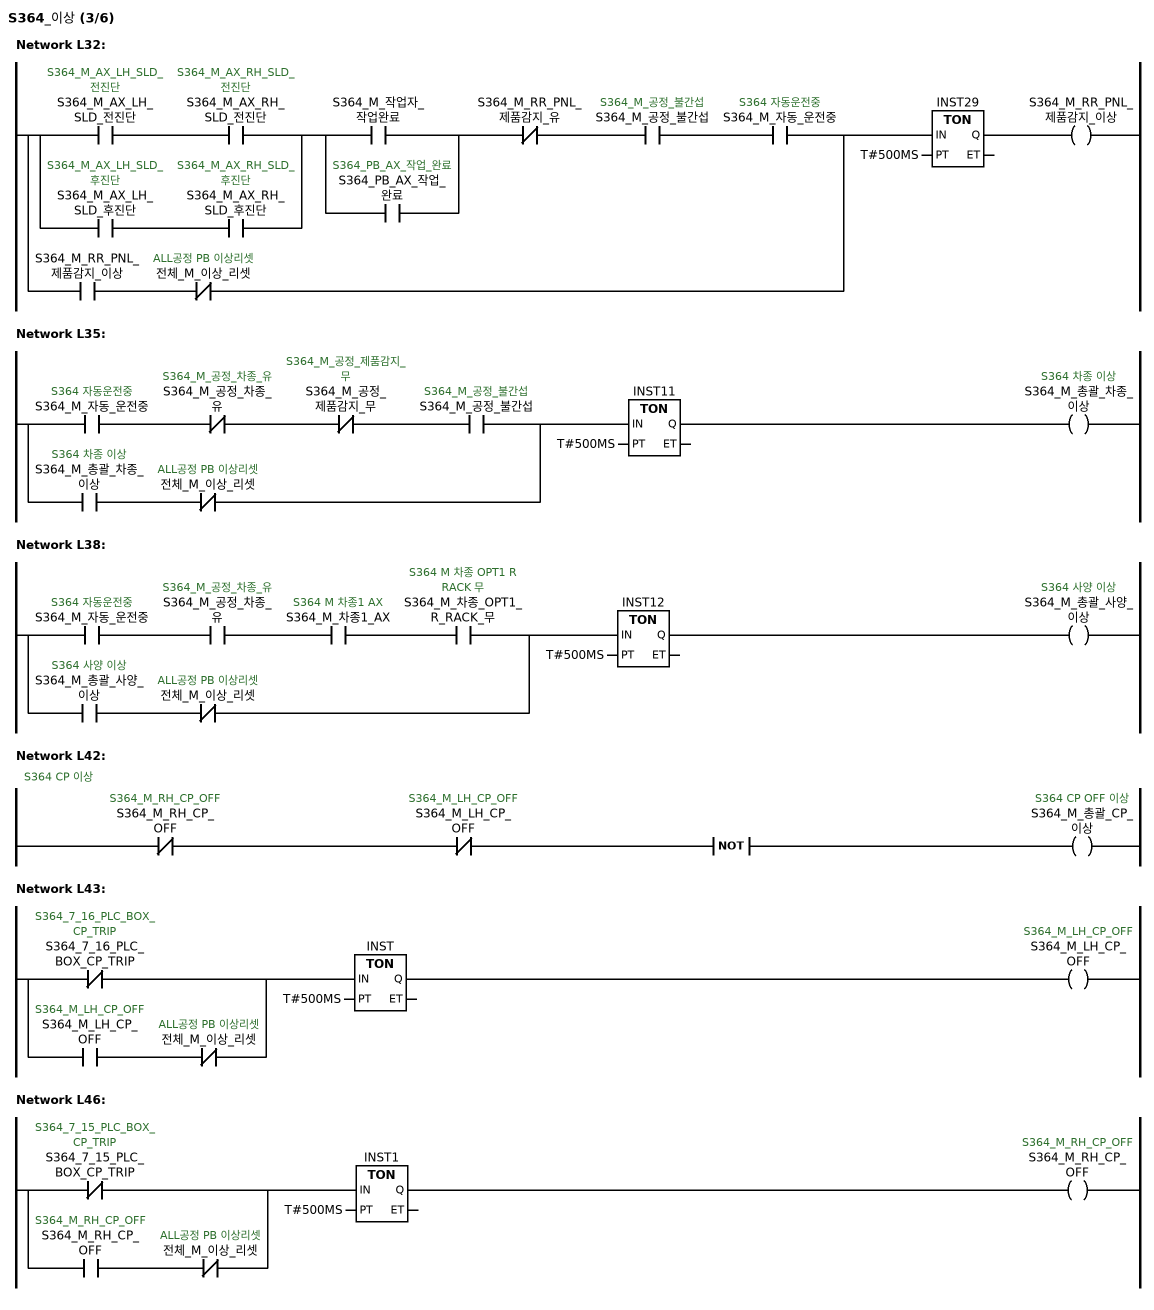
(* Rung L32 *)
INST29(IN := (((S364_M_AX_LH_SLD_전진단 AND S364_M_AX_RH_SLD_전진단) OR (S364_M_AX_LH_SLD_후진단 AND S364_M_AX_RH_SLD_후진단)) AND (S364_M_작업자_작업완료 OR S364_PB_AX_작업_완료) AND NOT S364_M_RR_PNL_제품감지_유 AND S364_M_공정_불간섭 AND S364_M_자동_운전중) OR (S364_M_RR_PNL_제품감지_이상 AND NOT 전체_M_이상_리셋), PT := T#500MS);
S364_M_RR_PNL_제품감지_이상 := INST29.Q;
(* Rung L35 *)
INST11(IN := (S364_M_자동_운전중 AND NOT S364_M_공정_차종_유 AND NOT S364_M_공정_제품감지_무 AND S364_M_공정_불간섭) OR (S364_M_총괄_차종_이상 AND NOT 전체_M_이상_리셋), PT := T#500MS);
S364_M_총괄_차종_이상 := INST11.Q;
(* Rung L38 *)
INST12(IN := (S364_M_자동_운전중 AND S364_M_공정_차종_유 AND S364_M_차종1_AX AND S364_M_차종_OPT1_R_RACK_무) OR (S364_M_총괄_사양_이상 AND NOT 전체_M_이상_리셋), PT := T#500MS);
S364_M_총괄_사양_이상 := INST12.Q;
(* S364 CP 이상 *)
(* Rung L42 *)
S364_M_총괄_CP_이상 := NOT (NOT S364_M_RH_CP_OFF AND NOT S364_M_LH_CP_OFF);
(* Rung L43 *)
INST(IN := NOT S364_7_16_PLC_BOX_CP_TRIP OR (S364_M_LH_CP_OFF AND NOT 전체_M_이상_리셋), PT := T#500MS);
S364_M_LH_CP_OFF := INST.Q;
(* Rung L46 *)
INST1(IN := NOT S364_7_15_PLC_BOX_CP_TRIP OR (S364_M_RH_CP_OFF AND NOT 전체_M_이상_리셋), PT := T#500MS);
S364_M_RH_CP_OFF := INST1.Q;

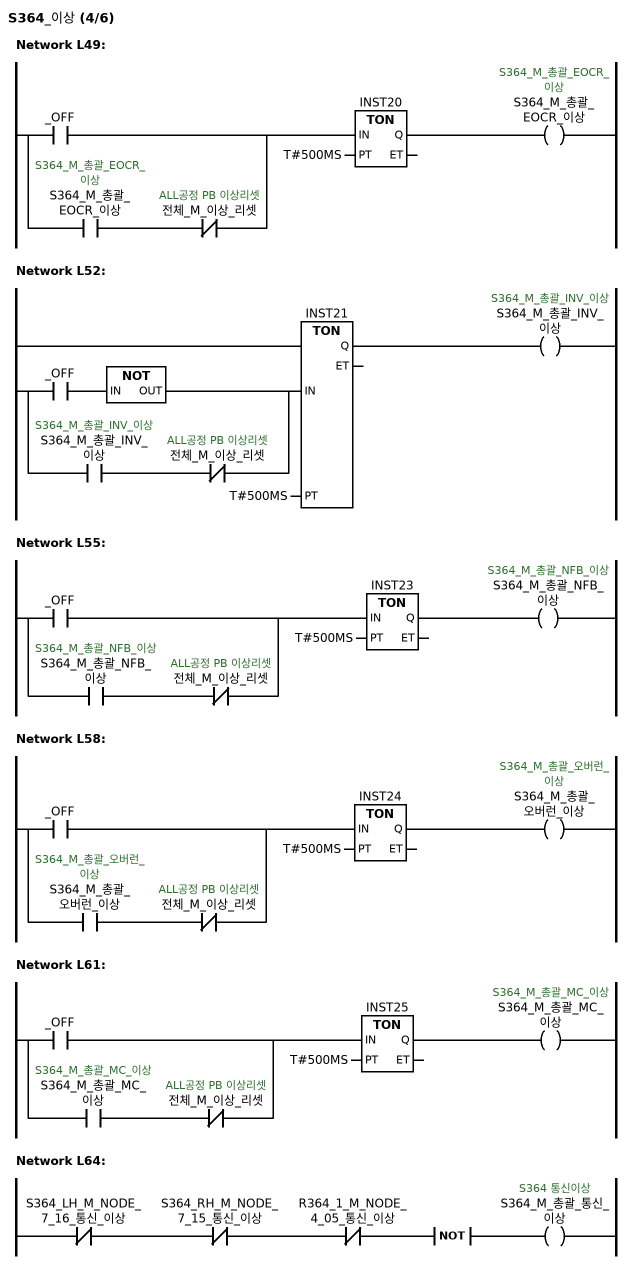
(* Rung L49 *)
INST20(IN := _OFF OR (S364_M_총괄_EOCR_이상 AND NOT 전체_M_이상_리셋), PT := T#500MS);
S364_M_총괄_EOCR_이상 := INST20.Q;
(* Rung L52 *)
INST21(IN := (NOT _OFF) OR (S364_M_총괄_INV_이상 AND NOT 전체_M_이상_리셋), PT := T#500MS);
S364_M_총괄_INV_이상 := INST21.Q;
(* Rung L55 *)
INST23(IN := _OFF OR (S364_M_총괄_NFB_이상 AND NOT 전체_M_이상_리셋), PT := T#500MS);
S364_M_총괄_NFB_이상 := INST23.Q;
(* Rung L58 *)
INST24(IN := _OFF OR (S364_M_총괄_오버런_이상 AND NOT 전체_M_이상_리셋), PT := T#500MS);
S364_M_총괄_오버런_이상 := INST24.Q;
(* Rung L61 *)
INST25(IN := _OFF OR (S364_M_총괄_MC_이상 AND NOT 전체_M_이상_리셋), PT := T#500MS);
S364_M_총괄_MC_이상 := INST25.Q;
(* Rung L64 *)
S364_M_총괄_통신_이상 := NOT (NOT S364_LH_M_NODE_7_16_통신_이상 AND NOT S364_RH_M_NODE_7_15_통신_이상 AND NOT R364_1_M_NODE_4_05_통신_이상);

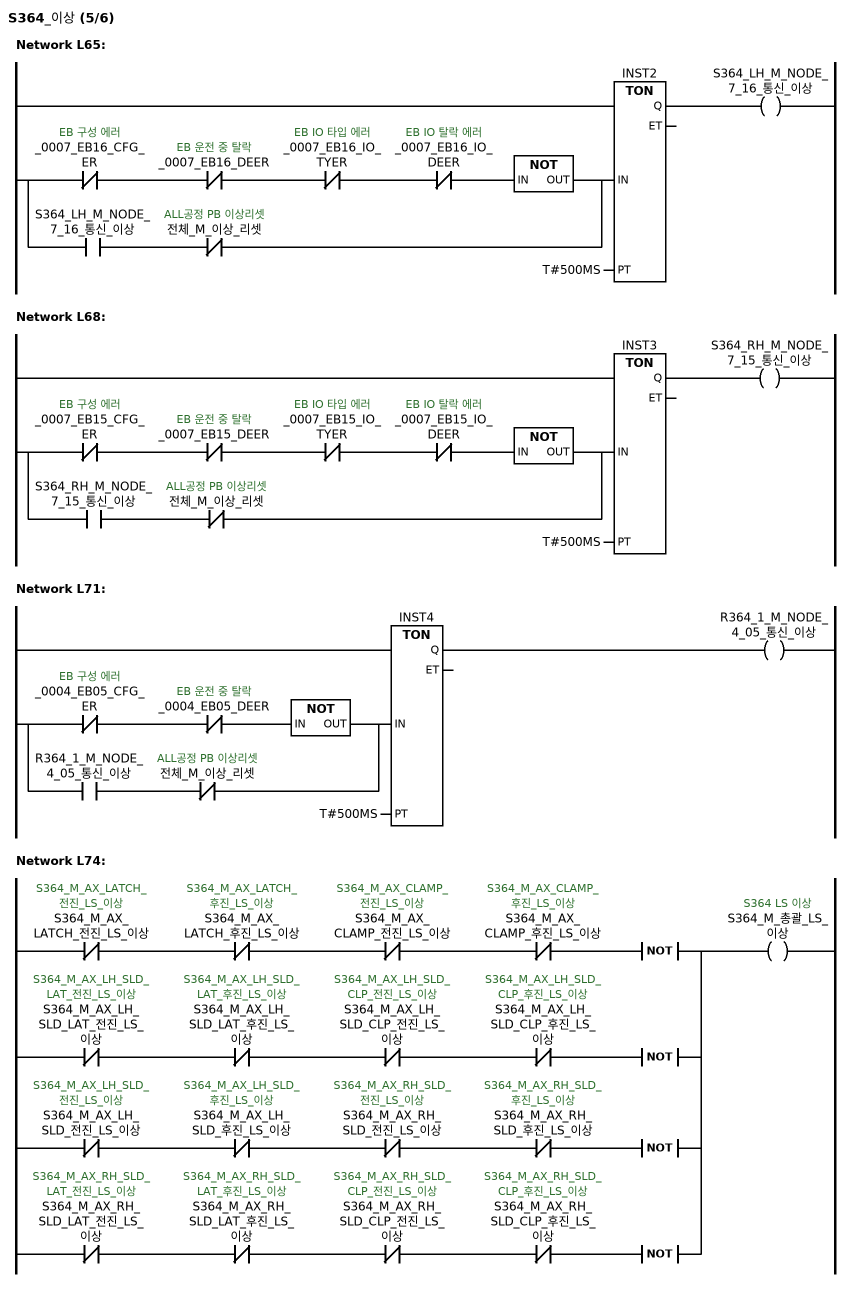
(* Rung L65 *)
INST2(IN := (NOT (NOT _0007_EB16_CFG_ER AND NOT _0007_EB16_DEER AND NOT _0007_EB16_IO_TYER AND NOT _0007_EB16_IO_DEER)) OR (S364_LH_M_NODE_7_16_통신_이상 AND NOT 전체_M_이상_리셋), PT := T#500MS);
S364_LH_M_NODE_7_16_통신_이상 := INST2.Q;
(* Rung L68 *)
INST3(IN := (NOT (NOT _0007_EB15_CFG_ER AND NOT _0007_EB15_DEER AND NOT _0007_EB15_IO_TYER AND NOT _0007_EB15_IO_DEER)) OR (S364_RH_M_NODE_7_15_통신_이상 AND NOT 전체_M_이상_리셋), PT := T#500MS);
S364_RH_M_NODE_7_15_통신_이상 := INST3.Q;
(* Rung L71 *)
INST4(IN := (NOT (NOT _0004_EB05_CFG_ER AND NOT _0004_EB05_DEER)) OR (R364_1_M_NODE_4_05_통신_이상 AND NOT 전체_M_이상_리셋), PT := T#500MS);
R364_1_M_NODE_4_05_통신_이상 := INST4.Q;
(* Rung L74 *)
S364_M_총괄_LS_이상 := NOT (NOT S364_M_AX_LATCH_전진_LS_이상 AND NOT S364_M_AX_LATCH_후진_LS_이상 AND NOT S364_M_AX_CLAMP_전진_LS_이상 AND NOT S364_M_AX_CLAMP_후진_LS_이상) OR NOT (NOT S364_M_AX_LH_SLD_LAT_전진_LS_이상 AND NOT S364_M_AX_LH_SLD_LAT_후진_LS_이상 AND NOT S364_M_AX_LH_SLD_CLP_전진_LS_이상 AND NOT S364_M_AX_LH_SLD_CLP_후진_LS_이상) OR NOT (NOT S364_M_AX_LH_SLD_전진_LS_이상 AND NOT S364_M_AX_LH_SLD_후진_LS_이상 AND NOT S364_M_AX_RH_SLD_전진_LS_이상 AND NOT S364_M_AX_RH_SLD_후진_LS_이상) OR NOT (NOT S364_M_AX_RH_SLD_LAT_전진_LS_이상 AND NOT S364_M_AX_RH_SLD_LAT_후진_LS_이상 AND NOT S364_M_AX_RH_SLD_CLP_전진_LS_이상 AND NOT S364_M_AX_RH_SLD_CLP_후진_LS_이상);

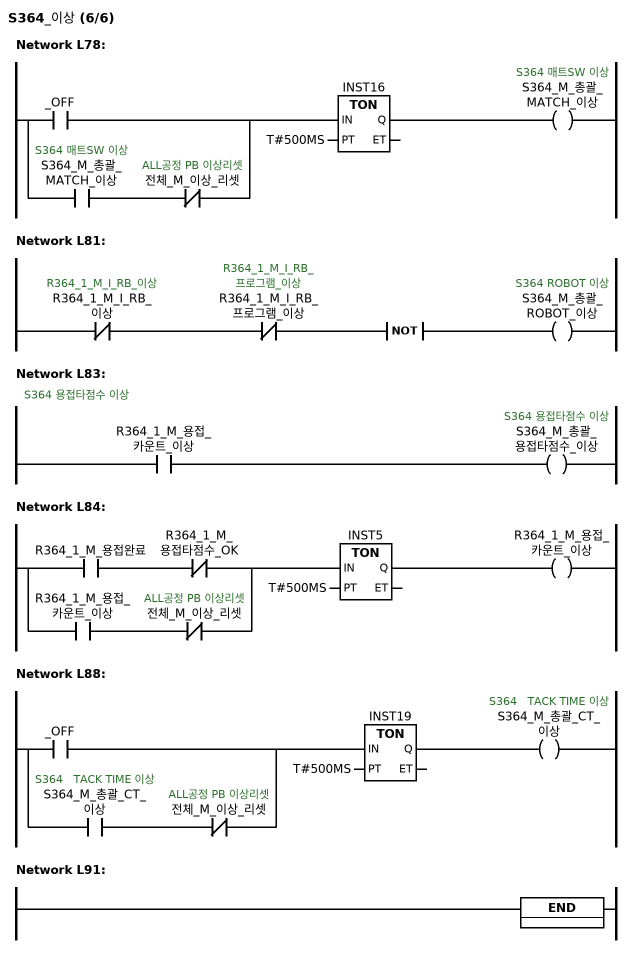
(* Rung L78 *)
INST16(IN := _OFF OR (S364_M_총괄_MATCH_이상 AND NOT 전체_M_이상_리셋), PT := T#500MS);
S364_M_총괄_MATCH_이상 := INST16.Q;
(* Rung L81 *)
S364_M_총괄_ROBOT_이상 := NOT (NOT R364_1_M_I_RB_이상 AND NOT R364_1_M_I_RB_프로그램_이상);
(* S364 용접타점수 이상 *)
(* Rung L83 *)
S364_M_총괄_용접타점수_이상 := R364_1_M_용접_카운트_이상;
(* Rung L84 *)
INST5(IN := (R364_1_M_용접완료 AND NOT R364_1_M_용접타점수_OK) OR (R364_1_M_용접_카운트_이상 AND NOT 전체_M_이상_리셋), PT := T#500MS);
R364_1_M_용접_카운트_이상 := INST5.Q;
(* Rung L88 *)
INST19(IN := _OFF OR (S364_M_총괄_CT_이상 AND NOT 전체_M_이상_리셋), PT := T#500MS);
S364_M_총괄_CT_이상 := INST19.Q;
(* Rung L91 *)
END();
END_PROGRAM

PROGRAM S365_유틸리티 (* task: 스캔 프로그램 *)
VAR_EXTERNAL RETAIN
    ALWAYS_ON : BOOL; (* AT %MW3.1 *) (* 항시 ON *)
    HMI_M_선택_MOD_S362 : BOOL; (* AT %MW6.0 *) (* HMI M 선택 MOD S362 *)
    HMI_M_선택_MOD_S365 : BOOL; (* AT %MW6.3 *) (* HMI M 선택 MOD S365 *)
    S362_M_작업완료_SET_PLS : BOOL; (* AT %MW1000.8 *) (* S362 M 작업완료 SET PLS *)
    S362_M_작업완료_리셋_PLS : BOOL; (* AT %MW1000.9 *) (* S362 M 작업완료 리셋 PLS *)
    S362_M_총괄_이상 : BOOL; (* AT %MW1009.0 *) (* S362_M_총괄_이상 *)
    S364_M_공정_차종_무 : BOOL; (* AT %MW2002.1 *) (* S364_M_공정_차종_무 *)
    S364_M_공정_차종_유 : BOOL; (* AT %MW2002.0 *) (* S364_M_공정_차종_유 *)
    S365_M_BYPASS_보조 : BOOL; (* AT %MW2503.15 *) (* S365 M BYPASS 보조 *)
    S365_M_R361_1_안착완료 : BOOL; (* AT %MW2501.1 *)
    S365_M_R361_1_언로딩완료 : BOOL; (* AT %MW2501.2 *)
    S365_M_SEQ : WORD; (* AT %MW10140 *) (* S365 M SEQ *)
    S365_M_공정_불간섭 : BOOL; (* AT %MW2504.1 *) (* S365_M_공정_불간섭 *)
    S365_M_공정_원위치 : BOOL; (* AT %MW2504.0 *) (* S365_M_공정_원위치 *)
    S365_M_공정_제품감지_무 : BOOL; (* AT %MW2501.4 *) (* S365_M_공정_제품감지_무 *)
    S365_M_공정_제품감지_유 : BOOL; (* AT %MW2501.3 *) (* S365_M_공정_제품감지_유 *)
    S365_M_공정_차종_무 : BOOL; (* AT %MW2502.1 *) (* S365_M_공정_차종_무 *)
    S365_M_공정_차종_유 : BOOL; (* AT %MW2502.0 *) (* S365_M_공정_차종_유 *)
    S365_M_수동모드 : BOOL; (* AT %MW2500.3 *) (* S365 선택 수동모드 *)
    S365_M_운전준비_ON : BOOL; (* AT %MW2500.0 *) (* S365 운전준비 ON *)
    S365_M_자동_START : BOOL; (* AT %MW2500.5 *) (* S365 자동운전중 *)
    S365_M_자동_운전중 : BOOL; (* AT %MW2500.4 *) (* S365 자동운전중 *)
    S365_M_자동모드 : BOOL; (* AT %MW2500.1 *) (* S365 선택 자동모드 *)
    S365_M_작업_완료 : BOOL; (* AT %MW2501.0 *) (* S365_M_작업_완료 *)
    S365_M_작업완료_SET_PLS : BOOL; (* AT %MW2500.8 *) (* S365 M 작업완료 SET PLS *)
    S365_M_작업완료_리셋_PLS : BOOL; (* AT %MW2500.9 *) (* S365 M 작업완료 리셋 PLS *)
    S365_M_차종1_AX : BOOL; (* AT %MW10141.0 *) (* S365 M 차종1 AX *)
    S365_M_차종1_B : BOOL; (* AT %MW10141.1 *) (* S365 M 차종1 B *)
    S365_M_차종1_C : BOOL; (* AT %MW10141.2 *) (* S365 M 차종1 C *)
    S365_M_차종1_D : BOOL; (* AT %MW10141.3 *) (* S365 M 차종1 D *)
    S365_M_차종1_E : BOOL; (* AT %MW10141.4 *) (* S365 M 차종1 E *)
    S365_M_차종1_F : BOOL; (* AT %MW10141.5 *) (* S365 M 차종1 F *)
    S365_M_차종1_G : BOOL; (* AT %MW10141.6 *) (* S365 M 차종1 G *)
    S365_M_차종1_H : BOOL; (* AT %MW10141.7 *) (* S365 M 차종1 H *)
    S365_M_차종2_3DR : BOOL; (* AT %MW10141.8 *) (* S365 M 차종2 3DR *)
    S365_M_차종2_4DR : BOOL; (* AT %MW10141.9 *) (* S365 M 차종2 4DR *)
    S365_M_차종2_5DR : BOOL; (* AT %MW10141.10 *) (* S365 M 차종2 5DR *)
    S365_M_차종2_SP1 : BOOL; (* AT %MW10141.12 *) (* S365 M 차종2 SP1 *)
    S365_M_차종2_SP2 : BOOL; (* AT %MW10141.13 *) (* S365 M 차종2 SP2 *)
    S365_M_차종2_WGN : BOOL; (* AT %MW10141.11 *) (* S365 M 차종2 WGN *)
    S365_M_차종3_LHD : BOOL; (* AT %MW10141.14 *) (* S365 M 차종3 LHD *)
    S365_M_차종3_RHD : BOOL; (* AT %MW10141.15 *) (* S365 M 차종3 RHD *)
    S365_M_차종4_EEC : BOOL; (* AT %MW10142.3 *) (* S365 M 차종4 EEC *)
    S365_M_차종4_SP1 : BOOL; (* AT %MW10142.8 *) (* S365 M 차종4 SP1 *)
    S365_M_차종4_SP2 : BOOL; (* AT %MW10142.9 *) (* S365 M 차종4 SP2 *)
    S365_M_차종4_SP3 : BOOL; (* AT %MW10142.11 *) (* S365 M 차종4 SP3 *)
    S365_M_차종4_SP4 : BOOL; (* AT %MW10142.12 *) (* S365 M 차종4 SP4 *)
    S365_M_차종4_SP5 : BOOL; (* AT %MW10142.13 *) (* S365 M 차종4 SP5 *)
    S365_M_차종4_SP6 : BOOL; (* AT %MW10142.14 *) (* S365 M 차종4 SP6 *)
    S365_M_차종4_SP7 : BOOL; (* AT %MW10142.15 *) (* S365 M 차종4 SP7 *)
    S365_M_차종4_내수 : BOOL; (* AT %MW10142.0 *) (* S365 M 차종4 내수 *)
    S365_M_차종4_러시아 : BOOL; (* AT %MW10142.10 *) (* S365 M 차종4 러시아 *)
    S365_M_차종4_북미 : BOOL; (* AT %MW10142.2 *) (* S365 M 차종4 북미 *)
    S365_M_차종4_브라질 : BOOL; (* AT %MW10142.7 *) (* S365 M 차종4 브라질 *)
    S365_M_차종4_수출 : BOOL; (* AT %MW10142.1 *) (* S365 M 차종4 수출 *)
    S365_M_차종4_중국 : BOOL; (* AT %MW10142.6 *) (* S365 M 차종4 중국 *)
    S365_M_차종4_중동 : BOOL; (* AT %MW10142.5 *) (* S365 M 차종4 중동 *)
    S365_M_차종4_호주 : BOOL; (* AT %MW10142.4 *) (* S365 M 차종4 호주 *)
    S365_M_차종5_AT : BOOL; (* AT %MW10143.1 *) (* S365 M 차종5 AT *)
    S365_M_차종5_MT : BOOL; (* AT %MW10143.0 *) (* S365 M 차종5 MT *)
    S365_M_차종5_SP1 : BOOL; (* AT %MW10143.2 *) (* S365 M 차종5 SP1 *)
    S365_M_차종6_DSROOF : BOOL; (* AT %MW10143.6 *) (* S365 M 차종6 DSROOF *)
    S365_M_차종6_SP1 : BOOL; (* AT %MW10143.7 *) (* S365 M 차종6 SP1 *)
    S365_M_차종6_썬루프 : BOOL; (* AT %MW10143.4 *) (* S365 M 차종6 썬루프 *)
    S365_M_차종6_일반루프 : BOOL; (* AT %MW10143.3 *) (* S365 M 차종6 일반루프 *)
    S365_M_차종6_파노라마루프 : BOOL; (* AT %MW10143.5 *) (* S365 M 차종6 파노라마루프 *)
    S365_M_차종7_DSL : BOOL; (* AT %MW10143.9 *) (* S365 M 차종7 DSL *)
    S365_M_차종7_GSL : BOOL; (* AT %MW10143.8 *) (* S365 M 차종7 GSL *)
    S365_M_차종7_SP1 : BOOL; (* AT %MW10143.10 *) (* S365 M 차종7 SP1 *)
    S365_M_차종7_SP2 : BOOL; (* AT %MW10143.11 *) (* S365 M 차종7 SP2 *)
    S365_M_차종7_SP3 : BOOL; (* AT %MW10143.12 *) (* S365 M 차종7 SP3 *)
    S365_M_차종7_SP4 : BOOL; (* AT %MW10143.13 *) (* S365 M 차종7 SP4 *)
    S365_M_차종7_SP5 : BOOL; (* AT %MW10143.14 *) (* S365 M 차종7 SP5 *)
    S365_M_차종7_SP6 : BOOL; (* AT %MW10143.15 *) (* S365 M 차종7 SP6 *)
    S365_M_차종8_2WD : BOOL; (* AT %MW10144.0 *) (* S365 M 차종8 2WD *)
    S365_M_차종8_4WD : BOOL; (* AT %MW10144.1 *) (* S365 M 차종8 4WD *)
    S365_M_차종8_SP1 : BOOL; (* AT %MW10144.2 *) (* S365 M 차종8 SP1 *)
    S365_M_차종9_MPI : BOOL; (* AT %MW10144.3 *) (* S365 M 차종9 MPI *)
    S365_M_차종9_SP1 : BOOL; (* AT %MW10144.5 *) (* S365 M 차종9 SP1 *)
    S365_M_차종9_SP10 : BOOL; (* AT %MW10144.14 *) (* S365 M 차종9 SP10 *)
    S365_M_차종9_SP11 : BOOL; (* AT %MW10144.15 *) (* S365 M 차종9 SP11 *)
    S365_M_차종9_SP2 : BOOL; (* AT %MW10144.6 *) (* S365 M 차종9 SP2 *)
    S365_M_차종9_SP3 : BOOL; (* AT %MW10144.7 *) (* S365 M 차종9 SP3 *)
    S365_M_차종9_SP4 : BOOL; (* AT %MW10144.8 *) (* S365 M 차종9 SP4 *)
    S365_M_차종9_SP5 : BOOL; (* AT %MW10144.9 *) (* S365 M 차종9 SP5 *)
    S365_M_차종9_SP6 : BOOL; (* AT %MW10144.10 *) (* S365 M 차종9 SP6 *)
    S365_M_차종9_SP7 : BOOL; (* AT %MW10144.11 *) (* S365 M 차종9 SP7 *)
    S365_M_차종9_SP8 : BOOL; (* AT %MW10144.12 *) (* S365 M 차종9 SP8 *)
    S365_M_차종9_SP9 : BOOL; (* AT %MW10144.13 *) (* S365 M 차종9 SP9 *)
    S365_M_차종9_T_GDI : BOOL; (* AT %MW10144.4 *) (* S365 M 차종9 T GDI *)
    S365_M_차종_OPT1_R_RACK_무 : BOOL; (* AT %MW10145.3 *) (* S365 M 차종 OPT1 R RACK 무 *)
    S365_M_차종_OPT1_R_RACK_유 : BOOL; (* AT %MW10145.2 *) (* S365 M 차종 OPT1 R RACK 유 *)
    S365_M_차종_OPT1_S_REP_EATER_무 : BOOL; (* AT %MW10145.7 *) (* S365 M 차종 OPT1 S REP EATER 무 *)
    S365_M_차종_OPT1_S_REP_EATER_유 : BOOL; (* AT %MW10145.6 *) (* S365 M 차종 OPT1 S REP EATER 유 *)
    S365_M_차종_OPT1_VAN_무 : BOOL; (* AT %MW10145.9 *) (* S365 M 차종 OPT1 VAN 무 *)
    S365_M_차종_OPT1_VAN_유 : BOOL; (* AT %MW10145.8 *) (* S365 M 차종 OPT1 VAN 유 *)
    S365_M_차종_OPT1_슬라이딩_무 : BOOL; (* AT %MW10145.1 *) (* S365 M 차종 OPT1 슬라이딩 무 *)
    S365_M_차종_OPT1_슬라이딩_유 : BOOL; (* AT %MW10145.0 *) (* S365 M 차종 OPT1 슬라이딩 유 *)
    S365_M_차종_OPT1_폴딩_무 : BOOL; (* AT %MW10145.5 *) (* S365 M 차종 OPT1 폴딩 무 *)
    S365_M_차종_OPT1_폴딩_유 : BOOL; (* AT %MW10145.4 *) (* S365 M 차종 OPT1 폴딩 유 *)
    S365_M_차종_공대차 : BOOL; (* AT %MW10150.12 *) (* S365 M 차종 공대차 *)
    S365_M_차종_공차 : BOOL; (* AT %MW10150.10 *) (* S365 M 차종 공차 *)
    S365_M_차종_불량차 : BOOL; (* AT %MW10150.11 *) (* S365 M 차종 불량차 *)
    S365_M_총괄_이상 : BOOL; (* AT %MW2509.0 *) (* S365_M_총괄_이상 *)
    전체_M_GATE_자동기동 : BOOL; (* AT %MW308.1 *) (* 전체_M_자동_운전 *)
    전체_라인_M_총괄_SAFETY_이상 : BOOL; (* AT %MW300.2 *) (* ALL공정 SAFETY  이상총괄 *)
    전체_라인_M_총괄_공기압_이상 : BOOL; (* AT %MW300.3 *) (* ALL공정 공기압 이상총괄 *)
    전체_라인_M_총괄_비상정지_이상 : BOOL; (* AT %MW300.1 *) (* ALL공정 비상정지 이상총괄 *)
    전체_라인_M_총괄_이상 : BOOL; (* AT %MW300.0 *) (* ALL공정 총괄이상 *)
END_VAR
VAR_EXTERNAL
    HOP_PBL_365_8_자동_운전 : BOOL; (* AT %MW87500.7 *) (* HOP_PBL_365_8_자동_운전 *)
    HOP_PBL_운전준비_ON : BOOL; (* AT %MW87500.0 *) (* HOP_PBL_운전준비_ON *)
    HOP_SSP_365_8_수동_선택 : BOOL; (* AT %MW87500.6 *) (* HOP_SSP_365_8_수동_선택 *)
    HOP_SSP_365_8_자동_선택 : BOOL; (* AT %MW87500.5 *) (* HOP_SSP_365_8_자동_선택 *)
    MCP_PBL_365_8_자동_운전 : BOOL; (* AT %MW87630.7 *) (* MCP PBL 365~8 자동기동 *)
    MCP_PBL_운전준비_ON : BOOL; (* AT %MW87630.0 *) (* MCP_PBL_운전준비_ON *)
    MCP_SPB_작업완료_RESET : BOOL; (* AT %MW87631.6 *) (* MCP_SPB_작업완료_RESET *)
    MCP_SPB_작업완료_SET : BOOL; (* AT %MW87631.7 *) (* MCP_SPB_작업완료_SET *)
    MCP_SSP_365_8_수동_선택 : BOOL; (* AT %MW87630.5 *) (* MCP_SSP_365_8_수동_선택 *)
    MCP_SSP_365_8_자동_선택 : BOOL; (* AT %MW87630.6 *) (* MCP_SSP_365_8_자동_선택 *)
    R361_1_M_I_RB_2차_작업완료 : BOOL; (* AT %MW20011.3 *) (* R361_1_M_I_RB_2차_작업완료 *)
    R361_1_M_I_RB_3차_작업완료 : BOOL; (* AT %MW20011.4 *) (* R361_1_M_I_RB_3차_작업완료 *)
    R361_1_M_I_RB_간섭무_1 : BOOL; (* AT %MW20012.0 *) (* R361_1_M_I_RB_간섭무_1 *)
    R361_1_M_I_RB_원위치 : BOOL; (* AT %MW20010.3 *) (* R361_1_M_I_RB_원위치 *)
    R361_2_M_I_RB_2차_작업완료 : BOOL; (* AT %MW20021.3 *) (* R361_2_M_I_RB_2차_작업완료 *)
    R361_2_M_I_RB_간섭무_1 : BOOL; (* AT %MW20022.0 *) (* R361_2_M_I_RB_간섭무_1 *)
    R361_2_M_I_RB_원위치 : BOOL; (* AT %MW20020.3 *) (* R361_2_M_I_RB_원위치 *)
    S365_PHS_ROOF_PNL_썬루프_감지 : BOOL; (* AT %MW86010.3 *)
    S365_PRS_ROOF_PNL_제품감지1 : BOOL; (* AT %MW86010.0 *)
    S365_PRS_ROOF_PNL_제품감지2 : BOOL; (* AT %MW86010.1 *)
    S365_PRS_ROOF_PNL_제품감지3 : BOOL; (* AT %MW86010.2 *)
END_VAR
VAR
    S365_READY : TON;
    T365_AUTO : TON;
END_VAR
VAR
    _t1 : BOOL;
END_VAR

